// TIA Portal V20 export
FUNCTION_BLOCK "Sequence_3_SideTapeFixStage"   // FB32853, LAD
TITLE = Sequence
// Sequence template programmend in ladder logic
// stored: IsIECCheckEnabled true, MemoryReserve 100, Namespace Unit1.Em4, SetENOAutomatically true
   VAR_INPUT
      unitStatus { ExternalAccessible := 'False'; ExternalVisible := 'False'; ExternalWritable := 'False'} : "LAF_typeUnitStatus";   // Current unit status o be used in this EM
   END_VAR
   VAR
      instSequenceLADControl { ExternalWritable := 'False'} : "LAF_ControlLadSequence";
      instSequenceLADStatus { ExternalWritable := 'False'} : "LAF_StatusLadSequence";
      NoDataCheck { S7_SetPoint := 'True'} : "LER_typePartData";
      statTonTime { ExternalWritable := 'False'} : Array[0..9999] of TON_TIME;
   END_VAR
   VAR_TEMP
      tempCustomerAction : Bool;   // Placeholder for possible actions
      tempDo_nothing_and_wait_for_init : Bool;   // Placeholder for doing nothing
      tempSafeStateCondition : Bool;   // Temp Condition for the equipment module to be in a safe state
   END_VAR
   VAR CONSTANT
      stepDelayTime : Time := T#100ms;
      actionDelayTime : Time := T#1s;
      lowDelayTime : Time := T#300ms;
      STEP_IDLE : DInt := 1;
      JOB_1_STEP_01 : DInt := 101;
      JOB_1_STEP_10 : DInt := 110;
      JOB_1_STEP_11 : DInt := 111;
      JOB_1_STEP_20 : DInt := 120;
      JOB_1_STEP_30 : DInt := 130;
      JOB_1_STEP_31 : DInt := 131;
      JOB_1_STEP_32 : DInt := 132;
      JOB_1_STEP_33 : DInt := 133;
      JOB_1_STEP_34 : DInt := 134;
      JOB_1_STEP_35 : DInt := 135;
      JOB_1_STEP_40 : DInt := 140;
      JOB_1_STEP_50 : DInt := 150;
      JOB_1_STEP_60 : DInt := 160;
      JOB_1_STEP_70 : DInt := 170;
      JOB_1_STEP_80 : DInt := 180;
      JOB_1_STEP_90 : DInt := 190;
      JOB_2_STEP_01 : DInt := 201;
      JOB_2_STEP_10 : DInt := 210;
      JOB_2_STEP_11 : DInt := 211;
      JOB_2_STEP_12 : DInt := 212;
      JOB_2_STEP_13 : DInt := 213;
      JOB_2_STEP_14 : DInt := 214;
      JOB_2_STEP_20 : DInt := 220;
      JOB_2_STEP_21 : DInt := 221;
      JOB_2_STEP_22 : DInt := 222;
      JOB_2_STEP_23 : DInt := 223;
      JOB_2_STEP_24 : DInt := 224;
      JOB_2_STEP_30 : DInt := 230;
      JOB_2_STEP_31 : DInt := 231;
      JOB_2_STEP_32 : DInt := 232;
      JOB_2_STEP_40 : DInt := 240;
      JOB_2_STEP_50 : DInt := 250;
      JOB_2_STEP_60 : DInt := 260;
      JOB_2_STEP_70 : DInt := 270;
      JOB_2_STEP_80 : DInt := 280;
      JOB_2_STEP_90 : DInt := 290;
      JOB_3_STEP_01 : DInt := 301;
      JOB_3_STEP_02 : DInt := 302;
      JOB_3_STEP_03 : DInt := 303;
      JOB_3_STEP_10 : DInt := 310;
      JOB_3_STEP_11 : DInt := 311;
      JOB_3_STEP_12 : DInt := 312;
      JOB_3_STEP_13 : DInt := 313;
      JOB_3_STEP_14 : DInt := 314;
      JOB_3_STEP_15 : DInt := 315;
      JOB_3_STEP_16 : DInt := 316;
      JOB_3_STEP_17 : DInt := 317;
      JOB_3_STEP_20 : DInt := 320;
      JOB_3_STEP_21 : DInt := 321;
      JOB_3_STEP_22 : DInt := 322;
      JOB_3_STEP_23 : DInt := 323;
      JOB_3_STEP_24 : DInt := 324;
      JOB_3_STEP_25 : DInt := 325;
      JOB_3_STEP_26 : DInt := 326;
      JOB_3_STEP_27 : DInt := 327;
      JOB_3_STEP_30 : DInt := 330;
      JOB_3_STEP_31 : DInt := 331;
      JOB_3_STEP_32 : DInt := 332;
      JOB_3_STEP_33 : DInt := 333;
      JOB_3_STEP_34 : DInt := 334;
      JOB_3_STEP_35 : DInt := 335;
      JOB_3_STEP_36 : DInt := 336;
      JOB_3_STEP_37 : DInt := 337;
      JOB_3_STEP_40 : DInt := 340;
      JOB_3_STEP_41 : DInt := 341;
      JOB_3_STEP_42 : DInt := 342;
      JOB_3_STEP_43 : DInt := 343;
      JOB_3_STEP_44 : DInt := 344;
      JOB_3_STEP_45 : DInt := 345;
      JOB_3_STEP_46 : DInt := 346;
      JOB_3_STEP_47 : DInt := 347;
      JOB_3_STEP_50 : DInt := 350;
      JOB_3_STEP_60 : DInt := 360;
      JOB_3_STEP_70 : DInt := 370;
      JOB_3_STEP_80 : DInt := 380;
      JOB_3_STEP_90 : DInt := 390;
      JOB_4_STEP_01 : DInt := 401;
      JOB_4_STEP_10 : DInt := 410;
      JOB_4_STEP_11 : DInt := 411;
      JOB_4_STEP_12 : DInt := 412;
      JOB_4_STEP_20 : DInt := 420;
      JOB_4_STEP_21 : DInt := 421;
      JOB_4_STEP_22 : DInt := 422;
      JOB_4_STEP_23 : DInt := 423;
      JOB_4_STEP_24 : DInt := 424;
      JOB_4_STEP_25 : DInt := 425;
      JOB_4_STEP_30 : DInt := 430;
      JOB_4_STEP_40 : DInt := 440;
      JOB_4_STEP_50 : DInt := 450;
      JOB_4_STEP_60 : DInt := 460;
      JOB_4_STEP_70 : DInt := 470;
      JOB_4_STEP_80 : DInt := 480;
      JOB_4_STEP_90 : DInt := 490;
      JOB_5_STEP_01 : DInt := 501;
      JOB_5_STEP_10 : DInt := 510;
      JOB_5_STEP_11 : DInt := 511;
      JOB_5_STEP_12 : DInt := 512;
      JOB_5_STEP_20 : DInt := 520;
      JOB_5_STEP_30 : DInt := 530;
      JOB_5_STEP_40 : DInt := 540;
      JOB_5_STEP_50 : DInt := 550;
      JOB_5_STEP_60 : DInt := 560;
      JOB_5_STEP_70 : DInt := 570;
      JOB_5_STEP_80 : DInt := 580;
      JOB_5_STEP_90 : DInt := 590;
      JOB_6_STEP_01 : DInt := 601;
      JOB_6_STEP_10 : DInt := 610;
      JOB_6_STEP_11 : DInt := 611;
      JOB_6_STEP_12 : DInt := 612;
      JOB_6_STEP_20 : DInt := 620;
      JOB_6_STEP_21 : DInt := 621;
      JOB_6_STEP_22 : DInt := 622;
      JOB_6_STEP_30 : DInt := 630;
      JOB_6_STEP_40 : DInt := 640;
      JOB_6_STEP_50 : DInt := 650;
      JOB_6_STEP_60 : DInt := 660;
      JOB_6_STEP_70 : DInt := 670;
      JOB_6_STEP_80 : DInt := 680;
      JOB_6_STEP_90 : DInt := 690;
      JOB_7_STEP_01 : DInt := 701;
      JOB_7_STEP_10 : DInt := 710;
      JOB_7_STEP_20 : DInt := 720;
      JOB_7_STEP_21 : DInt := 721;
      JOB_7_STEP_22 : DInt := 722;
      JOB_7_STEP_23 : DInt := 723;
      JOB_7_STEP_30 : DInt := 730;
      JOB_7_STEP_40 : DInt := 740;
      JOB_7_STEP_50 : DInt := 750;
      JOB_7_STEP_60 : DInt := 760;
      JOB_7_STEP_70 : DInt := 770;
      JOB_7_STEP_80 : DInt := 780;
      JOB_7_STEP_81 : DInt := 781;
      JOB_7_STEP_82 : DInt := 782;
      JOB_7_STEP_90 : DInt := 790;
      STEP_IMMEDIATE_STOP : DInt := 9001;   // Step executed when an immediate stop command is triggered for the sequence (i.e. when unit is in state aborting)
      TO_DO_INSERT_ACTIONS_HERE : Bool := TRUE;   // Template : Add actions
      TO_DO_INSERT_CONDITION_FOR_TRANSITION_HERE : Bool := TRUE;   // Template : Add conditions
   END_VAR
   VAR_TEMP   // added for the SCL form of the ladder/FBD networks
      _w1 : Bool;
      _w2 : Bool;
      _w3 : Bool;
   END_VAR
BEGIN

REGION Network 1: BLOCK INFO HEADER
   // (company) / (C) Copyright (year)
   // ---------------------------------------------------------------------------------
   // Title:                             (Title of this block)
   // Comment/Function: (that is implemented in the block)
   // Library/Family:           (that the source is dedicated to)
   // Author:                        (department / person in charge / contact)
   // Target System:          (test system with FW version)
   // Engineering:              TIA Portal (SW version)
   // Restrictions:               (OB types, etc.)
   // Requirements:           (hardware, technological package, etc.)
   // ---------------------------------------------------------------------------------
   // Change log table:
   // Version          | Date             | Signature      | Expert in charge  | Changes applied ------------------------|----------------------|-------------------------|--------------------------------|-----------------------
   // 001.000.000 | yyyy-mm-dd | 0x00000000 | (name of expert) | First released version
END_REGION

REGION Network 2: DESCRIPTION
   // This is a template block provided by the Automation Framework. It can be used to create an own project.
   // The Block Info Header is prepared to put in your own data.
   // Description of the block could be added here and the docu created by Code2Docu.
END_REGION

REGION Network 3: *************** CONTROL **********************
END_REGION

REGION Network 4: Sequence Control ("Enter your Sequins number here")
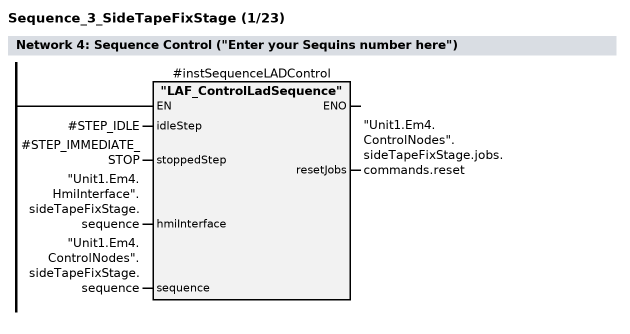
   RUNG wire#powerrail
      #instSequenceLADControl(idleStep := #STEP_IDLE, stoppedStep := #STEP_IMMEDIATE_STOP, hmiInterface := "Unit1.Em4.HmiInterface".sideTapeFixStage.sequence, sequence := "Unit1.Em4.ControlNodes".sideTapeFixStage.sequence, resetJobs => "Unit1.Em4.ControlNodes".sideTapeFixStage.jobs.commands.reset)
   END_RUNG
   // the same network as SCL:
   #instSequenceLADControl(idleStep := #STEP_IDLE,   // "LAF_ControlLadSequence"
                           stoppedStep := #STEP_IMMEDIATE_STOP,
                           hmiInterface := "Unit1.Em4.HmiInterface".sideTapeFixStage.sequence,
                           sequence := "Unit1.Em4.ControlNodes".sideTapeFixStage.sequence,
                           resetJobs => "Unit1.Em4.ControlNodes".sideTapeFixStage.jobs.commands.reset);
END_REGION

REGION Network 5: Step IDLE
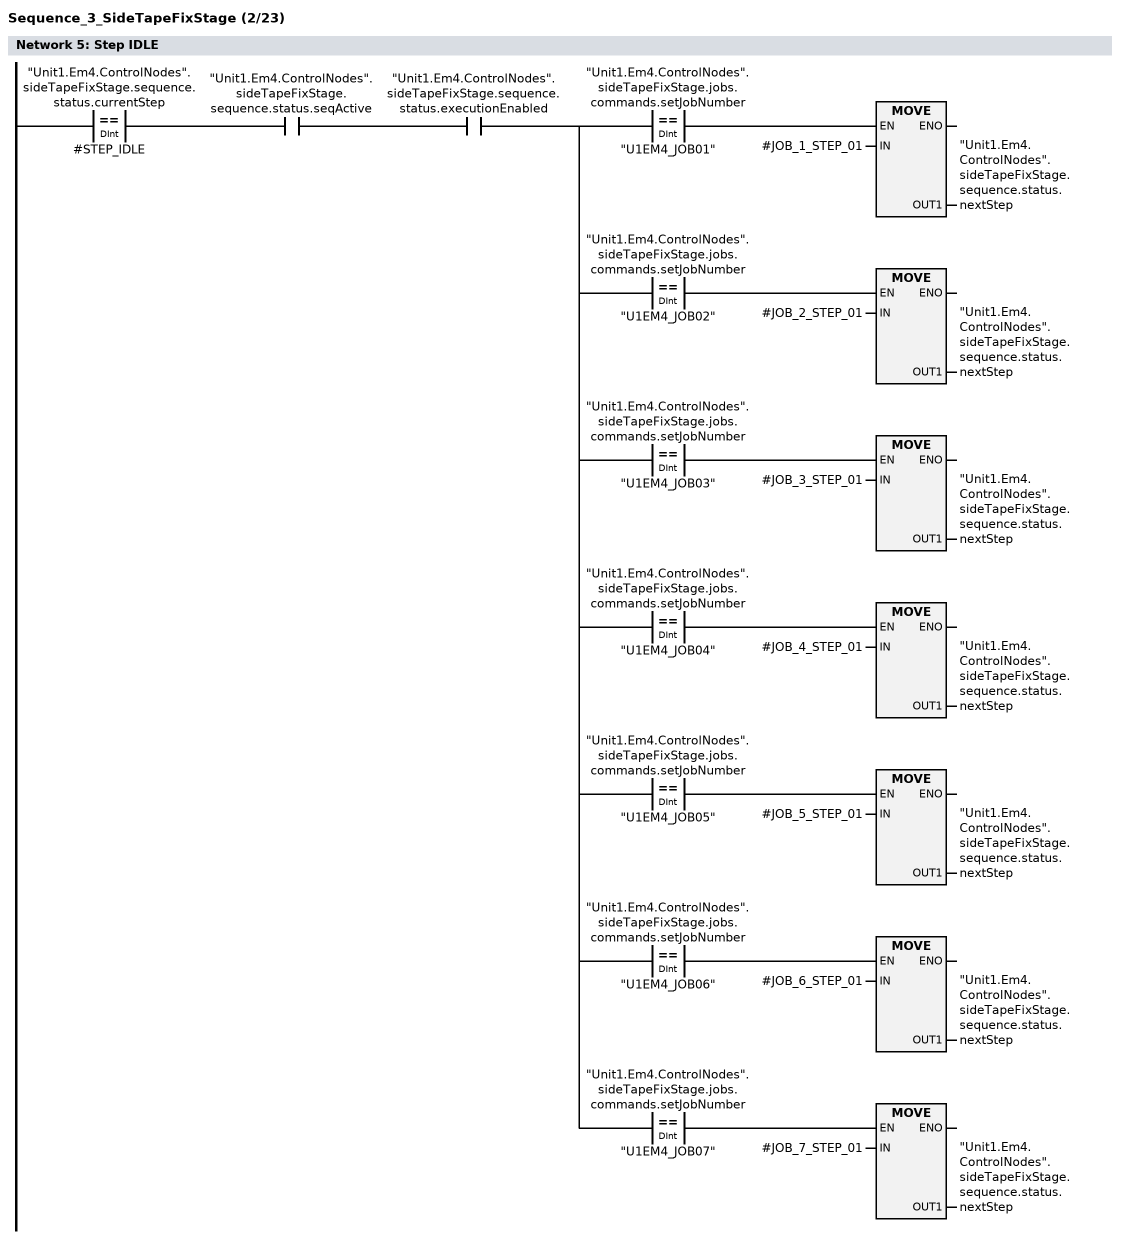
   RUNG wire#powerrail
      { S7_Templates := "SrcType := DInt" } EQ_Contact(in1 := "Unit1.Em4.ControlNodes".sideTapeFixStage.sequence.status.currentStep, in2 := #STEP_IDLE)
      Contact( "Unit1.Em4.ControlNodes".sideTapeFixStage.sequence.status.seqActive )
      Contact( "Unit1.Em4.ControlNodes".sideTapeFixStage.sequence.status.executionEnabled )
      wire#w1
      { S7_Templates := "SrcType := DInt" } EQ_Contact(in1 := "Unit1.Em4.ControlNodes".sideTapeFixStage.jobs.commands.setJobNumber, in2 := "U1EM4_JOB01")
      Move(in := #JOB_1_STEP_01, out1 => "Unit1.Em4.ControlNodes".sideTapeFixStage.sequence.status.nextStep)
   END_RUNG
   RUNG wire#w1
      { S7_Templates := "SrcType := DInt" } EQ_Contact(in1 := "Unit1.Em4.ControlNodes".sideTapeFixStage.jobs.commands.setJobNumber, in2 := "U1EM4_JOB02")
      Move(in := #JOB_2_STEP_01, out1 => "Unit1.Em4.ControlNodes".sideTapeFixStage.sequence.status.nextStep)
   END_RUNG
   RUNG wire#w1
      { S7_Templates := "SrcType := DInt" } EQ_Contact(in1 := "Unit1.Em4.ControlNodes".sideTapeFixStage.jobs.commands.setJobNumber, in2 := "U1EM4_JOB03")
      Move(in := #JOB_3_STEP_01, out1 => "Unit1.Em4.ControlNodes".sideTapeFixStage.sequence.status.nextStep)
   END_RUNG
   RUNG wire#w1
      { S7_Templates := "SrcType := DInt" } EQ_Contact(in1 := "Unit1.Em4.ControlNodes".sideTapeFixStage.jobs.commands.setJobNumber, in2 := "U1EM4_JOB04")
      Move(in := #JOB_4_STEP_01, out1 => "Unit1.Em4.ControlNodes".sideTapeFixStage.sequence.status.nextStep)
   END_RUNG
   RUNG wire#w1
      { S7_Templates := "SrcType := DInt" } EQ_Contact(in1 := "Unit1.Em4.ControlNodes".sideTapeFixStage.jobs.commands.setJobNumber, in2 := "U1EM4_JOB05")
      Move(in := #JOB_5_STEP_01, out1 => "Unit1.Em4.ControlNodes".sideTapeFixStage.sequence.status.nextStep)
   END_RUNG
   RUNG wire#w1
      { S7_Templates := "SrcType := DInt" } EQ_Contact(in1 := "Unit1.Em4.ControlNodes".sideTapeFixStage.jobs.commands.setJobNumber, in2 := "U1EM4_JOB06")
      Move(in := #JOB_6_STEP_01, out1 => "Unit1.Em4.ControlNodes".sideTapeFixStage.sequence.status.nextStep)
   END_RUNG
   RUNG wire#w1
      { S7_Templates := "SrcType := DInt" } EQ_Contact(in1 := "Unit1.Em4.ControlNodes".sideTapeFixStage.jobs.commands.setJobNumber, in2 := "U1EM4_JOB07")
      Move(in := #JOB_7_STEP_01, out1 => "Unit1.Em4.ControlNodes".sideTapeFixStage.sequence.status.nextStep)
   END_RUNG
   // the same network as SCL:
   #_w1 := ("Unit1.Em4.ControlNodes".sideTapeFixStage.sequence.status.currentStep = #STEP_IDLE) AND "Unit1.Em4.ControlNodes".sideTapeFixStage.sequence.status.seqActive AND "Unit1.Em4.ControlNodes".sideTapeFixStage.sequence.status.executionEnabled;
   IF #_w1 AND ("Unit1.Em4.ControlNodes".sideTapeFixStage.jobs.commands.setJobNumber = "U1EM4_JOB01") THEN
       "Unit1.Em4.ControlNodes".sideTapeFixStage.sequence.status.nextStep := #JOB_1_STEP_01;
   END_IF;
   IF #_w1 AND ("Unit1.Em4.ControlNodes".sideTapeFixStage.jobs.commands.setJobNumber = "U1EM4_JOB02") THEN
       "Unit1.Em4.ControlNodes".sideTapeFixStage.sequence.status.nextStep := #JOB_2_STEP_01;
   END_IF;
   IF #_w1 AND ("Unit1.Em4.ControlNodes".sideTapeFixStage.jobs.commands.setJobNumber = "U1EM4_JOB03") THEN
       "Unit1.Em4.ControlNodes".sideTapeFixStage.sequence.status.nextStep := #JOB_3_STEP_01;
   END_IF;
   IF #_w1 AND ("Unit1.Em4.ControlNodes".sideTapeFixStage.jobs.commands.setJobNumber = "U1EM4_JOB04") THEN
       "Unit1.Em4.ControlNodes".sideTapeFixStage.sequence.status.nextStep := #JOB_4_STEP_01;
   END_IF;
   IF #_w1 AND ("Unit1.Em4.ControlNodes".sideTapeFixStage.jobs.commands.setJobNumber = "U1EM4_JOB05") THEN
       "Unit1.Em4.ControlNodes".sideTapeFixStage.sequence.status.nextStep := #JOB_5_STEP_01;
   END_IF;
   IF #_w1 AND ("Unit1.Em4.ControlNodes".sideTapeFixStage.jobs.commands.setJobNumber = "U1EM4_JOB06") THEN
       "Unit1.Em4.ControlNodes".sideTapeFixStage.sequence.status.nextStep := #JOB_6_STEP_01;
   END_IF;
   IF #_w1 AND ("Unit1.Em4.ControlNodes".sideTapeFixStage.jobs.commands.setJobNumber = "U1EM4_JOB07") THEN
       "Unit1.Em4.ControlNodes".sideTapeFixStage.sequence.status.nextStep := #JOB_7_STEP_01;
   END_IF;
END_REGION

REGION Network 7: *************** JOB[1] HOMING *************************
END_REGION

REGION Network 8: Step[101] : JOB[1] Condition
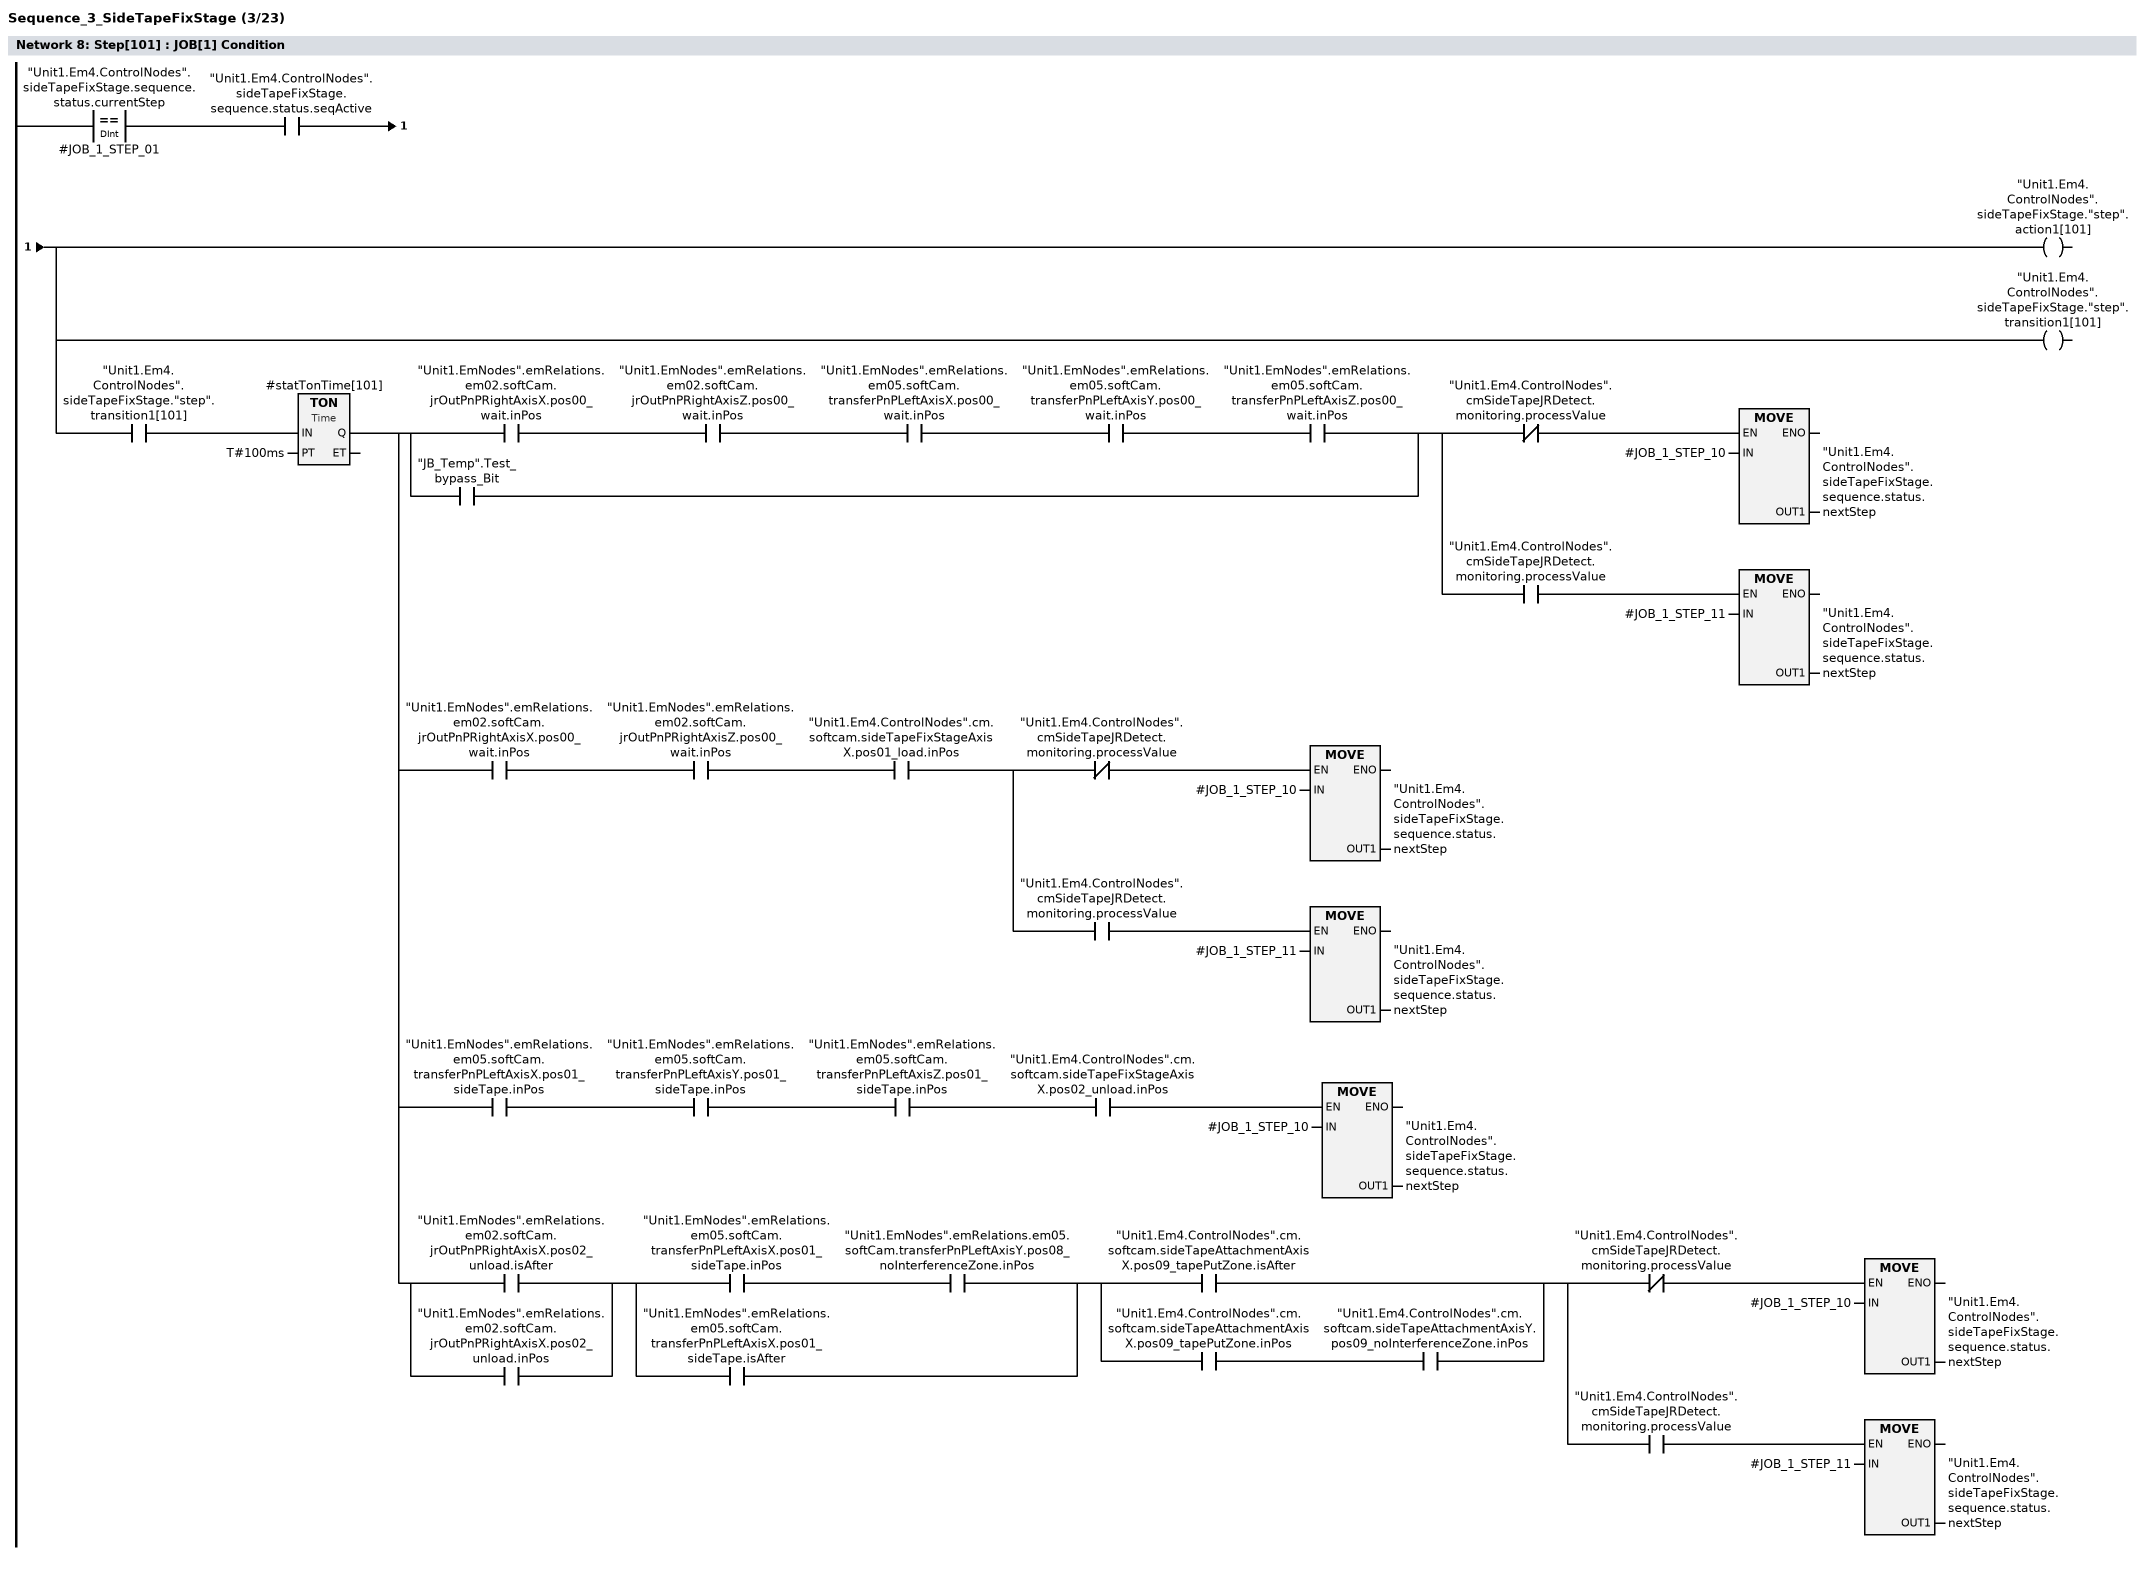
   RUNG wire#powerrail
      { S7_Templates := "SrcType := DInt" } EQ_Contact(in1 := "Unit1.Em4.ControlNodes".sideTapeFixStage.sequence.status.currentStep, in2 := #JOB_1_STEP_01)
      Contact( "Unit1.Em4.ControlNodes".sideTapeFixStage.sequence.status.seqActive )
      wire#w1
      Coil( "Unit1.Em4.ControlNodes".sideTapeFixStage."step".action1[101] )
   END_RUNG
   RUNG wire#w1
      Coil( "Unit1.Em4.ControlNodes".sideTapeFixStage."step".transition1[101] )
   END_RUNG
   RUNG wire#w1
      Contact( "Unit1.Em4.ControlNodes".sideTapeFixStage."step".transition1[101] )
      { S7_Templates := "time_type := Time" } #statTonTime[101].TON(pt := T#100ms, et =>)
      wire#w2
      Contact( "Unit1.EmNodes".emRelations.em02.softCam.jrOutPnPRightAxisX.pos00_wait.inPos )
      Contact( "Unit1.EmNodes".emRelations.em02.softCam.jrOutPnPRightAxisZ.pos00_wait.inPos )
      Contact( "Unit1.EmNodes".emRelations.em05.softCam.transferPnPLeftAxisX.pos00_wait.inPos )
      Contact( "Unit1.EmNodes".emRelations.em05.softCam.transferPnPLeftAxisY.pos00_wait.inPos )
      Contact( "Unit1.EmNodes".emRelations.em05.softCam.transferPnPLeftAxisZ.pos00_wait.inPos )
      wire#w3
      I_Contact( "Unit1.Em4.ControlNodes".cmSideTapeJRDetect.monitoring.processValue )
      Move(in := #JOB_1_STEP_10, out1 => "Unit1.Em4.ControlNodes".sideTapeFixStage.sequence.status.nextStep)
   END_RUNG
   RUNG wire#w2
      Contact( "JB_Temp".Test_bypass_Bit )
   END_RUNG wire#w3
   RUNG wire#w3
      Contact( "Unit1.Em4.ControlNodes".cmSideTapeJRDetect.monitoring.processValue )
      Move(in := #JOB_1_STEP_11, out1 => "Unit1.Em4.ControlNodes".sideTapeFixStage.sequence.status.nextStep)
   END_RUNG
   RUNG wire#w2
      Contact( "Unit1.EmNodes".emRelations.em02.softCam.jrOutPnPRightAxisX.pos00_wait.inPos )
      Contact( "Unit1.EmNodes".emRelations.em02.softCam.jrOutPnPRightAxisZ.pos00_wait.inPos )
      Contact( "Unit1.Em4.ControlNodes".cm.softcam.sideTapeFixStageAxisX.pos01_load.inPos )
      wire#w4
      I_Contact( "Unit1.Em4.ControlNodes".cmSideTapeJRDetect.monitoring.processValue )
      Move(in := #JOB_1_STEP_10, out1 => "Unit1.Em4.ControlNodes".sideTapeFixStage.sequence.status.nextStep)
   END_RUNG
   RUNG wire#w4
      Contact( "Unit1.Em4.ControlNodes".cmSideTapeJRDetect.monitoring.processValue )
      Move(in := #JOB_1_STEP_11, out1 => "Unit1.Em4.ControlNodes".sideTapeFixStage.sequence.status.nextStep)
   END_RUNG
   RUNG wire#w2
      Contact( "Unit1.EmNodes".emRelations.em05.softCam.transferPnPLeftAxisX.pos01_sideTape.inPos )
      Contact( "Unit1.EmNodes".emRelations.em05.softCam.transferPnPLeftAxisY.pos01_sideTape.inPos )
      Contact( "Unit1.EmNodes".emRelations.em05.softCam.transferPnPLeftAxisZ.pos01_sideTape.inPos )
      Contact( "Unit1.Em4.ControlNodes".cm.softcam.sideTapeFixStageAxisX.pos02_unload.inPos )
      Move(in := #JOB_1_STEP_10, out1 => "Unit1.Em4.ControlNodes".sideTapeFixStage.sequence.status.nextStep)
   END_RUNG
   RUNG wire#w2
      Contact( "Unit1.EmNodes".emRelations.em02.softCam.jrOutPnPRightAxisX.pos02_unload.isAfter )
      wire#w5
      Contact( "Unit1.EmNodes".emRelations.em05.softCam.transferPnPLeftAxisX.pos01_sideTape.inPos )
      Contact( "Unit1.EmNodes".emRelations.em05.softCam.transferPnPLeftAxisY.pos08_noInterferenceZone.inPos )
      wire#w6
      Contact( "Unit1.Em4.ControlNodes".cm.softcam.sideTapeAttachmentAxisX.pos09_tapePutZone.isAfter )
      wire#w7
      I_Contact( "Unit1.Em4.ControlNodes".cmSideTapeJRDetect.monitoring.processValue )
      Move(in := #JOB_1_STEP_10, out1 => "Unit1.Em4.ControlNodes".sideTapeFixStage.sequence.status.nextStep)
   END_RUNG
   RUNG wire#w2
      Contact( "Unit1.EmNodes".emRelations.em02.softCam.jrOutPnPRightAxisX.pos02_unload.inPos )
   END_RUNG wire#w5
   RUNG wire#w5
      Contact( "Unit1.EmNodes".emRelations.em05.softCam.transferPnPLeftAxisX.pos01_sideTape.isAfter )
   END_RUNG wire#w6
   RUNG wire#w6
      Contact( "Unit1.Em4.ControlNodes".cm.softcam.sideTapeAttachmentAxisX.pos09_tapePutZone.inPos )
      Contact( "Unit1.Em4.ControlNodes".cm.softcam.sideTapeAttachmentAxisY.pos09_noInterferenceZone.inPos )
   END_RUNG wire#w7
   RUNG wire#w7
      Contact( "Unit1.Em4.ControlNodes".cmSideTapeJRDetect.monitoring.processValue )
      Move(in := #JOB_1_STEP_11, out1 => "Unit1.Em4.ControlNodes".sideTapeFixStage.sequence.status.nextStep)
   END_RUNG
   // the same network as SCL:
   "Unit1.Em4.ControlNodes".sideTapeFixStage."step".action1[101] := ("Unit1.Em4.ControlNodes".sideTapeFixStage.sequence.status.currentStep = #JOB_1_STEP_01) AND "Unit1.Em4.ControlNodes".sideTapeFixStage.sequence.status.seqActive;
   "Unit1.Em4.ControlNodes".sideTapeFixStage."step".transition1[101] := ("Unit1.Em4.ControlNodes".sideTapeFixStage.sequence.status.currentStep = #JOB_1_STEP_01) AND "Unit1.Em4.ControlNodes".sideTapeFixStage.sequence.status.seqActive;
   #statTonTime[101].TON(IN := ("Unit1.Em4.ControlNodes".sideTapeFixStage.sequence.status.currentStep = #JOB_1_STEP_01) AND "Unit1.Em4.ControlNodes".sideTapeFixStage.sequence.status.seqActive AND "Unit1.Em4.ControlNodes".sideTapeFixStage."step".transition1[101],
                         PT := T#100ms);
   #_w1 := #statTonTime[101].Q AND (("Unit1.EmNodes".emRelations.em02.softCam.jrOutPnPRightAxisX.pos00_wait.inPos AND "Unit1.EmNodes".emRelations.em02.softCam.jrOutPnPRightAxisZ.pos00_wait.inPos AND "Unit1.EmNodes".emRelations.em05.softCam.transferPnPLeftAxisX.pos00_wait.inPos AND "Unit1.EmNodes".emRelations.em05.softCam.transferPnPLeftAxisY.pos00_wait.inPos AND "Unit1.EmNodes".emRelations.em05.softCam.transferPnPLeftAxisZ.pos00_wait.inPos) OR "JB_Temp".Test_bypass_Bit);
   IF #_w1 AND NOT "Unit1.Em4.ControlNodes".cmSideTapeJRDetect.monitoring.processValue THEN
       "Unit1.Em4.ControlNodes".sideTapeFixStage.sequence.status.nextStep := #JOB_1_STEP_10;
   END_IF;
   IF #_w1 AND "Unit1.Em4.ControlNodes".cmSideTapeJRDetect.monitoring.processValue THEN
       "Unit1.Em4.ControlNodes".sideTapeFixStage.sequence.status.nextStep := #JOB_1_STEP_11;
   END_IF;
   #_w2 := #statTonTime[101].Q AND "Unit1.EmNodes".emRelations.em02.softCam.jrOutPnPRightAxisX.pos00_wait.inPos AND "Unit1.EmNodes".emRelations.em02.softCam.jrOutPnPRightAxisZ.pos00_wait.inPos AND "Unit1.Em4.ControlNodes".cm.softcam.sideTapeFixStageAxisX.pos01_load.inPos;
   IF #_w2 AND NOT "Unit1.Em4.ControlNodes".cmSideTapeJRDetect.monitoring.processValue THEN
       "Unit1.Em4.ControlNodes".sideTapeFixStage.sequence.status.nextStep := #JOB_1_STEP_10;
   END_IF;
   IF #_w2 AND "Unit1.Em4.ControlNodes".cmSideTapeJRDetect.monitoring.processValue THEN
       "Unit1.Em4.ControlNodes".sideTapeFixStage.sequence.status.nextStep := #JOB_1_STEP_11;
   END_IF;
   IF #statTonTime[101].Q AND "Unit1.EmNodes".emRelations.em05.softCam.transferPnPLeftAxisX.pos01_sideTape.inPos AND "Unit1.EmNodes".emRelations.em05.softCam.transferPnPLeftAxisY.pos01_sideTape.inPos AND "Unit1.EmNodes".emRelations.em05.softCam.transferPnPLeftAxisZ.pos01_sideTape.inPos AND "Unit1.Em4.ControlNodes".cm.softcam.sideTapeFixStageAxisX.pos02_unload.inPos THEN
       "Unit1.Em4.ControlNodes".sideTapeFixStage.sequence.status.nextStep := #JOB_1_STEP_10;
   END_IF;
   #_w3 := #statTonTime[101].Q AND ("Unit1.EmNodes".emRelations.em02.softCam.jrOutPnPRightAxisX.pos02_unload.isAfter OR "Unit1.EmNodes".emRelations.em02.softCam.jrOutPnPRightAxisX.pos02_unload.inPos) AND (("Unit1.EmNodes".emRelations.em05.softCam.transferPnPLeftAxisX.pos01_sideTape.inPos AND "Unit1.EmNodes".emRelations.em05.softCam.transferPnPLeftAxisY.pos08_noInterferenceZone.inPos) OR "Unit1.EmNodes".emRelations.em05.softCam.transferPnPLeftAxisX.pos01_sideTape.isAfter) AND ("Unit1.Em4.ControlNodes".cm.softcam.sideTapeAttachmentAxisX.pos09_tapePutZone.isAfter OR ("Unit1.Em4.ControlNodes".cm.softcam.sideTapeAttachmentAxisX.pos09_tapePutZone.inPos AND "Unit1.Em4.ControlNodes".cm.softcam.sideTapeAttachmentAxisY.pos09_noInterferenceZone.inPos));
   IF #_w3 AND NOT "Unit1.Em4.ControlNodes".cmSideTapeJRDetect.monitoring.processValue THEN
       "Unit1.Em4.ControlNodes".sideTapeFixStage.sequence.status.nextStep := #JOB_1_STEP_10;
   END_IF;
   IF #_w3 AND "Unit1.Em4.ControlNodes".cmSideTapeJRDetect.monitoring.processValue THEN
       "Unit1.Em4.ControlNodes".sideTapeFixStage.sequence.status.nextStep := #JOB_1_STEP_11;
   END_IF;
END_REGION

REGION Network 9: Step[110] : Side Tape Fix Stage Clamp Open
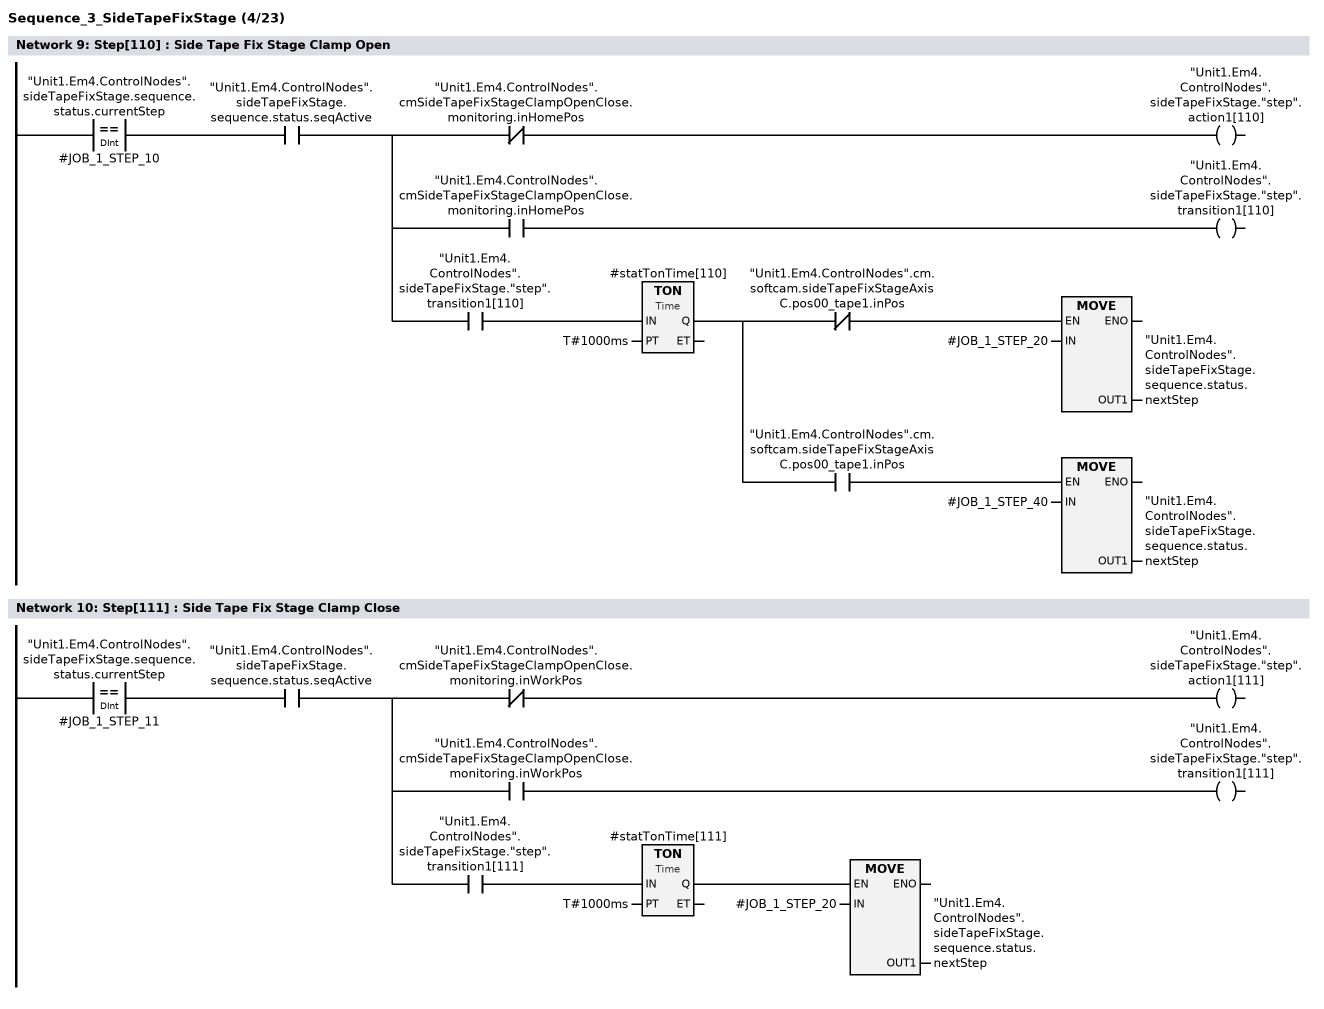
   RUNG wire#powerrail
      { S7_Templates := "SrcType := DInt" } EQ_Contact(in1 := "Unit1.Em4.ControlNodes".sideTapeFixStage.sequence.status.currentStep, in2 := #JOB_1_STEP_10)
      Contact( "Unit1.Em4.ControlNodes".sideTapeFixStage.sequence.status.seqActive )
      wire#w1
      I_Contact( "Unit1.Em4.ControlNodes".cmSideTapeFixStageClampOpenClose.monitoring.inHomePos )
      Coil( "Unit1.Em4.ControlNodes".sideTapeFixStage."step".action1[110] )
   END_RUNG
   RUNG wire#w1
      Contact( "Unit1.Em4.ControlNodes".cmSideTapeFixStageClampOpenClose.monitoring.inHomePos )
      Coil( "Unit1.Em4.ControlNodes".sideTapeFixStage."step".transition1[110] )
   END_RUNG
   RUNG wire#w1
      Contact( "Unit1.Em4.ControlNodes".sideTapeFixStage."step".transition1[110] )
      { S7_Templates := "time_type := Time" } #statTonTime[110].TON(pt := T#1000ms, et =>)
      wire#w2
      I_Contact( "Unit1.Em4.ControlNodes".cm.softcam.sideTapeFixStageAxisC.pos00_tape1.inPos )
      Move(in := #JOB_1_STEP_20, out1 => "Unit1.Em4.ControlNodes".sideTapeFixStage.sequence.status.nextStep)
   END_RUNG
   RUNG wire#w2
      Contact( "Unit1.Em4.ControlNodes".cm.softcam.sideTapeFixStageAxisC.pos00_tape1.inPos )
      Move(in := #JOB_1_STEP_40, out1 => "Unit1.Em4.ControlNodes".sideTapeFixStage.sequence.status.nextStep)
   END_RUNG
   // the same network as SCL:
   #_w1 := ("Unit1.Em4.ControlNodes".sideTapeFixStage.sequence.status.currentStep = #JOB_1_STEP_10) AND "Unit1.Em4.ControlNodes".sideTapeFixStage.sequence.status.seqActive;
   "Unit1.Em4.ControlNodes".sideTapeFixStage."step".action1[110] := #_w1 AND NOT "Unit1.Em4.ControlNodes".cmSideTapeFixStageClampOpenClose.monitoring.inHomePos;
   "Unit1.Em4.ControlNodes".sideTapeFixStage."step".transition1[110] := #_w1 AND "Unit1.Em4.ControlNodes".cmSideTapeFixStageClampOpenClose.monitoring.inHomePos;
   #statTonTime[110].TON(IN := #_w1 AND "Unit1.Em4.ControlNodes".sideTapeFixStage."step".transition1[110],
                         PT := T#1000ms);
   IF #statTonTime[110].Q AND NOT "Unit1.Em4.ControlNodes".cm.softcam.sideTapeFixStageAxisC.pos00_tape1.inPos THEN
       "Unit1.Em4.ControlNodes".sideTapeFixStage.sequence.status.nextStep := #JOB_1_STEP_20;
   END_IF;
   IF #statTonTime[110].Q AND "Unit1.Em4.ControlNodes".cm.softcam.sideTapeFixStageAxisC.pos00_tape1.inPos THEN
       "Unit1.Em4.ControlNodes".sideTapeFixStage.sequence.status.nextStep := #JOB_1_STEP_40;
   END_IF;
END_REGION

REGION Network 10: Step[111] : Side Tape Fix Stage Clamp Close
   RUNG wire#powerrail
      { S7_Templates := "SrcType := DInt" } EQ_Contact(in1 := "Unit1.Em4.ControlNodes".sideTapeFixStage.sequence.status.currentStep, in2 := #JOB_1_STEP_11)
      Contact( "Unit1.Em4.ControlNodes".sideTapeFixStage.sequence.status.seqActive )
      wire#w1
      I_Contact( "Unit1.Em4.ControlNodes".cmSideTapeFixStageClampOpenClose.monitoring.inWorkPos )
      Coil( "Unit1.Em4.ControlNodes".sideTapeFixStage."step".action1[111] )
   END_RUNG
   RUNG wire#w1
      Contact( "Unit1.Em4.ControlNodes".cmSideTapeFixStageClampOpenClose.monitoring.inWorkPos )
      Coil( "Unit1.Em4.ControlNodes".sideTapeFixStage."step".transition1[111] )
   END_RUNG
   RUNG wire#w1
      Contact( "Unit1.Em4.ControlNodes".sideTapeFixStage."step".transition1[111] )
      { S7_Templates := "time_type := Time" } #statTonTime[111].TON(pt := T#1000ms, et =>)
      Move(in := #JOB_1_STEP_20, out1 => "Unit1.Em4.ControlNodes".sideTapeFixStage.sequence.status.nextStep)
   END_RUNG
   // the same network as SCL:
   #_w1 := ("Unit1.Em4.ControlNodes".sideTapeFixStage.sequence.status.currentStep = #JOB_1_STEP_11) AND "Unit1.Em4.ControlNodes".sideTapeFixStage.sequence.status.seqActive;
   "Unit1.Em4.ControlNodes".sideTapeFixStage."step".action1[111] := #_w1 AND NOT "Unit1.Em4.ControlNodes".cmSideTapeFixStageClampOpenClose.monitoring.inWorkPos;
   "Unit1.Em4.ControlNodes".sideTapeFixStage."step".transition1[111] := #_w1 AND "Unit1.Em4.ControlNodes".cmSideTapeFixStageClampOpenClose.monitoring.inWorkPos;
   #statTonTime[111].TON(IN := #_w1 AND "Unit1.Em4.ControlNodes".sideTapeFixStage."step".transition1[111],
                         PT := T#1000ms);
   IF #statTonTime[111].Q THEN
       "Unit1.Em4.ControlNodes".sideTapeFixStage.sequence.status.nextStep := #JOB_1_STEP_20;
   END_IF;
END_REGION

REGION Network 11: Step[120] : Side Tape Fix Stage X-Axis Load Pos
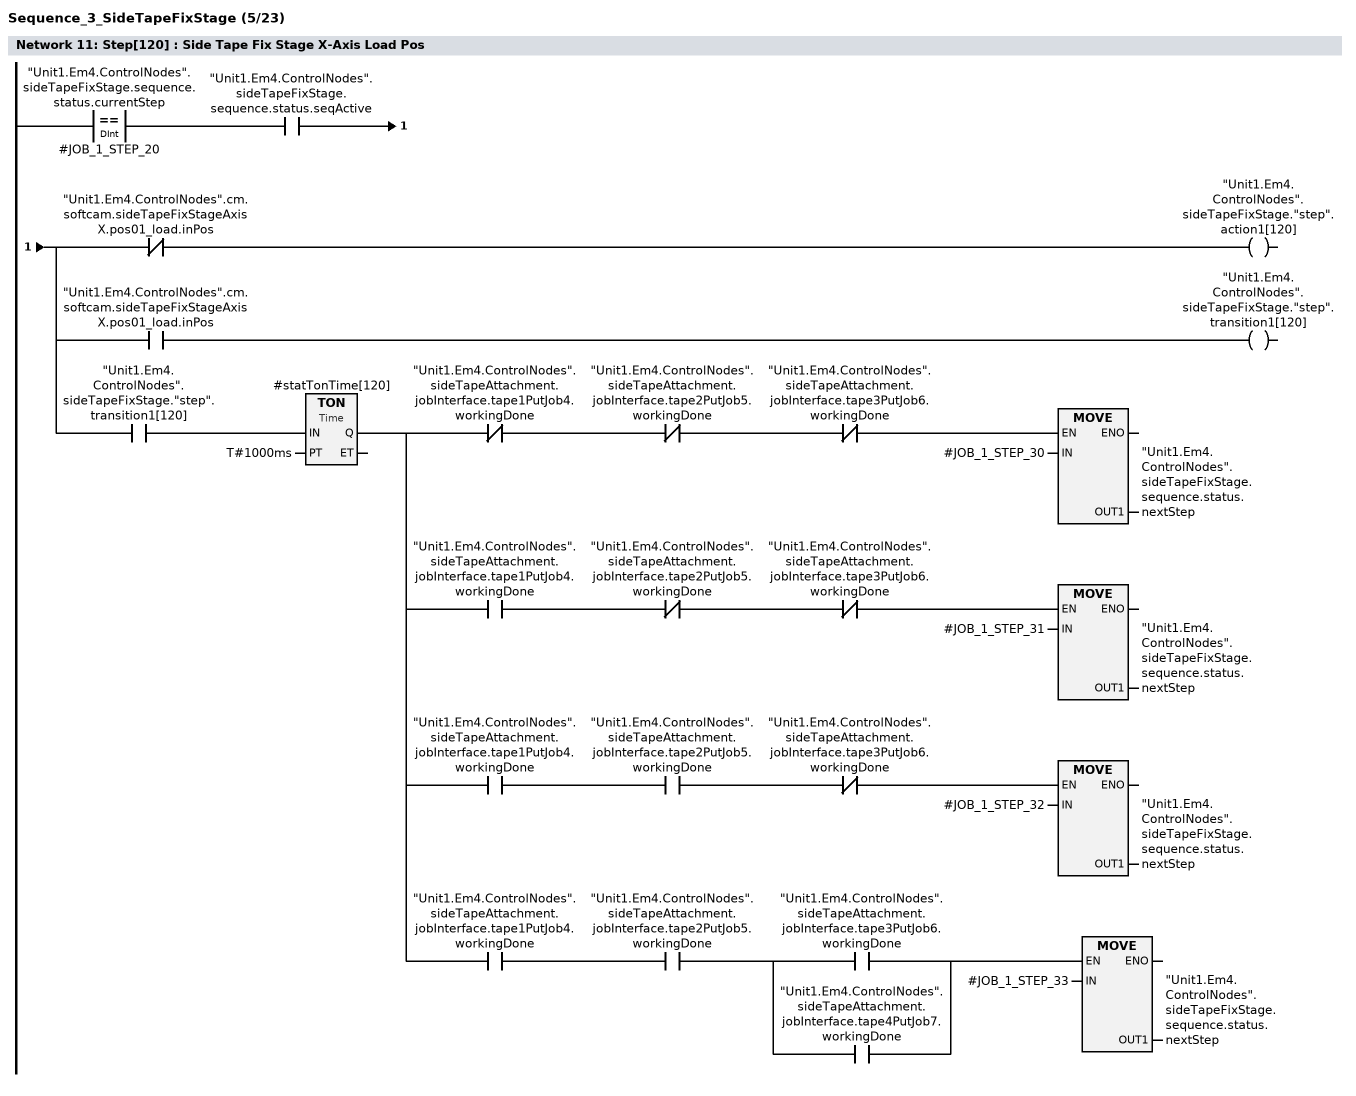
   RUNG wire#powerrail
      { S7_Templates := "SrcType := DInt" } EQ_Contact(in1 := "Unit1.Em4.ControlNodes".sideTapeFixStage.sequence.status.currentStep, in2 := #JOB_1_STEP_20)
      Contact( "Unit1.Em4.ControlNodes".sideTapeFixStage.sequence.status.seqActive )
      wire#w1
      I_Contact( "Unit1.Em4.ControlNodes".cm.softcam.sideTapeFixStageAxisX.pos01_load.inPos )
      Coil( "Unit1.Em4.ControlNodes".sideTapeFixStage."step".action1[120] )
   END_RUNG
   RUNG wire#w1
      Contact( "Unit1.Em4.ControlNodes".cm.softcam.sideTapeFixStageAxisX.pos01_load.inPos )
      Coil( "Unit1.Em4.ControlNodes".sideTapeFixStage."step".transition1[120] )
   END_RUNG
   RUNG wire#w1
      Contact( "Unit1.Em4.ControlNodes".sideTapeFixStage."step".transition1[120] )
      { S7_Templates := "time_type := Time" } #statTonTime[120].TON(pt := T#1000ms, et =>)
      wire#w2
      I_Contact( "Unit1.Em4.ControlNodes".sideTapeAttachment.jobInterface.tape1PutJob4.workingDone )
      I_Contact( "Unit1.Em4.ControlNodes".sideTapeAttachment.jobInterface.tape2PutJob5.workingDone )
      I_Contact( "Unit1.Em4.ControlNodes".sideTapeAttachment.jobInterface.tape3PutJob6.workingDone )
      Move(in := #JOB_1_STEP_30, out1 => "Unit1.Em4.ControlNodes".sideTapeFixStage.sequence.status.nextStep)
   END_RUNG
   RUNG wire#w2
      Contact( "Unit1.Em4.ControlNodes".sideTapeAttachment.jobInterface.tape1PutJob4.workingDone )
      I_Contact( "Unit1.Em4.ControlNodes".sideTapeAttachment.jobInterface.tape2PutJob5.workingDone )
      I_Contact( "Unit1.Em4.ControlNodes".sideTapeAttachment.jobInterface.tape3PutJob6.workingDone )
      Move(in := #JOB_1_STEP_31, out1 => "Unit1.Em4.ControlNodes".sideTapeFixStage.sequence.status.nextStep)
   END_RUNG
   RUNG wire#w2
      Contact( "Unit1.Em4.ControlNodes".sideTapeAttachment.jobInterface.tape1PutJob4.workingDone )
      Contact( "Unit1.Em4.ControlNodes".sideTapeAttachment.jobInterface.tape2PutJob5.workingDone )
      I_Contact( "Unit1.Em4.ControlNodes".sideTapeAttachment.jobInterface.tape3PutJob6.workingDone )
      Move(in := #JOB_1_STEP_32, out1 => "Unit1.Em4.ControlNodes".sideTapeFixStage.sequence.status.nextStep)
   END_RUNG
   RUNG wire#w2
      Contact( "Unit1.Em4.ControlNodes".sideTapeAttachment.jobInterface.tape1PutJob4.workingDone )
      Contact( "Unit1.Em4.ControlNodes".sideTapeAttachment.jobInterface.tape2PutJob5.workingDone )
      wire#w3
      Contact( "Unit1.Em4.ControlNodes".sideTapeAttachment.jobInterface.tape3PutJob6.workingDone )
      wire#w4
      Move(in := #JOB_1_STEP_33, out1 => "Unit1.Em4.ControlNodes".sideTapeFixStage.sequence.status.nextStep)
   END_RUNG
   RUNG wire#w3
      Contact( "Unit1.Em4.ControlNodes".sideTapeAttachment.jobInterface.tape4PutJob7.workingDone )
   END_RUNG wire#w4
   // the same network as SCL:
   #_w1 := ("Unit1.Em4.ControlNodes".sideTapeFixStage.sequence.status.currentStep = #JOB_1_STEP_20) AND "Unit1.Em4.ControlNodes".sideTapeFixStage.sequence.status.seqActive;
   "Unit1.Em4.ControlNodes".sideTapeFixStage."step".action1[120] := #_w1 AND NOT "Unit1.Em4.ControlNodes".cm.softcam.sideTapeFixStageAxisX.pos01_load.inPos;
   "Unit1.Em4.ControlNodes".sideTapeFixStage."step".transition1[120] := #_w1 AND "Unit1.Em4.ControlNodes".cm.softcam.sideTapeFixStageAxisX.pos01_load.inPos;
   #statTonTime[120].TON(IN := #_w1 AND "Unit1.Em4.ControlNodes".sideTapeFixStage."step".transition1[120],
                         PT := T#1000ms);
   IF #statTonTime[120].Q AND NOT "Unit1.Em4.ControlNodes".sideTapeAttachment.jobInterface.tape1PutJob4.workingDone AND NOT "Unit1.Em4.ControlNodes".sideTapeAttachment.jobInterface.tape2PutJob5.workingDone AND NOT "Unit1.Em4.ControlNodes".sideTapeAttachment.jobInterface.tape3PutJob6.workingDone THEN
       "Unit1.Em4.ControlNodes".sideTapeFixStage.sequence.status.nextStep := #JOB_1_STEP_30;
   END_IF;
   IF #statTonTime[120].Q AND "Unit1.Em4.ControlNodes".sideTapeAttachment.jobInterface.tape1PutJob4.workingDone AND NOT "Unit1.Em4.ControlNodes".sideTapeAttachment.jobInterface.tape2PutJob5.workingDone AND NOT "Unit1.Em4.ControlNodes".sideTapeAttachment.jobInterface.tape3PutJob6.workingDone THEN
       "Unit1.Em4.ControlNodes".sideTapeFixStage.sequence.status.nextStep := #JOB_1_STEP_31;
   END_IF;
   IF #statTonTime[120].Q AND "Unit1.Em4.ControlNodes".sideTapeAttachment.jobInterface.tape1PutJob4.workingDone AND "Unit1.Em4.ControlNodes".sideTapeAttachment.jobInterface.tape2PutJob5.workingDone AND NOT "Unit1.Em4.ControlNodes".sideTapeAttachment.jobInterface.tape3PutJob6.workingDone THEN
       "Unit1.Em4.ControlNodes".sideTapeFixStage.sequence.status.nextStep := #JOB_1_STEP_32;
   END_IF;
   IF #statTonTime[120].Q AND "Unit1.Em4.ControlNodes".sideTapeAttachment.jobInterface.tape1PutJob4.workingDone AND "Unit1.Em4.ControlNodes".sideTapeAttachment.jobInterface.tape2PutJob5.workingDone AND ("Unit1.Em4.ControlNodes".sideTapeAttachment.jobInterface.tape3PutJob6.workingDone OR "Unit1.Em4.ControlNodes".sideTapeAttachment.jobInterface.tape4PutJob7.workingDone) THEN
       "Unit1.Em4.ControlNodes".sideTapeFixStage.sequence.status.nextStep := #JOB_1_STEP_33;
   END_IF;
END_REGION

REGION Network 12: Step[130] : Side Tape Fix Stage C-Axis Wait Pos [Tape-1]
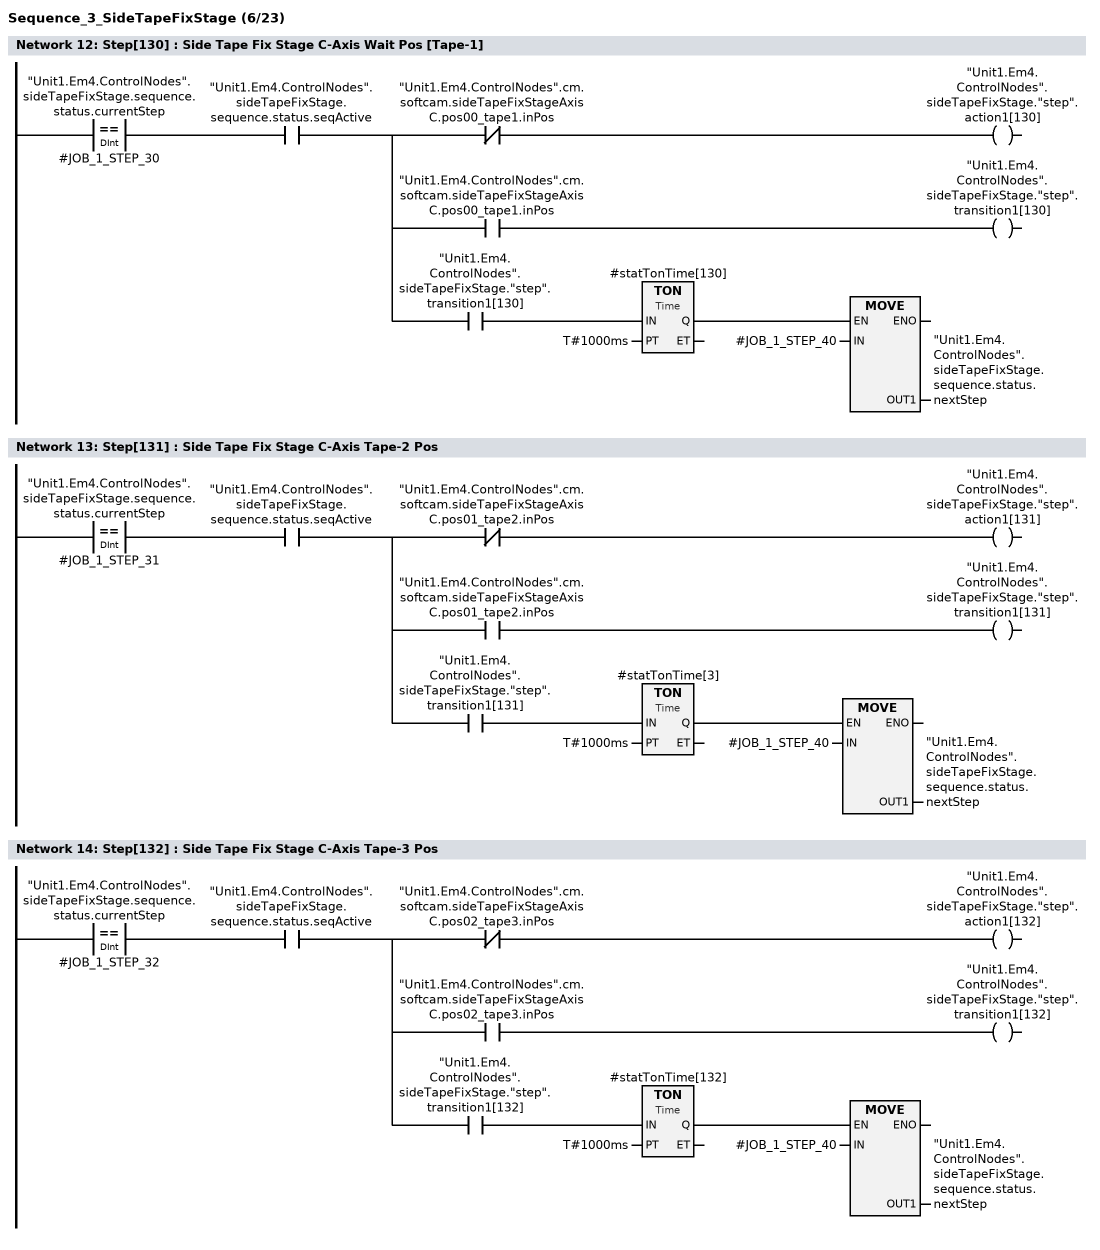
   RUNG wire#powerrail
      { S7_Templates := "SrcType := DInt" } EQ_Contact(in1 := "Unit1.Em4.ControlNodes".sideTapeFixStage.sequence.status.currentStep, in2 := #JOB_1_STEP_30)
      Contact( "Unit1.Em4.ControlNodes".sideTapeFixStage.sequence.status.seqActive )
      wire#w1
      I_Contact( "Unit1.Em4.ControlNodes".cm.softcam.sideTapeFixStageAxisC.pos00_tape1.inPos )
      Coil( "Unit1.Em4.ControlNodes".sideTapeFixStage."step".action1[130] )
   END_RUNG
   RUNG wire#w1
      Contact( "Unit1.Em4.ControlNodes".cm.softcam.sideTapeFixStageAxisC.pos00_tape1.inPos )
      Coil( "Unit1.Em4.ControlNodes".sideTapeFixStage."step".transition1[130] )
   END_RUNG
   RUNG wire#w1
      Contact( "Unit1.Em4.ControlNodes".sideTapeFixStage."step".transition1[130] )
      { S7_Templates := "time_type := Time" } #statTonTime[130].TON(pt := T#1000ms, et =>)
      Move(in := #JOB_1_STEP_40, out1 => "Unit1.Em4.ControlNodes".sideTapeFixStage.sequence.status.nextStep)
   END_RUNG
   // the same network as SCL:
   #_w1 := ("Unit1.Em4.ControlNodes".sideTapeFixStage.sequence.status.currentStep = #JOB_1_STEP_30) AND "Unit1.Em4.ControlNodes".sideTapeFixStage.sequence.status.seqActive;
   "Unit1.Em4.ControlNodes".sideTapeFixStage."step".action1[130] := #_w1 AND NOT "Unit1.Em4.ControlNodes".cm.softcam.sideTapeFixStageAxisC.pos00_tape1.inPos;
   "Unit1.Em4.ControlNodes".sideTapeFixStage."step".transition1[130] := #_w1 AND "Unit1.Em4.ControlNodes".cm.softcam.sideTapeFixStageAxisC.pos00_tape1.inPos;
   #statTonTime[130].TON(IN := #_w1 AND "Unit1.Em4.ControlNodes".sideTapeFixStage."step".transition1[130],
                         PT := T#1000ms);
   IF #statTonTime[130].Q THEN
       "Unit1.Em4.ControlNodes".sideTapeFixStage.sequence.status.nextStep := #JOB_1_STEP_40;
   END_IF;
END_REGION

REGION Network 13: Step[131] : Side Tape Fix Stage C-Axis Tape-2 Pos
   RUNG wire#powerrail
      { S7_Templates := "SrcType := DInt" } EQ_Contact(in1 := "Unit1.Em4.ControlNodes".sideTapeFixStage.sequence.status.currentStep, in2 := #JOB_1_STEP_31)
      Contact( "Unit1.Em4.ControlNodes".sideTapeFixStage.sequence.status.seqActive )
      wire#w1
      I_Contact( "Unit1.Em4.ControlNodes".cm.softcam.sideTapeFixStageAxisC.pos01_tape2.inPos )
      Coil( "Unit1.Em4.ControlNodes".sideTapeFixStage."step".action1[131] )
   END_RUNG
   RUNG wire#w1
      Contact( "Unit1.Em4.ControlNodes".cm.softcam.sideTapeFixStageAxisC.pos01_tape2.inPos )
      Coil( "Unit1.Em4.ControlNodes".sideTapeFixStage."step".transition1[131] )
   END_RUNG
   RUNG wire#w1
      Contact( "Unit1.Em4.ControlNodes".sideTapeFixStage."step".transition1[131] )
      { S7_Templates := "time_type := Time" } #statTonTime[3].TON(pt := T#1000ms, et =>)
      Move(in := #JOB_1_STEP_40, out1 => "Unit1.Em4.ControlNodes".sideTapeFixStage.sequence.status.nextStep)
   END_RUNG
   // the same network as SCL:
   #_w1 := ("Unit1.Em4.ControlNodes".sideTapeFixStage.sequence.status.currentStep = #JOB_1_STEP_31) AND "Unit1.Em4.ControlNodes".sideTapeFixStage.sequence.status.seqActive;
   "Unit1.Em4.ControlNodes".sideTapeFixStage."step".action1[131] := #_w1 AND NOT "Unit1.Em4.ControlNodes".cm.softcam.sideTapeFixStageAxisC.pos01_tape2.inPos;
   "Unit1.Em4.ControlNodes".sideTapeFixStage."step".transition1[131] := #_w1 AND "Unit1.Em4.ControlNodes".cm.softcam.sideTapeFixStageAxisC.pos01_tape2.inPos;
   #statTonTime[3].TON(IN := #_w1 AND "Unit1.Em4.ControlNodes".sideTapeFixStage."step".transition1[131],
                       PT := T#1000ms);
   IF #statTonTime[3].Q THEN
       "Unit1.Em4.ControlNodes".sideTapeFixStage.sequence.status.nextStep := #JOB_1_STEP_40;
   END_IF;
END_REGION

REGION Network 14: Step[132] : Side Tape Fix Stage C-Axis Tape-3 Pos
   RUNG wire#powerrail
      { S7_Templates := "SrcType := DInt" } EQ_Contact(in1 := "Unit1.Em4.ControlNodes".sideTapeFixStage.sequence.status.currentStep, in2 := #JOB_1_STEP_32)
      Contact( "Unit1.Em4.ControlNodes".sideTapeFixStage.sequence.status.seqActive )
      wire#w1
      I_Contact( "Unit1.Em4.ControlNodes".cm.softcam.sideTapeFixStageAxisC.pos02_tape3.inPos )
      Coil( "Unit1.Em4.ControlNodes".sideTapeFixStage."step".action1[132] )
   END_RUNG
   RUNG wire#w1
      Contact( "Unit1.Em4.ControlNodes".cm.softcam.sideTapeFixStageAxisC.pos02_tape3.inPos )
      Coil( "Unit1.Em4.ControlNodes".sideTapeFixStage."step".transition1[132] )
   END_RUNG
   RUNG wire#w1
      Contact( "Unit1.Em4.ControlNodes".sideTapeFixStage."step".transition1[132] )
      { S7_Templates := "time_type := Time" } #statTonTime[132].TON(pt := T#1000ms, et =>)
      Move(in := #JOB_1_STEP_40, out1 => "Unit1.Em4.ControlNodes".sideTapeFixStage.sequence.status.nextStep)
   END_RUNG
   // the same network as SCL:
   #_w1 := ("Unit1.Em4.ControlNodes".sideTapeFixStage.sequence.status.currentStep = #JOB_1_STEP_32) AND "Unit1.Em4.ControlNodes".sideTapeFixStage.sequence.status.seqActive;
   "Unit1.Em4.ControlNodes".sideTapeFixStage."step".action1[132] := #_w1 AND NOT "Unit1.Em4.ControlNodes".cm.softcam.sideTapeFixStageAxisC.pos02_tape3.inPos;
   "Unit1.Em4.ControlNodes".sideTapeFixStage."step".transition1[132] := #_w1 AND "Unit1.Em4.ControlNodes".cm.softcam.sideTapeFixStageAxisC.pos02_tape3.inPos;
   #statTonTime[132].TON(IN := #_w1 AND "Unit1.Em4.ControlNodes".sideTapeFixStage."step".transition1[132],
                         PT := T#1000ms);
   IF #statTonTime[132].Q THEN
       "Unit1.Em4.ControlNodes".sideTapeFixStage.sequence.status.nextStep := #JOB_1_STEP_40;
   END_IF;
END_REGION

REGION Network 15: Step[133] : Side Tape Fix Stage C-Axis Tape-4 Pos
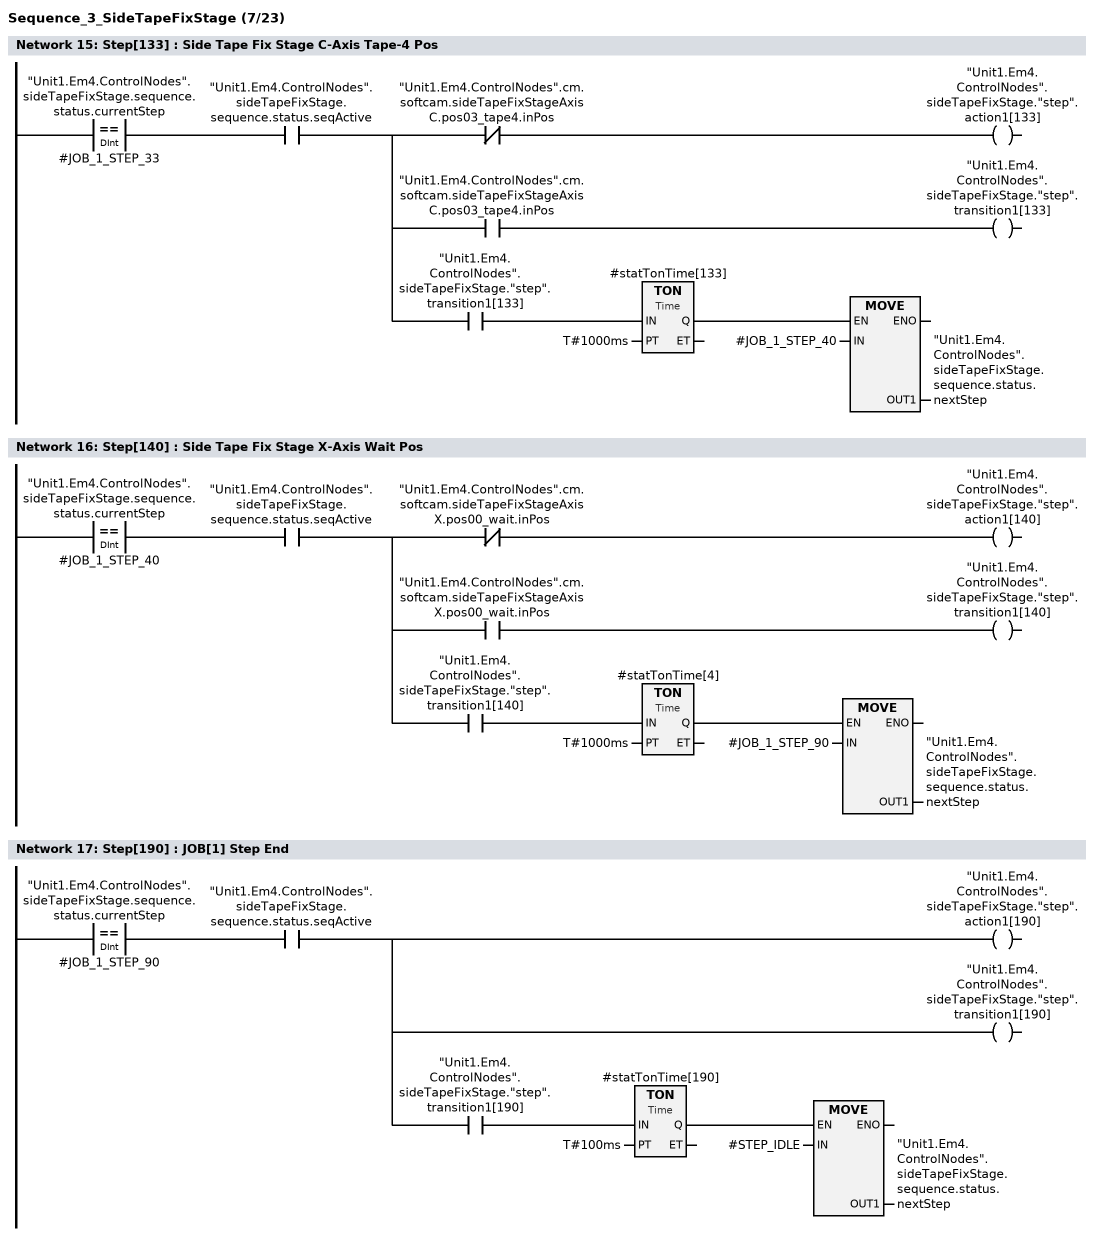
   RUNG wire#powerrail
      { S7_Templates := "SrcType := DInt" } EQ_Contact(in1 := "Unit1.Em4.ControlNodes".sideTapeFixStage.sequence.status.currentStep, in2 := #JOB_1_STEP_33)
      Contact( "Unit1.Em4.ControlNodes".sideTapeFixStage.sequence.status.seqActive )
      wire#w1
      I_Contact( "Unit1.Em4.ControlNodes".cm.softcam.sideTapeFixStageAxisC.pos03_tape4.inPos )
      Coil( "Unit1.Em4.ControlNodes".sideTapeFixStage."step".action1[133] )
   END_RUNG
   RUNG wire#w1
      Contact( "Unit1.Em4.ControlNodes".cm.softcam.sideTapeFixStageAxisC.pos03_tape4.inPos )
      Coil( "Unit1.Em4.ControlNodes".sideTapeFixStage."step".transition1[133] )
   END_RUNG
   RUNG wire#w1
      Contact( "Unit1.Em4.ControlNodes".sideTapeFixStage."step".transition1[133] )
      { S7_Templates := "time_type := Time" } #statTonTime[133].TON(pt := T#1000ms, et =>)
      Move(in := #JOB_1_STEP_40, out1 => "Unit1.Em4.ControlNodes".sideTapeFixStage.sequence.status.nextStep)
   END_RUNG
   // the same network as SCL:
   #_w1 := ("Unit1.Em4.ControlNodes".sideTapeFixStage.sequence.status.currentStep = #JOB_1_STEP_33) AND "Unit1.Em4.ControlNodes".sideTapeFixStage.sequence.status.seqActive;
   "Unit1.Em4.ControlNodes".sideTapeFixStage."step".action1[133] := #_w1 AND NOT "Unit1.Em4.ControlNodes".cm.softcam.sideTapeFixStageAxisC.pos03_tape4.inPos;
   "Unit1.Em4.ControlNodes".sideTapeFixStage."step".transition1[133] := #_w1 AND "Unit1.Em4.ControlNodes".cm.softcam.sideTapeFixStageAxisC.pos03_tape4.inPos;
   #statTonTime[133].TON(IN := #_w1 AND "Unit1.Em4.ControlNodes".sideTapeFixStage."step".transition1[133],
                         PT := T#1000ms);
   IF #statTonTime[133].Q THEN
       "Unit1.Em4.ControlNodes".sideTapeFixStage.sequence.status.nextStep := #JOB_1_STEP_40;
   END_IF;
END_REGION

REGION Network 16: Step[140] : Side Tape Fix Stage X-Axis Wait Pos
   RUNG wire#powerrail
      { S7_Templates := "SrcType := DInt" } EQ_Contact(in1 := "Unit1.Em4.ControlNodes".sideTapeFixStage.sequence.status.currentStep, in2 := #JOB_1_STEP_40)
      Contact( "Unit1.Em4.ControlNodes".sideTapeFixStage.sequence.status.seqActive )
      wire#w1
      I_Contact( "Unit1.Em4.ControlNodes".cm.softcam.sideTapeFixStageAxisX.pos00_wait.inPos )
      Coil( "Unit1.Em4.ControlNodes".sideTapeFixStage."step".action1[140] )
   END_RUNG
   RUNG wire#w1
      Contact( "Unit1.Em4.ControlNodes".cm.softcam.sideTapeFixStageAxisX.pos00_wait.inPos )
      Coil( "Unit1.Em4.ControlNodes".sideTapeFixStage."step".transition1[140] )
   END_RUNG
   RUNG wire#w1
      Contact( "Unit1.Em4.ControlNodes".sideTapeFixStage."step".transition1[140] )
      { S7_Templates := "time_type := Time" } #statTonTime[4].TON(pt := T#1000ms, et =>)
      Move(in := #JOB_1_STEP_90, out1 => "Unit1.Em4.ControlNodes".sideTapeFixStage.sequence.status.nextStep)
   END_RUNG
   // the same network as SCL:
   #_w1 := ("Unit1.Em4.ControlNodes".sideTapeFixStage.sequence.status.currentStep = #JOB_1_STEP_40) AND "Unit1.Em4.ControlNodes".sideTapeFixStage.sequence.status.seqActive;
   "Unit1.Em4.ControlNodes".sideTapeFixStage."step".action1[140] := #_w1 AND NOT "Unit1.Em4.ControlNodes".cm.softcam.sideTapeFixStageAxisX.pos00_wait.inPos;
   "Unit1.Em4.ControlNodes".sideTapeFixStage."step".transition1[140] := #_w1 AND "Unit1.Em4.ControlNodes".cm.softcam.sideTapeFixStageAxisX.pos00_wait.inPos;
   #statTonTime[4].TON(IN := #_w1 AND "Unit1.Em4.ControlNodes".sideTapeFixStage."step".transition1[140],
                       PT := T#1000ms);
   IF #statTonTime[4].Q THEN
       "Unit1.Em4.ControlNodes".sideTapeFixStage.sequence.status.nextStep := #JOB_1_STEP_90;
   END_IF;
END_REGION

REGION Network 17: Step[190] : JOB[1] Step End
   RUNG wire#powerrail
      { S7_Templates := "SrcType := DInt" } EQ_Contact(in1 := "Unit1.Em4.ControlNodes".sideTapeFixStage.sequence.status.currentStep, in2 := #JOB_1_STEP_90)
      Contact( "Unit1.Em4.ControlNodes".sideTapeFixStage.sequence.status.seqActive )
      wire#w1
      Coil( "Unit1.Em4.ControlNodes".sideTapeFixStage."step".action1[190] )
   END_RUNG
   RUNG wire#w1
      Coil( "Unit1.Em4.ControlNodes".sideTapeFixStage."step".transition1[190] )
   END_RUNG
   RUNG wire#w1
      Contact( "Unit1.Em4.ControlNodes".sideTapeFixStage."step".transition1[190] )
      { S7_Templates := "time_type := Time" } #statTonTime[190].TON(pt := T#100ms, et =>)
      Move(in := #STEP_IDLE, out1 => "Unit1.Em4.ControlNodes".sideTapeFixStage.sequence.status.nextStep)
   END_RUNG
   // the same network as SCL:
   "Unit1.Em4.ControlNodes".sideTapeFixStage."step".action1[190] := ("Unit1.Em4.ControlNodes".sideTapeFixStage.sequence.status.currentStep = #JOB_1_STEP_90) AND "Unit1.Em4.ControlNodes".sideTapeFixStage.sequence.status.seqActive;
   "Unit1.Em4.ControlNodes".sideTapeFixStage."step".transition1[190] := ("Unit1.Em4.ControlNodes".sideTapeFixStage.sequence.status.currentStep = #JOB_1_STEP_90) AND "Unit1.Em4.ControlNodes".sideTapeFixStage.sequence.status.seqActive;
   #statTonTime[190].TON(IN := ("Unit1.Em4.ControlNodes".sideTapeFixStage.sequence.status.currentStep = #JOB_1_STEP_90) AND "Unit1.Em4.ControlNodes".sideTapeFixStage.sequence.status.seqActive AND "Unit1.Em4.ControlNodes".sideTapeFixStage."step".transition1[190],
                         PT := T#100ms);
   IF #statTonTime[190].Q THEN
       "Unit1.Em4.ControlNodes".sideTapeFixStage.sequence.status.nextStep := #STEP_IDLE;
   END_IF;
END_REGION

REGION Network 18: *************** JOB[2] JR GET=AUTO *************************
END_REGION

REGION Network 19: Step[201] : JOB[2] Condition
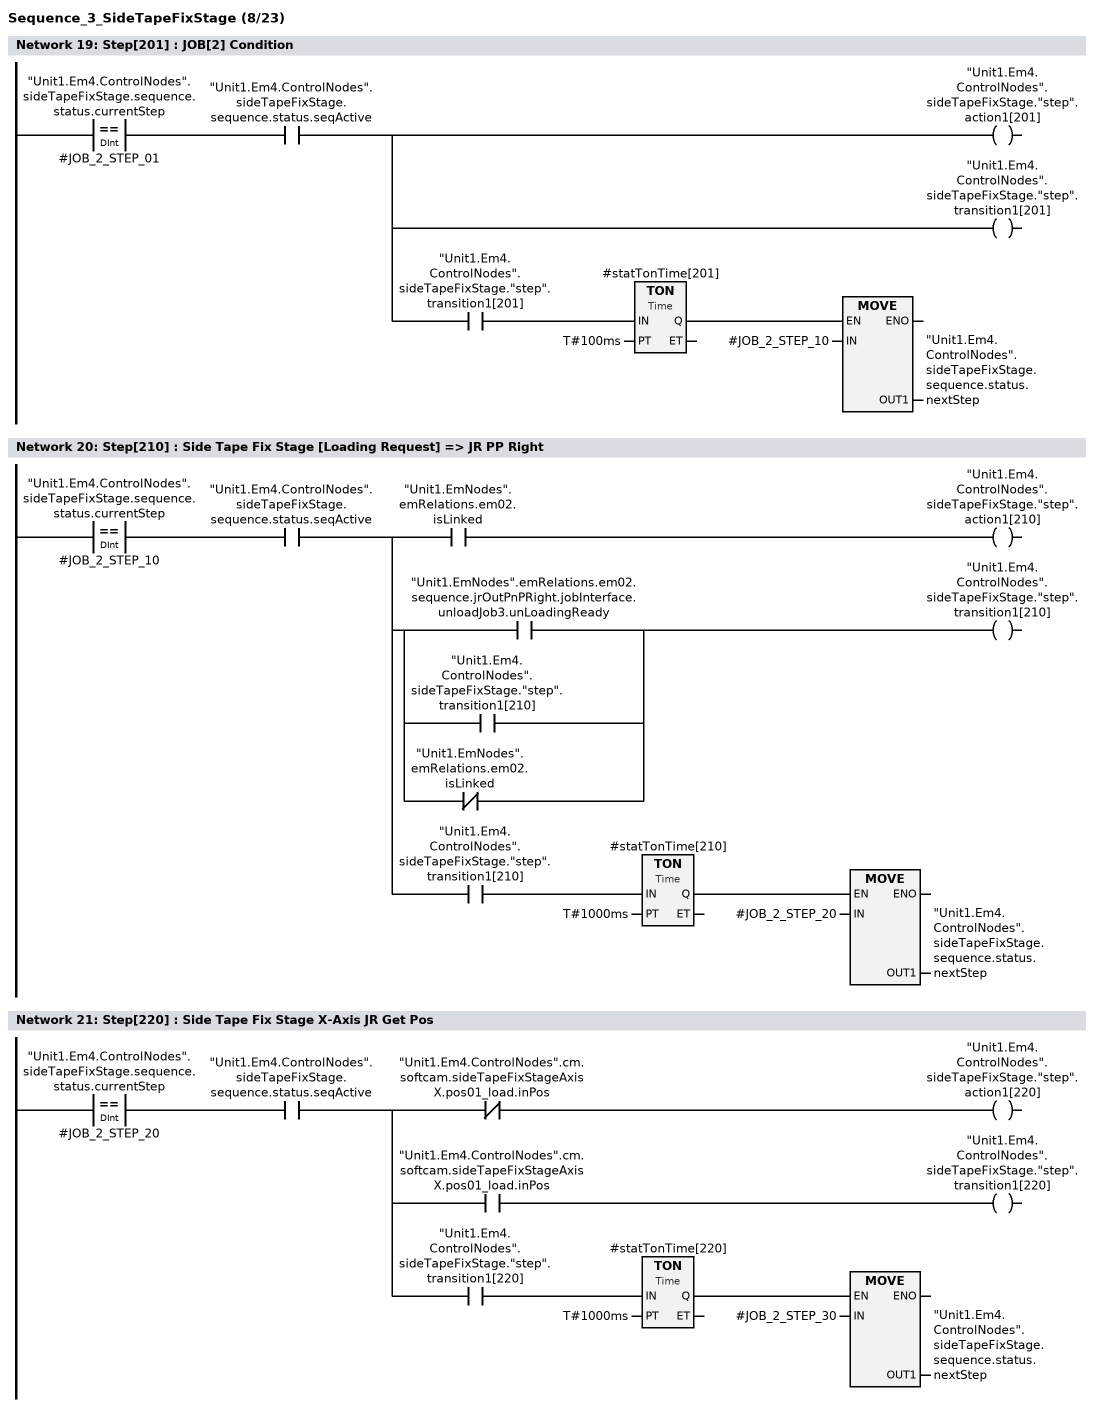
   RUNG wire#powerrail
      { S7_Templates := "SrcType := DInt" } EQ_Contact(in1 := "Unit1.Em4.ControlNodes".sideTapeFixStage.sequence.status.currentStep, in2 := #JOB_2_STEP_01)
      Contact( "Unit1.Em4.ControlNodes".sideTapeFixStage.sequence.status.seqActive )
      wire#w1
      Coil( "Unit1.Em4.ControlNodes".sideTapeFixStage."step".action1[201] )
   END_RUNG
   RUNG wire#w1
      Coil( "Unit1.Em4.ControlNodes".sideTapeFixStage."step".transition1[201] )
   END_RUNG
   RUNG wire#w1
      Contact( "Unit1.Em4.ControlNodes".sideTapeFixStage."step".transition1[201] )
      { S7_Templates := "time_type := Time" } #statTonTime[201].TON(pt := T#100ms, et =>)
      Move(in := #JOB_2_STEP_10, out1 => "Unit1.Em4.ControlNodes".sideTapeFixStage.sequence.status.nextStep)
   END_RUNG
   // the same network as SCL:
   "Unit1.Em4.ControlNodes".sideTapeFixStage."step".action1[201] := ("Unit1.Em4.ControlNodes".sideTapeFixStage.sequence.status.currentStep = #JOB_2_STEP_01) AND "Unit1.Em4.ControlNodes".sideTapeFixStage.sequence.status.seqActive;
   "Unit1.Em4.ControlNodes".sideTapeFixStage."step".transition1[201] := ("Unit1.Em4.ControlNodes".sideTapeFixStage.sequence.status.currentStep = #JOB_2_STEP_01) AND "Unit1.Em4.ControlNodes".sideTapeFixStage.sequence.status.seqActive;
   #statTonTime[201].TON(IN := ("Unit1.Em4.ControlNodes".sideTapeFixStage.sequence.status.currentStep = #JOB_2_STEP_01) AND "Unit1.Em4.ControlNodes".sideTapeFixStage.sequence.status.seqActive AND "Unit1.Em4.ControlNodes".sideTapeFixStage."step".transition1[201],
                         PT := T#100ms);
   IF #statTonTime[201].Q THEN
       "Unit1.Em4.ControlNodes".sideTapeFixStage.sequence.status.nextStep := #JOB_2_STEP_10;
   END_IF;
END_REGION

REGION Network 20: Step[210] : Side Tape Fix Stage [Loading Request] => JR PP Right
   RUNG wire#powerrail
      { S7_Templates := "SrcType := DInt" } EQ_Contact(in1 := "Unit1.Em4.ControlNodes".sideTapeFixStage.sequence.status.currentStep, in2 := #JOB_2_STEP_10)
      Contact( "Unit1.Em4.ControlNodes".sideTapeFixStage.sequence.status.seqActive )
      wire#w1
      Contact( "Unit1.EmNodes".emRelations.em02.isLinked )
      Coil( "Unit1.Em4.ControlNodes".sideTapeFixStage."step".action1[210] )
   END_RUNG
   RUNG wire#w1
      Contact( "Unit1.EmNodes".emRelations.em02.sequence.jrOutPnPRight.jobInterface.unloadJob3.unLoadingReady )
      wire#w2
      Coil( "Unit1.Em4.ControlNodes".sideTapeFixStage."step".transition1[210] )
   END_RUNG
   RUNG wire#w1
      Contact( "Unit1.Em4.ControlNodes".sideTapeFixStage."step".transition1[210] )
   END_RUNG wire#w2
   RUNG wire#w1
      I_Contact( "Unit1.EmNodes".emRelations.em02.isLinked )
   END_RUNG wire#w2
   RUNG wire#w1
      Contact( "Unit1.Em4.ControlNodes".sideTapeFixStage."step".transition1[210] )
      { S7_Templates := "time_type := Time" } #statTonTime[210].TON(pt := T#1000ms, et =>)
      Move(in := #JOB_2_STEP_20, out1 => "Unit1.Em4.ControlNodes".sideTapeFixStage.sequence.status.nextStep)
   END_RUNG
   // the same network as SCL:
   #_w1 := ("Unit1.Em4.ControlNodes".sideTapeFixStage.sequence.status.currentStep = #JOB_2_STEP_10) AND "Unit1.Em4.ControlNodes".sideTapeFixStage.sequence.status.seqActive;
   "Unit1.Em4.ControlNodes".sideTapeFixStage."step".action1[210] := #_w1 AND "Unit1.EmNodes".emRelations.em02.isLinked;
   "Unit1.Em4.ControlNodes".sideTapeFixStage."step".transition1[210] := #_w1 AND ("Unit1.EmNodes".emRelations.em02.sequence.jrOutPnPRight.jobInterface.unloadJob3.unLoadingReady OR "Unit1.Em4.ControlNodes".sideTapeFixStage."step".transition1[210] OR NOT "Unit1.EmNodes".emRelations.em02.isLinked);
   #statTonTime[210].TON(IN := #_w1 AND "Unit1.Em4.ControlNodes".sideTapeFixStage."step".transition1[210],
                         PT := T#1000ms);
   IF #statTonTime[210].Q THEN
       "Unit1.Em4.ControlNodes".sideTapeFixStage.sequence.status.nextStep := #JOB_2_STEP_20;
   END_IF;
END_REGION

REGION Network 21: Step[220] : Side Tape Fix Stage X-Axis JR Get Pos
   RUNG wire#powerrail
      { S7_Templates := "SrcType := DInt" } EQ_Contact(in1 := "Unit1.Em4.ControlNodes".sideTapeFixStage.sequence.status.currentStep, in2 := #JOB_2_STEP_20)
      Contact( "Unit1.Em4.ControlNodes".sideTapeFixStage.sequence.status.seqActive )
      wire#w1
      I_Contact( "Unit1.Em4.ControlNodes".cm.softcam.sideTapeFixStageAxisX.pos01_load.inPos )
      Coil( "Unit1.Em4.ControlNodes".sideTapeFixStage."step".action1[220] )
   END_RUNG
   RUNG wire#w1
      Contact( "Unit1.Em4.ControlNodes".cm.softcam.sideTapeFixStageAxisX.pos01_load.inPos )
      Coil( "Unit1.Em4.ControlNodes".sideTapeFixStage."step".transition1[220] )
   END_RUNG
   RUNG wire#w1
      Contact( "Unit1.Em4.ControlNodes".sideTapeFixStage."step".transition1[220] )
      { S7_Templates := "time_type := Time" } #statTonTime[220].TON(pt := T#1000ms, et =>)
      Move(in := #JOB_2_STEP_30, out1 => "Unit1.Em4.ControlNodes".sideTapeFixStage.sequence.status.nextStep)
   END_RUNG
   // the same network as SCL:
   #_w1 := ("Unit1.Em4.ControlNodes".sideTapeFixStage.sequence.status.currentStep = #JOB_2_STEP_20) AND "Unit1.Em4.ControlNodes".sideTapeFixStage.sequence.status.seqActive;
   "Unit1.Em4.ControlNodes".sideTapeFixStage."step".action1[220] := #_w1 AND NOT "Unit1.Em4.ControlNodes".cm.softcam.sideTapeFixStageAxisX.pos01_load.inPos;
   "Unit1.Em4.ControlNodes".sideTapeFixStage."step".transition1[220] := #_w1 AND "Unit1.Em4.ControlNodes".cm.softcam.sideTapeFixStageAxisX.pos01_load.inPos;
   #statTonTime[220].TON(IN := #_w1 AND "Unit1.Em4.ControlNodes".sideTapeFixStage."step".transition1[220],
                         PT := T#1000ms);
   IF #statTonTime[220].Q THEN
       "Unit1.Em4.ControlNodes".sideTapeFixStage.sequence.status.nextStep := #JOB_2_STEP_30;
   END_IF;
END_REGION

REGION Network 22: Step[230] : Side Tape Fix Stage Clamp Close
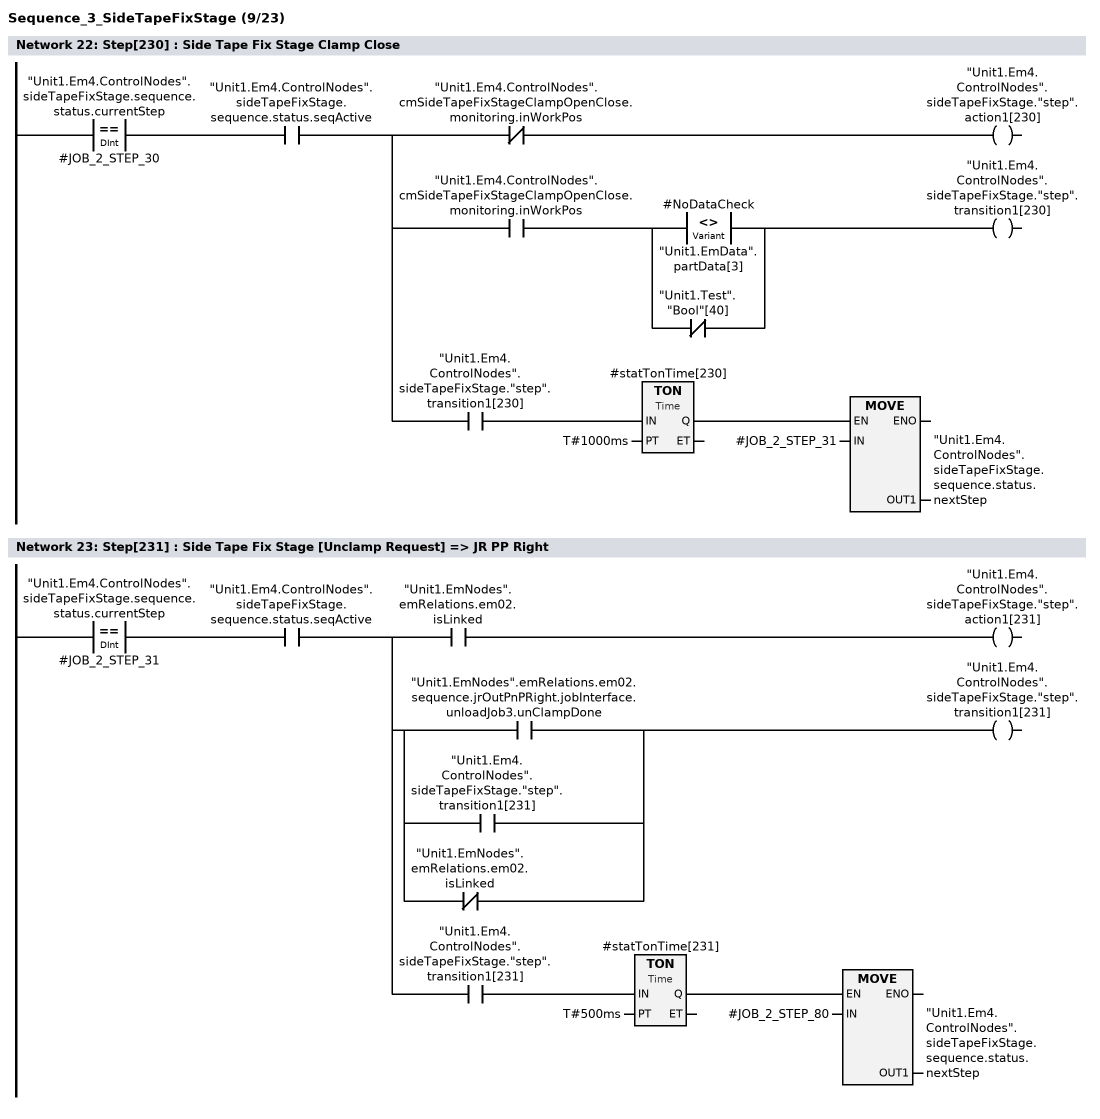
   RUNG wire#powerrail
      { S7_Templates := "SrcType := DInt" } EQ_Contact(in1 := "Unit1.Em4.ControlNodes".sideTapeFixStage.sequence.status.currentStep, in2 := #JOB_2_STEP_30)
      Contact( "Unit1.Em4.ControlNodes".sideTapeFixStage.sequence.status.seqActive )
      wire#w1
      I_Contact( "Unit1.Em4.ControlNodes".cmSideTapeFixStageClampOpenClose.monitoring.inWorkPos )
      Coil( "Unit1.Em4.ControlNodes".sideTapeFixStage."step".action1[230] )
   END_RUNG
   RUNG wire#w1
      Contact( "Unit1.Em4.ControlNodes".cmSideTapeFixStageClampOpenClose.monitoring.inWorkPos )
      wire#w2
      { S7_Templates := "SrcType := Variant" } NE_Contact(in1 := #NoDataCheck, in2 := "Unit1.EmData".partData[3])
      wire#w3
      Coil( "Unit1.Em4.ControlNodes".sideTapeFixStage."step".transition1[230] )
   END_RUNG
   RUNG wire#w2
      I_Contact( "Unit1.Test"."Bool"[40] )
   END_RUNG wire#w3
   RUNG wire#w1
      Contact( "Unit1.Em4.ControlNodes".sideTapeFixStage."step".transition1[230] )
      { S7_Templates := "time_type := Time" } #statTonTime[230].TON(pt := T#1000ms, et =>)
      Move(in := #JOB_2_STEP_31, out1 => "Unit1.Em4.ControlNodes".sideTapeFixStage.sequence.status.nextStep)
   END_RUNG
   // the same network as SCL:
   #_w1 := ("Unit1.Em4.ControlNodes".sideTapeFixStage.sequence.status.currentStep = #JOB_2_STEP_30) AND "Unit1.Em4.ControlNodes".sideTapeFixStage.sequence.status.seqActive;
   "Unit1.Em4.ControlNodes".sideTapeFixStage."step".action1[230] := #_w1 AND NOT "Unit1.Em4.ControlNodes".cmSideTapeFixStageClampOpenClose.monitoring.inWorkPos;
   "Unit1.Em4.ControlNodes".sideTapeFixStage."step".transition1[230] := #_w1 AND "Unit1.Em4.ControlNodes".cmSideTapeFixStageClampOpenClose.monitoring.inWorkPos AND ((#NoDataCheck <> "Unit1.EmData".partData[3]) OR NOT "Unit1.Test"."Bool"[40]);
   #statTonTime[230].TON(IN := #_w1 AND "Unit1.Em4.ControlNodes".sideTapeFixStage."step".transition1[230],
                         PT := T#1000ms);
   IF #statTonTime[230].Q THEN
       "Unit1.Em4.ControlNodes".sideTapeFixStage.sequence.status.nextStep := #JOB_2_STEP_31;
   END_IF;
END_REGION

REGION Network 23: Step[231] : Side Tape Fix Stage [Unclamp Request] => JR PP Right
   RUNG wire#powerrail
      { S7_Templates := "SrcType := DInt" } EQ_Contact(in1 := "Unit1.Em4.ControlNodes".sideTapeFixStage.sequence.status.currentStep, in2 := #JOB_2_STEP_31)
      Contact( "Unit1.Em4.ControlNodes".sideTapeFixStage.sequence.status.seqActive )
      wire#w1
      Contact( "Unit1.EmNodes".emRelations.em02.isLinked )
      Coil( "Unit1.Em4.ControlNodes".sideTapeFixStage."step".action1[231] )
   END_RUNG
   RUNG wire#w1
      Contact( "Unit1.EmNodes".emRelations.em02.sequence.jrOutPnPRight.jobInterface.unloadJob3.unClampDone )
      wire#w2
      Coil( "Unit1.Em4.ControlNodes".sideTapeFixStage."step".transition1[231] )
   END_RUNG
   RUNG wire#w1
      Contact( "Unit1.Em4.ControlNodes".sideTapeFixStage."step".transition1[231] )
   END_RUNG wire#w2
   RUNG wire#w1
      I_Contact( "Unit1.EmNodes".emRelations.em02.isLinked )
   END_RUNG wire#w2
   RUNG wire#w1
      Contact( "Unit1.Em4.ControlNodes".sideTapeFixStage."step".transition1[231] )
      { S7_Templates := "time_type := Time" } #statTonTime[231].TON(pt := T#500ms, et =>)
      Move(in := #JOB_2_STEP_80, out1 => "Unit1.Em4.ControlNodes".sideTapeFixStage.sequence.status.nextStep)
   END_RUNG
   // the same network as SCL:
   #_w1 := ("Unit1.Em4.ControlNodes".sideTapeFixStage.sequence.status.currentStep = #JOB_2_STEP_31) AND "Unit1.Em4.ControlNodes".sideTapeFixStage.sequence.status.seqActive;
   "Unit1.Em4.ControlNodes".sideTapeFixStage."step".action1[231] := #_w1 AND "Unit1.EmNodes".emRelations.em02.isLinked;
   "Unit1.Em4.ControlNodes".sideTapeFixStage."step".transition1[231] := #_w1 AND ("Unit1.EmNodes".emRelations.em02.sequence.jrOutPnPRight.jobInterface.unloadJob3.unClampDone OR "Unit1.Em4.ControlNodes".sideTapeFixStage."step".transition1[231] OR NOT "Unit1.EmNodes".emRelations.em02.isLinked);
   #statTonTime[231].TON(IN := #_w1 AND "Unit1.Em4.ControlNodes".sideTapeFixStage."step".transition1[231],
                         PT := T#500ms);
   IF #statTonTime[231].Q THEN
       "Unit1.Em4.ControlNodes".sideTapeFixStage.sequence.status.nextStep := #JOB_2_STEP_80;
   END_IF;
END_REGION

REGION Network 24: Step[280] : Side Tape Fix Stage X-Axis Wait Pos
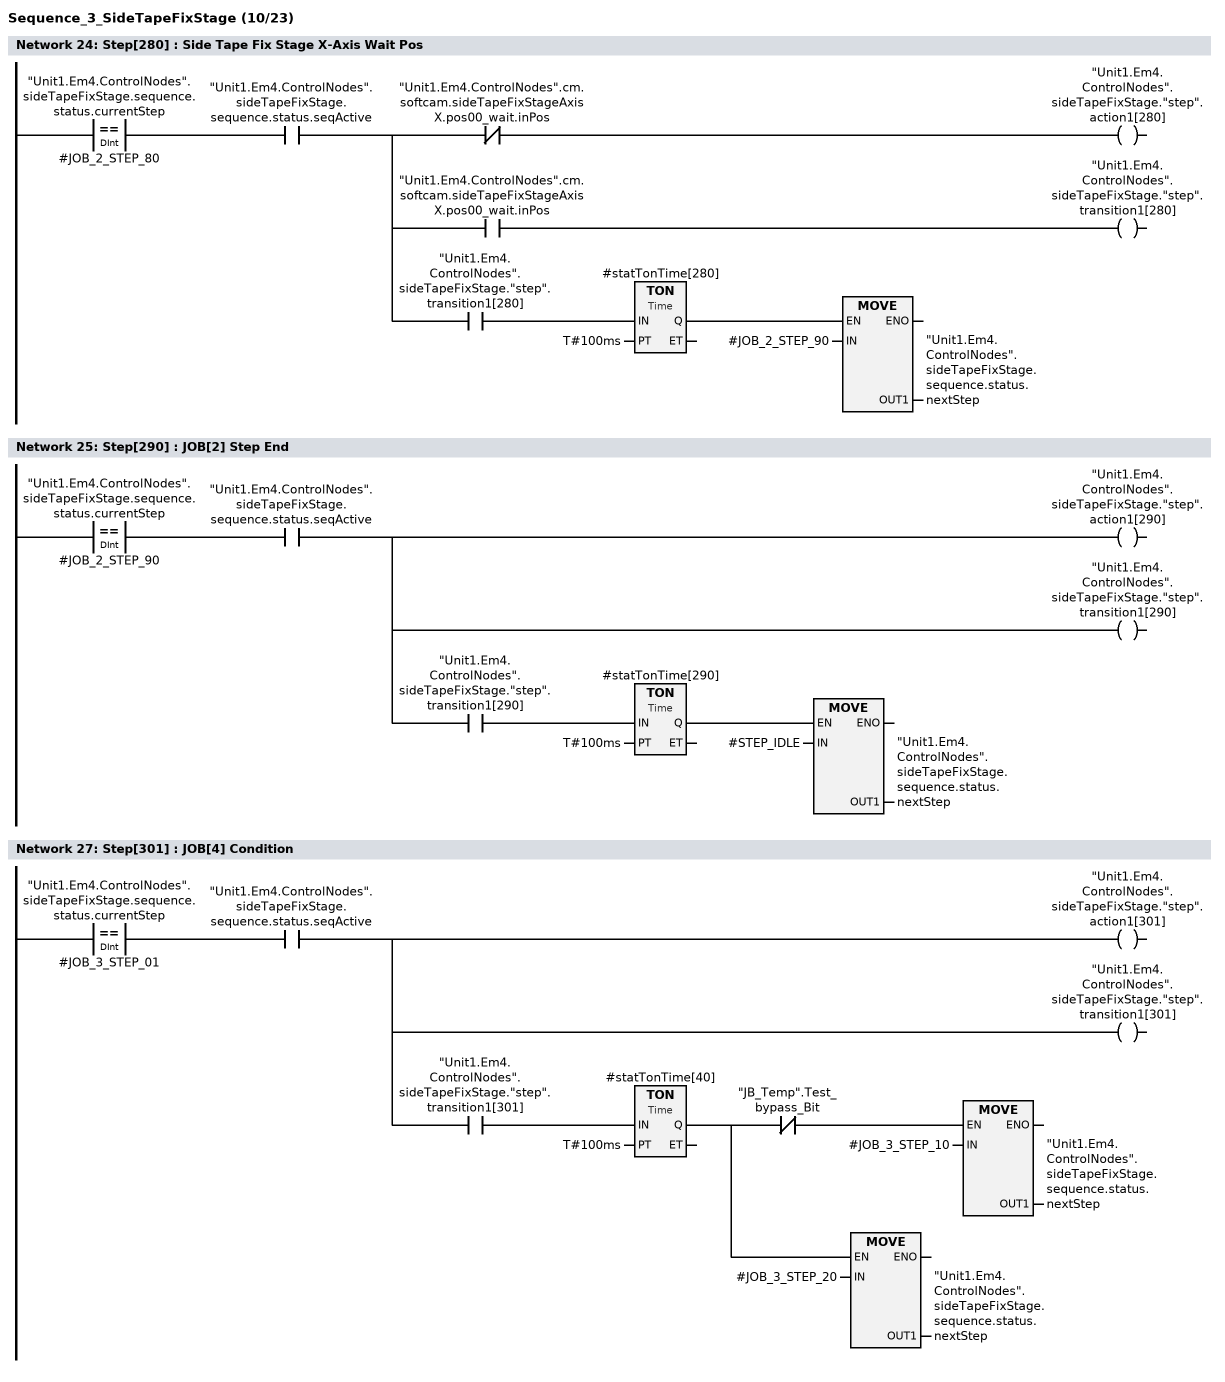
   RUNG wire#powerrail
      { S7_Templates := "SrcType := DInt" } EQ_Contact(in1 := "Unit1.Em4.ControlNodes".sideTapeFixStage.sequence.status.currentStep, in2 := #JOB_2_STEP_80)
      Contact( "Unit1.Em4.ControlNodes".sideTapeFixStage.sequence.status.seqActive )
      wire#w1
      I_Contact( "Unit1.Em4.ControlNodes".cm.softcam.sideTapeFixStageAxisX.pos00_wait.inPos )
      Coil( "Unit1.Em4.ControlNodes".sideTapeFixStage."step".action1[280] )
   END_RUNG
   RUNG wire#w1
      Contact( "Unit1.Em4.ControlNodes".cm.softcam.sideTapeFixStageAxisX.pos00_wait.inPos )
      Coil( "Unit1.Em4.ControlNodes".sideTapeFixStage."step".transition1[280] )
   END_RUNG
   RUNG wire#w1
      Contact( "Unit1.Em4.ControlNodes".sideTapeFixStage."step".transition1[280] )
      { S7_Templates := "time_type := Time" } #statTonTime[280].TON(pt := T#100ms, et =>)
      Move(in := #JOB_2_STEP_90, out1 => "Unit1.Em4.ControlNodes".sideTapeFixStage.sequence.status.nextStep)
   END_RUNG
   // the same network as SCL:
   #_w1 := ("Unit1.Em4.ControlNodes".sideTapeFixStage.sequence.status.currentStep = #JOB_2_STEP_80) AND "Unit1.Em4.ControlNodes".sideTapeFixStage.sequence.status.seqActive;
   "Unit1.Em4.ControlNodes".sideTapeFixStage."step".action1[280] := #_w1 AND NOT "Unit1.Em4.ControlNodes".cm.softcam.sideTapeFixStageAxisX.pos00_wait.inPos;
   "Unit1.Em4.ControlNodes".sideTapeFixStage."step".transition1[280] := #_w1 AND "Unit1.Em4.ControlNodes".cm.softcam.sideTapeFixStageAxisX.pos00_wait.inPos;
   #statTonTime[280].TON(IN := #_w1 AND "Unit1.Em4.ControlNodes".sideTapeFixStage."step".transition1[280],
                         PT := T#100ms);
   IF #statTonTime[280].Q THEN
       "Unit1.Em4.ControlNodes".sideTapeFixStage.sequence.status.nextStep := #JOB_2_STEP_90;
   END_IF;
END_REGION

REGION Network 25: Step[290] : JOB[2] Step End
   RUNG wire#powerrail
      { S7_Templates := "SrcType := DInt" } EQ_Contact(in1 := "Unit1.Em4.ControlNodes".sideTapeFixStage.sequence.status.currentStep, in2 := #JOB_2_STEP_90)
      Contact( "Unit1.Em4.ControlNodes".sideTapeFixStage.sequence.status.seqActive )
      wire#w1
      Coil( "Unit1.Em4.ControlNodes".sideTapeFixStage."step".action1[290] )
   END_RUNG
   RUNG wire#w1
      Coil( "Unit1.Em4.ControlNodes".sideTapeFixStage."step".transition1[290] )
   END_RUNG
   RUNG wire#w1
      Contact( "Unit1.Em4.ControlNodes".sideTapeFixStage."step".transition1[290] )
      { S7_Templates := "time_type := Time" } #statTonTime[290].TON(pt := T#100ms, et =>)
      Move(in := #STEP_IDLE, out1 => "Unit1.Em4.ControlNodes".sideTapeFixStage.sequence.status.nextStep)
   END_RUNG
   // the same network as SCL:
   "Unit1.Em4.ControlNodes".sideTapeFixStage."step".action1[290] := ("Unit1.Em4.ControlNodes".sideTapeFixStage.sequence.status.currentStep = #JOB_2_STEP_90) AND "Unit1.Em4.ControlNodes".sideTapeFixStage.sequence.status.seqActive;
   "Unit1.Em4.ControlNodes".sideTapeFixStage."step".transition1[290] := ("Unit1.Em4.ControlNodes".sideTapeFixStage.sequence.status.currentStep = #JOB_2_STEP_90) AND "Unit1.Em4.ControlNodes".sideTapeFixStage.sequence.status.seqActive;
   #statTonTime[290].TON(IN := ("Unit1.Em4.ControlNodes".sideTapeFixStage.sequence.status.currentStep = #JOB_2_STEP_90) AND "Unit1.Em4.ControlNodes".sideTapeFixStage.sequence.status.seqActive AND "Unit1.Em4.ControlNodes".sideTapeFixStage."step".transition1[290],
                         PT := T#100ms);
   IF #statTonTime[290].Q THEN
       "Unit1.Em4.ControlNodes".sideTapeFixStage.sequence.status.nextStep := #STEP_IDLE;
   END_IF;
END_REGION

REGION Network 26: *************** JOB[3] SIDE TAPING-1=AUTO *************************
END_REGION

REGION Network 27: Step[301] : JOB[4] Condition
   RUNG wire#powerrail
      { S7_Templates := "SrcType := DInt" } EQ_Contact(in1 := "Unit1.Em4.ControlNodes".sideTapeFixStage.sequence.status.currentStep, in2 := #JOB_3_STEP_01)
      Contact( "Unit1.Em4.ControlNodes".sideTapeFixStage.sequence.status.seqActive )
      wire#w1
      Coil( "Unit1.Em4.ControlNodes".sideTapeFixStage."step".action1[301] )
   END_RUNG
   RUNG wire#w1
      Coil( "Unit1.Em4.ControlNodes".sideTapeFixStage."step".transition1[301] )
   END_RUNG
   RUNG wire#w1
      Contact( "Unit1.Em4.ControlNodes".sideTapeFixStage."step".transition1[301] )
      { S7_Templates := "time_type := Time" } #statTonTime[40].TON(pt := T#100ms, et =>)
      wire#w2
      I_Contact( "JB_Temp".Test_bypass_Bit )
      Move(in := #JOB_3_STEP_10, out1 => "Unit1.Em4.ControlNodes".sideTapeFixStage.sequence.status.nextStep)
   END_RUNG
   RUNG wire#w2
      Move(in := #JOB_3_STEP_20, out1 => "Unit1.Em4.ControlNodes".sideTapeFixStage.sequence.status.nextStep)
   END_RUNG
   // the same network as SCL:
   "Unit1.Em4.ControlNodes".sideTapeFixStage."step".action1[301] := ("Unit1.Em4.ControlNodes".sideTapeFixStage.sequence.status.currentStep = #JOB_3_STEP_01) AND "Unit1.Em4.ControlNodes".sideTapeFixStage.sequence.status.seqActive;
   "Unit1.Em4.ControlNodes".sideTapeFixStage."step".transition1[301] := ("Unit1.Em4.ControlNodes".sideTapeFixStage.sequence.status.currentStep = #JOB_3_STEP_01) AND "Unit1.Em4.ControlNodes".sideTapeFixStage.sequence.status.seqActive;
   #statTonTime[40].TON(IN := ("Unit1.Em4.ControlNodes".sideTapeFixStage.sequence.status.currentStep = #JOB_3_STEP_01) AND "Unit1.Em4.ControlNodes".sideTapeFixStage.sequence.status.seqActive AND "Unit1.Em4.ControlNodes".sideTapeFixStage."step".transition1[301],
                        PT := T#100ms);
   IF #statTonTime[40].Q AND NOT "JB_Temp".Test_bypass_Bit THEN
       "Unit1.Em4.ControlNodes".sideTapeFixStage.sequence.status.nextStep := #JOB_3_STEP_10;
   END_IF;
   IF #statTonTime[40].Q THEN
       "Unit1.Em4.ControlNodes".sideTapeFixStage.sequence.status.nextStep := #JOB_3_STEP_20;
   END_IF;
END_REGION

REGION Network 28: Step[310] : Spare
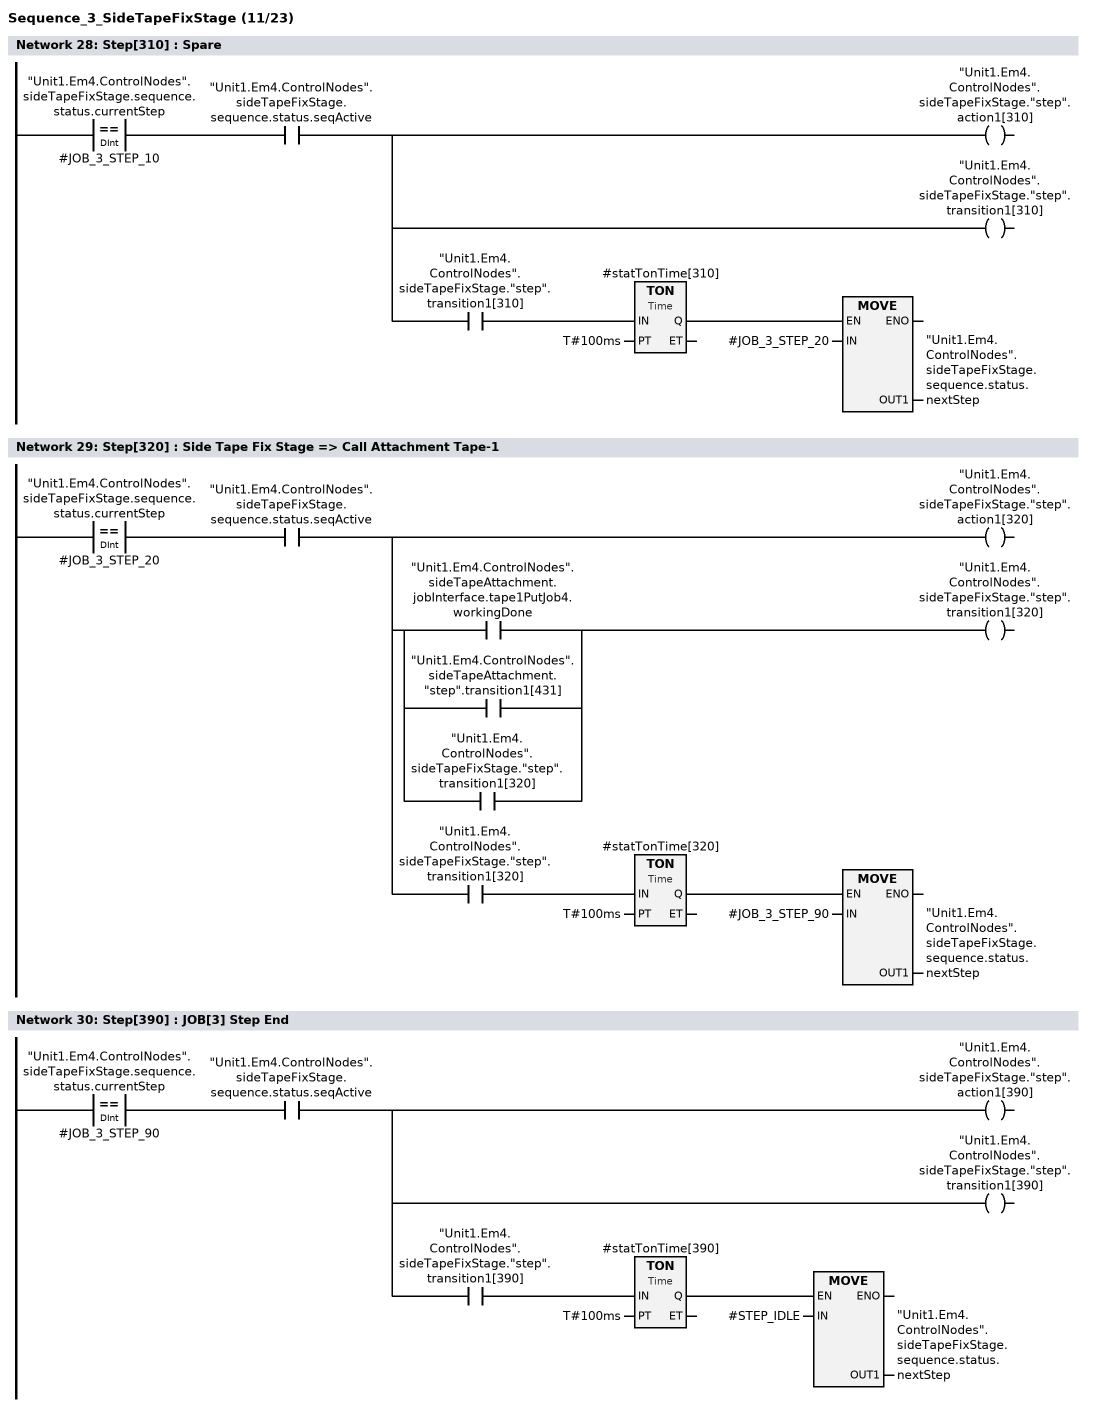
   RUNG wire#powerrail
      { S7_Templates := "SrcType := DInt" } EQ_Contact(in1 := "Unit1.Em4.ControlNodes".sideTapeFixStage.sequence.status.currentStep, in2 := #JOB_3_STEP_10)
      Contact( "Unit1.Em4.ControlNodes".sideTapeFixStage.sequence.status.seqActive )
      wire#w1
      Coil( "Unit1.Em4.ControlNodes".sideTapeFixStage."step".action1[310] )
   END_RUNG
   RUNG wire#w1
      Coil( "Unit1.Em4.ControlNodes".sideTapeFixStage."step".transition1[310] )
   END_RUNG
   RUNG wire#w1
      Contact( "Unit1.Em4.ControlNodes".sideTapeFixStage."step".transition1[310] )
      { S7_Templates := "time_type := Time" } #statTonTime[310].TON(pt := T#100ms, et =>)
      Move(in := #JOB_3_STEP_20, out1 => "Unit1.Em4.ControlNodes".sideTapeFixStage.sequence.status.nextStep)
   END_RUNG
   // the same network as SCL:
   "Unit1.Em4.ControlNodes".sideTapeFixStage."step".action1[310] := ("Unit1.Em4.ControlNodes".sideTapeFixStage.sequence.status.currentStep = #JOB_3_STEP_10) AND "Unit1.Em4.ControlNodes".sideTapeFixStage.sequence.status.seqActive;
   "Unit1.Em4.ControlNodes".sideTapeFixStage."step".transition1[310] := ("Unit1.Em4.ControlNodes".sideTapeFixStage.sequence.status.currentStep = #JOB_3_STEP_10) AND "Unit1.Em4.ControlNodes".sideTapeFixStage.sequence.status.seqActive;
   #statTonTime[310].TON(IN := ("Unit1.Em4.ControlNodes".sideTapeFixStage.sequence.status.currentStep = #JOB_3_STEP_10) AND "Unit1.Em4.ControlNodes".sideTapeFixStage.sequence.status.seqActive AND "Unit1.Em4.ControlNodes".sideTapeFixStage."step".transition1[310],
                         PT := T#100ms);
   IF #statTonTime[310].Q THEN
       "Unit1.Em4.ControlNodes".sideTapeFixStage.sequence.status.nextStep := #JOB_3_STEP_20;
   END_IF;
END_REGION

REGION Network 29: Step[320] : Side Tape Fix Stage => Call Attachment Tape-1
   RUNG wire#powerrail
      { S7_Templates := "SrcType := DInt" } EQ_Contact(in1 := "Unit1.Em4.ControlNodes".sideTapeFixStage.sequence.status.currentStep, in2 := #JOB_3_STEP_20)
      Contact( "Unit1.Em4.ControlNodes".sideTapeFixStage.sequence.status.seqActive )
      wire#w1
      Coil( "Unit1.Em4.ControlNodes".sideTapeFixStage."step".action1[320] )
   END_RUNG
   RUNG wire#w1
      Contact( "Unit1.Em4.ControlNodes".sideTapeAttachment.jobInterface.tape1PutJob4.workingDone )
      wire#w2
      Coil( "Unit1.Em4.ControlNodes".sideTapeFixStage."step".transition1[320] )
   END_RUNG
   RUNG wire#w1
      Contact( "Unit1.Em4.ControlNodes".sideTapeAttachment."step".transition1[431] )
   END_RUNG wire#w2
   RUNG wire#w1
      Contact( "Unit1.Em4.ControlNodes".sideTapeFixStage."step".transition1[320] )
   END_RUNG wire#w2
   RUNG wire#w1
      Contact( "Unit1.Em4.ControlNodes".sideTapeFixStage."step".transition1[320] )
      { S7_Templates := "time_type := Time" } #statTonTime[320].TON(pt := T#100ms, et =>)
      Move(in := #JOB_3_STEP_90, out1 => "Unit1.Em4.ControlNodes".sideTapeFixStage.sequence.status.nextStep)
   END_RUNG
   // the same network as SCL:
   "Unit1.Em4.ControlNodes".sideTapeFixStage."step".action1[320] := ("Unit1.Em4.ControlNodes".sideTapeFixStage.sequence.status.currentStep = #JOB_3_STEP_20) AND "Unit1.Em4.ControlNodes".sideTapeFixStage.sequence.status.seqActive;
   "Unit1.Em4.ControlNodes".sideTapeFixStage."step".transition1[320] := ("Unit1.Em4.ControlNodes".sideTapeFixStage.sequence.status.currentStep = #JOB_3_STEP_20) AND "Unit1.Em4.ControlNodes".sideTapeFixStage.sequence.status.seqActive AND ("Unit1.Em4.ControlNodes".sideTapeAttachment.jobInterface.tape1PutJob4.workingDone OR "Unit1.Em4.ControlNodes".sideTapeAttachment."step".transition1[431] OR "Unit1.Em4.ControlNodes".sideTapeFixStage."step".transition1[320]);
   #statTonTime[320].TON(IN := ("Unit1.Em4.ControlNodes".sideTapeFixStage.sequence.status.currentStep = #JOB_3_STEP_20) AND "Unit1.Em4.ControlNodes".sideTapeFixStage.sequence.status.seqActive AND "Unit1.Em4.ControlNodes".sideTapeFixStage."step".transition1[320],
                         PT := T#100ms);
   IF #statTonTime[320].Q THEN
       "Unit1.Em4.ControlNodes".sideTapeFixStage.sequence.status.nextStep := #JOB_3_STEP_90;
   END_IF;
END_REGION

REGION Network 30: Step[390] : JOB[3] Step End
   RUNG wire#powerrail
      { S7_Templates := "SrcType := DInt" } EQ_Contact(in1 := "Unit1.Em4.ControlNodes".sideTapeFixStage.sequence.status.currentStep, in2 := #JOB_3_STEP_90)
      Contact( "Unit1.Em4.ControlNodes".sideTapeFixStage.sequence.status.seqActive )
      wire#w1
      Coil( "Unit1.Em4.ControlNodes".sideTapeFixStage."step".action1[390] )
   END_RUNG
   RUNG wire#w1
      Coil( "Unit1.Em4.ControlNodes".sideTapeFixStage."step".transition1[390] )
   END_RUNG
   RUNG wire#w1
      Contact( "Unit1.Em4.ControlNodes".sideTapeFixStage."step".transition1[390] )
      { S7_Templates := "time_type := Time" } #statTonTime[390].TON(pt := T#100ms, et =>)
      Move(in := #STEP_IDLE, out1 => "Unit1.Em4.ControlNodes".sideTapeFixStage.sequence.status.nextStep)
   END_RUNG
   // the same network as SCL:
   "Unit1.Em4.ControlNodes".sideTapeFixStage."step".action1[390] := ("Unit1.Em4.ControlNodes".sideTapeFixStage.sequence.status.currentStep = #JOB_3_STEP_90) AND "Unit1.Em4.ControlNodes".sideTapeFixStage.sequence.status.seqActive;
   "Unit1.Em4.ControlNodes".sideTapeFixStage."step".transition1[390] := ("Unit1.Em4.ControlNodes".sideTapeFixStage.sequence.status.currentStep = #JOB_3_STEP_90) AND "Unit1.Em4.ControlNodes".sideTapeFixStage.sequence.status.seqActive;
   #statTonTime[390].TON(IN := ("Unit1.Em4.ControlNodes".sideTapeFixStage.sequence.status.currentStep = #JOB_3_STEP_90) AND "Unit1.Em4.ControlNodes".sideTapeFixStage.sequence.status.seqActive AND "Unit1.Em4.ControlNodes".sideTapeFixStage."step".transition1[390],
                         PT := T#100ms);
   IF #statTonTime[390].Q THEN
       "Unit1.Em4.ControlNodes".sideTapeFixStage.sequence.status.nextStep := #STEP_IDLE;
   END_IF;
END_REGION

REGION Network 31: *************** JOB[4] SIDE TAPING-2=AUTO *************************
END_REGION

REGION Network 32: Step[401] : JOB[4] Condition
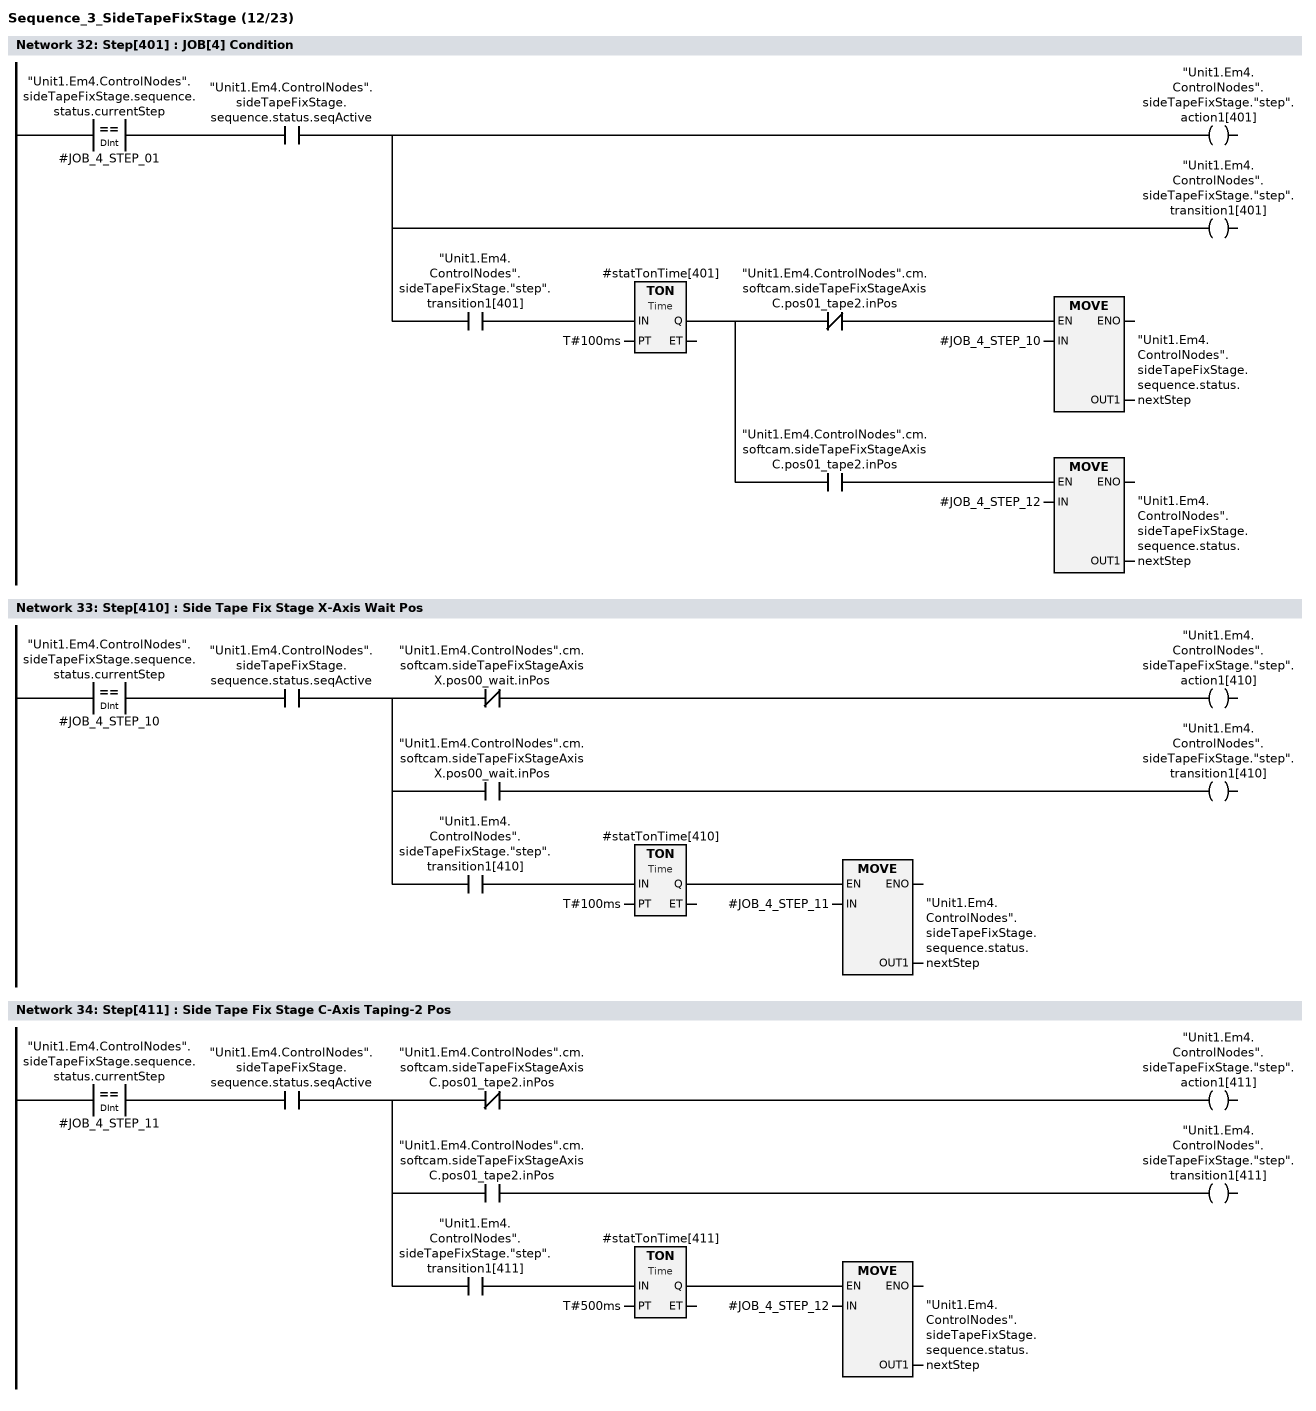
   RUNG wire#powerrail
      { S7_Templates := "SrcType := DInt" } EQ_Contact(in1 := "Unit1.Em4.ControlNodes".sideTapeFixStage.sequence.status.currentStep, in2 := #JOB_4_STEP_01)
      Contact( "Unit1.Em4.ControlNodes".sideTapeFixStage.sequence.status.seqActive )
      wire#w1
      Coil( "Unit1.Em4.ControlNodes".sideTapeFixStage."step".action1[401] )
   END_RUNG
   RUNG wire#w1
      Coil( "Unit1.Em4.ControlNodes".sideTapeFixStage."step".transition1[401] )
   END_RUNG
   RUNG wire#w1
      Contact( "Unit1.Em4.ControlNodes".sideTapeFixStage."step".transition1[401] )
      { S7_Templates := "time_type := Time" } #statTonTime[401].TON(pt := T#100ms, et =>)
      wire#w2
      I_Contact( "Unit1.Em4.ControlNodes".cm.softcam.sideTapeFixStageAxisC.pos01_tape2.inPos )
      Move(in := #JOB_4_STEP_10, out1 => "Unit1.Em4.ControlNodes".sideTapeFixStage.sequence.status.nextStep)
   END_RUNG
   RUNG wire#w2
      Contact( "Unit1.Em4.ControlNodes".cm.softcam.sideTapeFixStageAxisC.pos01_tape2.inPos )
      Move(in := #JOB_4_STEP_12, out1 => "Unit1.Em4.ControlNodes".sideTapeFixStage.sequence.status.nextStep)
   END_RUNG
   // the same network as SCL:
   "Unit1.Em4.ControlNodes".sideTapeFixStage."step".action1[401] := ("Unit1.Em4.ControlNodes".sideTapeFixStage.sequence.status.currentStep = #JOB_4_STEP_01) AND "Unit1.Em4.ControlNodes".sideTapeFixStage.sequence.status.seqActive;
   "Unit1.Em4.ControlNodes".sideTapeFixStage."step".transition1[401] := ("Unit1.Em4.ControlNodes".sideTapeFixStage.sequence.status.currentStep = #JOB_4_STEP_01) AND "Unit1.Em4.ControlNodes".sideTapeFixStage.sequence.status.seqActive;
   #statTonTime[401].TON(IN := ("Unit1.Em4.ControlNodes".sideTapeFixStage.sequence.status.currentStep = #JOB_4_STEP_01) AND "Unit1.Em4.ControlNodes".sideTapeFixStage.sequence.status.seqActive AND "Unit1.Em4.ControlNodes".sideTapeFixStage."step".transition1[401],
                         PT := T#100ms);
   IF #statTonTime[401].Q AND NOT "Unit1.Em4.ControlNodes".cm.softcam.sideTapeFixStageAxisC.pos01_tape2.inPos THEN
       "Unit1.Em4.ControlNodes".sideTapeFixStage.sequence.status.nextStep := #JOB_4_STEP_10;
   END_IF;
   IF #statTonTime[401].Q AND "Unit1.Em4.ControlNodes".cm.softcam.sideTapeFixStageAxisC.pos01_tape2.inPos THEN
       "Unit1.Em4.ControlNodes".sideTapeFixStage.sequence.status.nextStep := #JOB_4_STEP_12;
   END_IF;
END_REGION

REGION Network 33: Step[410] : Side Tape Fix Stage X-Axis Wait Pos
   RUNG wire#powerrail
      { S7_Templates := "SrcType := DInt" } EQ_Contact(in1 := "Unit1.Em4.ControlNodes".sideTapeFixStage.sequence.status.currentStep, in2 := #JOB_4_STEP_10)
      Contact( "Unit1.Em4.ControlNodes".sideTapeFixStage.sequence.status.seqActive )
      wire#w1
      I_Contact( "Unit1.Em4.ControlNodes".cm.softcam.sideTapeFixStageAxisX.pos00_wait.inPos )
      Coil( "Unit1.Em4.ControlNodes".sideTapeFixStage."step".action1[410] )
   END_RUNG
   RUNG wire#w1
      Contact( "Unit1.Em4.ControlNodes".cm.softcam.sideTapeFixStageAxisX.pos00_wait.inPos )
      Coil( "Unit1.Em4.ControlNodes".sideTapeFixStage."step".transition1[410] )
   END_RUNG
   RUNG wire#w1
      Contact( "Unit1.Em4.ControlNodes".sideTapeFixStage."step".transition1[410] )
      { S7_Templates := "time_type := Time" } #statTonTime[410].TON(pt := T#100ms, et =>)
      Move(in := #JOB_4_STEP_11, out1 => "Unit1.Em4.ControlNodes".sideTapeFixStage.sequence.status.nextStep)
   END_RUNG
   // the same network as SCL:
   #_w1 := ("Unit1.Em4.ControlNodes".sideTapeFixStage.sequence.status.currentStep = #JOB_4_STEP_10) AND "Unit1.Em4.ControlNodes".sideTapeFixStage.sequence.status.seqActive;
   "Unit1.Em4.ControlNodes".sideTapeFixStage."step".action1[410] := #_w1 AND NOT "Unit1.Em4.ControlNodes".cm.softcam.sideTapeFixStageAxisX.pos00_wait.inPos;
   "Unit1.Em4.ControlNodes".sideTapeFixStage."step".transition1[410] := #_w1 AND "Unit1.Em4.ControlNodes".cm.softcam.sideTapeFixStageAxisX.pos00_wait.inPos;
   #statTonTime[410].TON(IN := #_w1 AND "Unit1.Em4.ControlNodes".sideTapeFixStage."step".transition1[410],
                         PT := T#100ms);
   IF #statTonTime[410].Q THEN
       "Unit1.Em4.ControlNodes".sideTapeFixStage.sequence.status.nextStep := #JOB_4_STEP_11;
   END_IF;
END_REGION

REGION Network 34: Step[411] : Side Tape Fix Stage C-Axis Taping-2 Pos
   RUNG wire#powerrail
      { S7_Templates := "SrcType := DInt" } EQ_Contact(in1 := "Unit1.Em4.ControlNodes".sideTapeFixStage.sequence.status.currentStep, in2 := #JOB_4_STEP_11)
      Contact( "Unit1.Em4.ControlNodes".sideTapeFixStage.sequence.status.seqActive )
      wire#w1
      I_Contact( "Unit1.Em4.ControlNodes".cm.softcam.sideTapeFixStageAxisC.pos01_tape2.inPos )
      Coil( "Unit1.Em4.ControlNodes".sideTapeFixStage."step".action1[411] )
   END_RUNG
   RUNG wire#w1
      Contact( "Unit1.Em4.ControlNodes".cm.softcam.sideTapeFixStageAxisC.pos01_tape2.inPos )
      Coil( "Unit1.Em4.ControlNodes".sideTapeFixStage."step".transition1[411] )
   END_RUNG
   RUNG wire#w1
      Contact( "Unit1.Em4.ControlNodes".sideTapeFixStage."step".transition1[411] )
      { S7_Templates := "time_type := Time" } #statTonTime[411].TON(pt := T#500ms, et =>)
      Move(in := #JOB_4_STEP_12, out1 => "Unit1.Em4.ControlNodes".sideTapeFixStage.sequence.status.nextStep)
   END_RUNG
   // the same network as SCL:
   #_w1 := ("Unit1.Em4.ControlNodes".sideTapeFixStage.sequence.status.currentStep = #JOB_4_STEP_11) AND "Unit1.Em4.ControlNodes".sideTapeFixStage.sequence.status.seqActive;
   "Unit1.Em4.ControlNodes".sideTapeFixStage."step".action1[411] := #_w1 AND NOT "Unit1.Em4.ControlNodes".cm.softcam.sideTapeFixStageAxisC.pos01_tape2.inPos;
   "Unit1.Em4.ControlNodes".sideTapeFixStage."step".transition1[411] := #_w1 AND "Unit1.Em4.ControlNodes".cm.softcam.sideTapeFixStageAxisC.pos01_tape2.inPos;
   #statTonTime[411].TON(IN := #_w1 AND "Unit1.Em4.ControlNodes".sideTapeFixStage."step".transition1[411],
                         PT := T#500ms);
   IF #statTonTime[411].Q THEN
       "Unit1.Em4.ControlNodes".sideTapeFixStage.sequence.status.nextStep := #JOB_4_STEP_12;
   END_IF;
END_REGION

REGION Network 35: Step[412] : Side Tape Fix Stage X-Axis Wait Pos
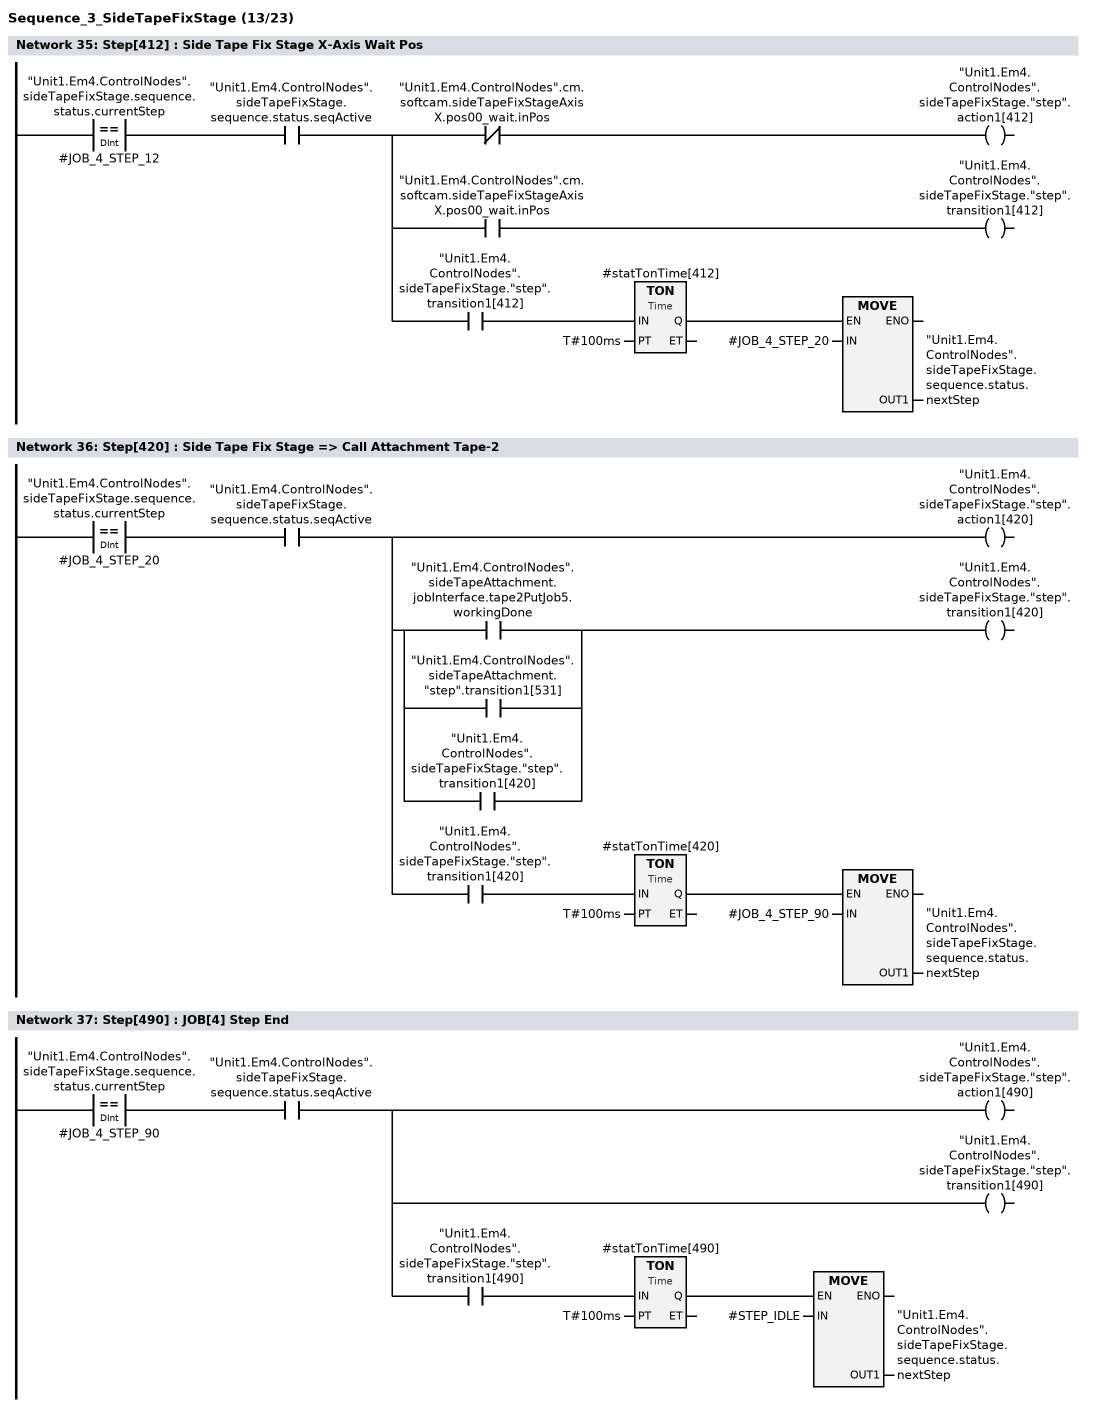
   RUNG wire#powerrail
      { S7_Templates := "SrcType := DInt" } EQ_Contact(in1 := "Unit1.Em4.ControlNodes".sideTapeFixStage.sequence.status.currentStep, in2 := #JOB_4_STEP_12)
      Contact( "Unit1.Em4.ControlNodes".sideTapeFixStage.sequence.status.seqActive )
      wire#w1
      I_Contact( "Unit1.Em4.ControlNodes".cm.softcam.sideTapeFixStageAxisX.pos00_wait.inPos )
      Coil( "Unit1.Em4.ControlNodes".sideTapeFixStage."step".action1[412] )
   END_RUNG
   RUNG wire#w1
      Contact( "Unit1.Em4.ControlNodes".cm.softcam.sideTapeFixStageAxisX.pos00_wait.inPos )
      Coil( "Unit1.Em4.ControlNodes".sideTapeFixStage."step".transition1[412] )
   END_RUNG
   RUNG wire#w1
      Contact( "Unit1.Em4.ControlNodes".sideTapeFixStage."step".transition1[412] )
      { S7_Templates := "time_type := Time" } #statTonTime[412].TON(pt := T#100ms, et =>)
      Move(in := #JOB_4_STEP_20, out1 => "Unit1.Em4.ControlNodes".sideTapeFixStage.sequence.status.nextStep)
   END_RUNG
   // the same network as SCL:
   #_w1 := ("Unit1.Em4.ControlNodes".sideTapeFixStage.sequence.status.currentStep = #JOB_4_STEP_12) AND "Unit1.Em4.ControlNodes".sideTapeFixStage.sequence.status.seqActive;
   "Unit1.Em4.ControlNodes".sideTapeFixStage."step".action1[412] := #_w1 AND NOT "Unit1.Em4.ControlNodes".cm.softcam.sideTapeFixStageAxisX.pos00_wait.inPos;
   "Unit1.Em4.ControlNodes".sideTapeFixStage."step".transition1[412] := #_w1 AND "Unit1.Em4.ControlNodes".cm.softcam.sideTapeFixStageAxisX.pos00_wait.inPos;
   #statTonTime[412].TON(IN := #_w1 AND "Unit1.Em4.ControlNodes".sideTapeFixStage."step".transition1[412],
                         PT := T#100ms);
   IF #statTonTime[412].Q THEN
       "Unit1.Em4.ControlNodes".sideTapeFixStage.sequence.status.nextStep := #JOB_4_STEP_20;
   END_IF;
END_REGION

REGION Network 36: Step[420] : Side Tape Fix Stage => Call Attachment Tape-2
   RUNG wire#powerrail
      { S7_Templates := "SrcType := DInt" } EQ_Contact(in1 := "Unit1.Em4.ControlNodes".sideTapeFixStage.sequence.status.currentStep, in2 := #JOB_4_STEP_20)
      Contact( "Unit1.Em4.ControlNodes".sideTapeFixStage.sequence.status.seqActive )
      wire#w1
      Coil( "Unit1.Em4.ControlNodes".sideTapeFixStage."step".action1[420] )
   END_RUNG
   RUNG wire#w1
      Contact( "Unit1.Em4.ControlNodes".sideTapeAttachment.jobInterface.tape2PutJob5.workingDone )
      wire#w2
      Coil( "Unit1.Em4.ControlNodes".sideTapeFixStage."step".transition1[420] )
   END_RUNG
   RUNG wire#w1
      Contact( "Unit1.Em4.ControlNodes".sideTapeAttachment."step".transition1[531] )
   END_RUNG wire#w2
   RUNG wire#w1
      Contact( "Unit1.Em4.ControlNodes".sideTapeFixStage."step".transition1[420] )
   END_RUNG wire#w2
   RUNG wire#w1
      Contact( "Unit1.Em4.ControlNodes".sideTapeFixStage."step".transition1[420] )
      { S7_Templates := "time_type := Time" } #statTonTime[420].TON(pt := T#100ms, et =>)
      Move(in := #JOB_4_STEP_90, out1 => "Unit1.Em4.ControlNodes".sideTapeFixStage.sequence.status.nextStep)
   END_RUNG
   // the same network as SCL:
   "Unit1.Em4.ControlNodes".sideTapeFixStage."step".action1[420] := ("Unit1.Em4.ControlNodes".sideTapeFixStage.sequence.status.currentStep = #JOB_4_STEP_20) AND "Unit1.Em4.ControlNodes".sideTapeFixStage.sequence.status.seqActive;
   "Unit1.Em4.ControlNodes".sideTapeFixStage."step".transition1[420] := ("Unit1.Em4.ControlNodes".sideTapeFixStage.sequence.status.currentStep = #JOB_4_STEP_20) AND "Unit1.Em4.ControlNodes".sideTapeFixStage.sequence.status.seqActive AND ("Unit1.Em4.ControlNodes".sideTapeAttachment.jobInterface.tape2PutJob5.workingDone OR "Unit1.Em4.ControlNodes".sideTapeAttachment."step".transition1[531] OR "Unit1.Em4.ControlNodes".sideTapeFixStage."step".transition1[420]);
   #statTonTime[420].TON(IN := ("Unit1.Em4.ControlNodes".sideTapeFixStage.sequence.status.currentStep = #JOB_4_STEP_20) AND "Unit1.Em4.ControlNodes".sideTapeFixStage.sequence.status.seqActive AND "Unit1.Em4.ControlNodes".sideTapeFixStage."step".transition1[420],
                         PT := T#100ms);
   IF #statTonTime[420].Q THEN
       "Unit1.Em4.ControlNodes".sideTapeFixStage.sequence.status.nextStep := #JOB_4_STEP_90;
   END_IF;
END_REGION

REGION Network 37: Step[490] : JOB[4] Step End
   RUNG wire#powerrail
      { S7_Templates := "SrcType := DInt" } EQ_Contact(in1 := "Unit1.Em4.ControlNodes".sideTapeFixStage.sequence.status.currentStep, in2 := #JOB_4_STEP_90)
      Contact( "Unit1.Em4.ControlNodes".sideTapeFixStage.sequence.status.seqActive )
      wire#w1
      Coil( "Unit1.Em4.ControlNodes".sideTapeFixStage."step".action1[490] )
   END_RUNG
   RUNG wire#w1
      Coil( "Unit1.Em4.ControlNodes".sideTapeFixStage."step".transition1[490] )
   END_RUNG
   RUNG wire#w1
      Contact( "Unit1.Em4.ControlNodes".sideTapeFixStage."step".transition1[490] )
      { S7_Templates := "time_type := Time" } #statTonTime[490].TON(pt := T#100ms, et =>)
      Move(in := #STEP_IDLE, out1 => "Unit1.Em4.ControlNodes".sideTapeFixStage.sequence.status.nextStep)
   END_RUNG
   // the same network as SCL:
   "Unit1.Em4.ControlNodes".sideTapeFixStage."step".action1[490] := ("Unit1.Em4.ControlNodes".sideTapeFixStage.sequence.status.currentStep = #JOB_4_STEP_90) AND "Unit1.Em4.ControlNodes".sideTapeFixStage.sequence.status.seqActive;
   "Unit1.Em4.ControlNodes".sideTapeFixStage."step".transition1[490] := ("Unit1.Em4.ControlNodes".sideTapeFixStage.sequence.status.currentStep = #JOB_4_STEP_90) AND "Unit1.Em4.ControlNodes".sideTapeFixStage.sequence.status.seqActive;
   #statTonTime[490].TON(IN := ("Unit1.Em4.ControlNodes".sideTapeFixStage.sequence.status.currentStep = #JOB_4_STEP_90) AND "Unit1.Em4.ControlNodes".sideTapeFixStage.sequence.status.seqActive AND "Unit1.Em4.ControlNodes".sideTapeFixStage."step".transition1[490],
                         PT := T#100ms);
   IF #statTonTime[490].Q THEN
       "Unit1.Em4.ControlNodes".sideTapeFixStage.sequence.status.nextStep := #STEP_IDLE;
   END_IF;
END_REGION

REGION Network 38: *************** JOB[5] SIDE TAPING-3=AUTO *************************
END_REGION

REGION Network 39: Step[501] : JOB[5] Condition
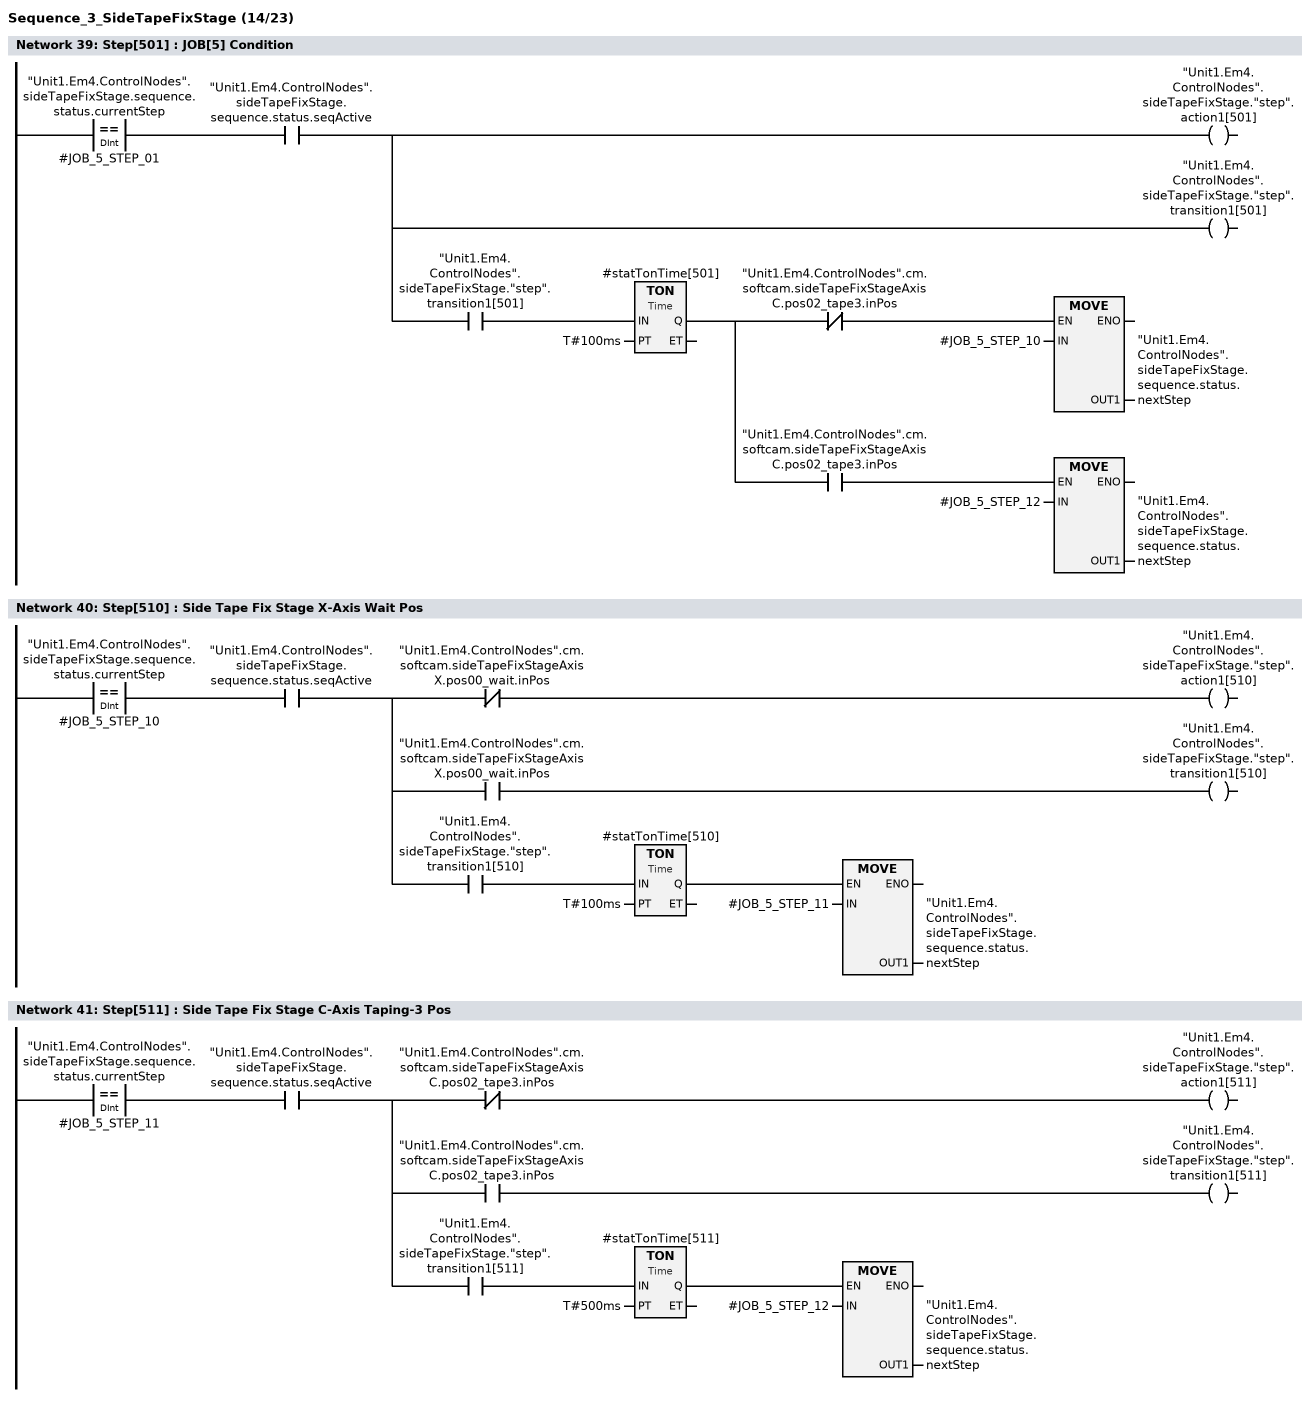
   RUNG wire#powerrail
      { S7_Templates := "SrcType := DInt" } EQ_Contact(in1 := "Unit1.Em4.ControlNodes".sideTapeFixStage.sequence.status.currentStep, in2 := #JOB_5_STEP_01)
      Contact( "Unit1.Em4.ControlNodes".sideTapeFixStage.sequence.status.seqActive )
      wire#w1
      Coil( "Unit1.Em4.ControlNodes".sideTapeFixStage."step".action1[501] )
   END_RUNG
   RUNG wire#w1
      Coil( "Unit1.Em4.ControlNodes".sideTapeFixStage."step".transition1[501] )
   END_RUNG
   RUNG wire#w1
      Contact( "Unit1.Em4.ControlNodes".sideTapeFixStage."step".transition1[501] )
      { S7_Templates := "time_type := Time" } #statTonTime[501].TON(pt := T#100ms, et =>)
      wire#w2
      I_Contact( "Unit1.Em4.ControlNodes".cm.softcam.sideTapeFixStageAxisC.pos02_tape3.inPos )
      Move(in := #JOB_5_STEP_10, out1 => "Unit1.Em4.ControlNodes".sideTapeFixStage.sequence.status.nextStep)
   END_RUNG
   RUNG wire#w2
      Contact( "Unit1.Em4.ControlNodes".cm.softcam.sideTapeFixStageAxisC.pos02_tape3.inPos )
      Move(in := #JOB_5_STEP_12, out1 => "Unit1.Em4.ControlNodes".sideTapeFixStage.sequence.status.nextStep)
   END_RUNG
   // the same network as SCL:
   "Unit1.Em4.ControlNodes".sideTapeFixStage."step".action1[501] := ("Unit1.Em4.ControlNodes".sideTapeFixStage.sequence.status.currentStep = #JOB_5_STEP_01) AND "Unit1.Em4.ControlNodes".sideTapeFixStage.sequence.status.seqActive;
   "Unit1.Em4.ControlNodes".sideTapeFixStage."step".transition1[501] := ("Unit1.Em4.ControlNodes".sideTapeFixStage.sequence.status.currentStep = #JOB_5_STEP_01) AND "Unit1.Em4.ControlNodes".sideTapeFixStage.sequence.status.seqActive;
   #statTonTime[501].TON(IN := ("Unit1.Em4.ControlNodes".sideTapeFixStage.sequence.status.currentStep = #JOB_5_STEP_01) AND "Unit1.Em4.ControlNodes".sideTapeFixStage.sequence.status.seqActive AND "Unit1.Em4.ControlNodes".sideTapeFixStage."step".transition1[501],
                         PT := T#100ms);
   IF #statTonTime[501].Q AND NOT "Unit1.Em4.ControlNodes".cm.softcam.sideTapeFixStageAxisC.pos02_tape3.inPos THEN
       "Unit1.Em4.ControlNodes".sideTapeFixStage.sequence.status.nextStep := #JOB_5_STEP_10;
   END_IF;
   IF #statTonTime[501].Q AND "Unit1.Em4.ControlNodes".cm.softcam.sideTapeFixStageAxisC.pos02_tape3.inPos THEN
       "Unit1.Em4.ControlNodes".sideTapeFixStage.sequence.status.nextStep := #JOB_5_STEP_12;
   END_IF;
END_REGION

REGION Network 40: Step[510] : Side Tape Fix Stage X-Axis Wait Pos
   RUNG wire#powerrail
      { S7_Templates := "SrcType := DInt" } EQ_Contact(in1 := "Unit1.Em4.ControlNodes".sideTapeFixStage.sequence.status.currentStep, in2 := #JOB_5_STEP_10)
      Contact( "Unit1.Em4.ControlNodes".sideTapeFixStage.sequence.status.seqActive )
      wire#w1
      I_Contact( "Unit1.Em4.ControlNodes".cm.softcam.sideTapeFixStageAxisX.pos00_wait.inPos )
      Coil( "Unit1.Em4.ControlNodes".sideTapeFixStage."step".action1[510] )
   END_RUNG
   RUNG wire#w1
      Contact( "Unit1.Em4.ControlNodes".cm.softcam.sideTapeFixStageAxisX.pos00_wait.inPos )
      Coil( "Unit1.Em4.ControlNodes".sideTapeFixStage."step".transition1[510] )
   END_RUNG
   RUNG wire#w1
      Contact( "Unit1.Em4.ControlNodes".sideTapeFixStage."step".transition1[510] )
      { S7_Templates := "time_type := Time" } #statTonTime[510].TON(pt := T#100ms, et =>)
      Move(in := #JOB_5_STEP_11, out1 => "Unit1.Em4.ControlNodes".sideTapeFixStage.sequence.status.nextStep)
   END_RUNG
   // the same network as SCL:
   #_w1 := ("Unit1.Em4.ControlNodes".sideTapeFixStage.sequence.status.currentStep = #JOB_5_STEP_10) AND "Unit1.Em4.ControlNodes".sideTapeFixStage.sequence.status.seqActive;
   "Unit1.Em4.ControlNodes".sideTapeFixStage."step".action1[510] := #_w1 AND NOT "Unit1.Em4.ControlNodes".cm.softcam.sideTapeFixStageAxisX.pos00_wait.inPos;
   "Unit1.Em4.ControlNodes".sideTapeFixStage."step".transition1[510] := #_w1 AND "Unit1.Em4.ControlNodes".cm.softcam.sideTapeFixStageAxisX.pos00_wait.inPos;
   #statTonTime[510].TON(IN := #_w1 AND "Unit1.Em4.ControlNodes".sideTapeFixStage."step".transition1[510],
                         PT := T#100ms);
   IF #statTonTime[510].Q THEN
       "Unit1.Em4.ControlNodes".sideTapeFixStage.sequence.status.nextStep := #JOB_5_STEP_11;
   END_IF;
END_REGION

REGION Network 41: Step[511] : Side Tape Fix Stage C-Axis Taping-3 Pos
   RUNG wire#powerrail
      { S7_Templates := "SrcType := DInt" } EQ_Contact(in1 := "Unit1.Em4.ControlNodes".sideTapeFixStage.sequence.status.currentStep, in2 := #JOB_5_STEP_11)
      Contact( "Unit1.Em4.ControlNodes".sideTapeFixStage.sequence.status.seqActive )
      wire#w1
      I_Contact( "Unit1.Em4.ControlNodes".cm.softcam.sideTapeFixStageAxisC.pos02_tape3.inPos )
      Coil( "Unit1.Em4.ControlNodes".sideTapeFixStage."step".action1[511] )
   END_RUNG
   RUNG wire#w1
      Contact( "Unit1.Em4.ControlNodes".cm.softcam.sideTapeFixStageAxisC.pos02_tape3.inPos )
      Coil( "Unit1.Em4.ControlNodes".sideTapeFixStage."step".transition1[511] )
   END_RUNG
   RUNG wire#w1
      Contact( "Unit1.Em4.ControlNodes".sideTapeFixStage."step".transition1[511] )
      { S7_Templates := "time_type := Time" } #statTonTime[511].TON(pt := T#500ms, et =>)
      Move(in := #JOB_5_STEP_12, out1 => "Unit1.Em4.ControlNodes".sideTapeFixStage.sequence.status.nextStep)
   END_RUNG
   // the same network as SCL:
   #_w1 := ("Unit1.Em4.ControlNodes".sideTapeFixStage.sequence.status.currentStep = #JOB_5_STEP_11) AND "Unit1.Em4.ControlNodes".sideTapeFixStage.sequence.status.seqActive;
   "Unit1.Em4.ControlNodes".sideTapeFixStage."step".action1[511] := #_w1 AND NOT "Unit1.Em4.ControlNodes".cm.softcam.sideTapeFixStageAxisC.pos02_tape3.inPos;
   "Unit1.Em4.ControlNodes".sideTapeFixStage."step".transition1[511] := #_w1 AND "Unit1.Em4.ControlNodes".cm.softcam.sideTapeFixStageAxisC.pos02_tape3.inPos;
   #statTonTime[511].TON(IN := #_w1 AND "Unit1.Em4.ControlNodes".sideTapeFixStage."step".transition1[511],
                         PT := T#500ms);
   IF #statTonTime[511].Q THEN
       "Unit1.Em4.ControlNodes".sideTapeFixStage.sequence.status.nextStep := #JOB_5_STEP_12;
   END_IF;
END_REGION

REGION Network 42: Step[512] : Side Tape Fix Stage X-Axis Wait Pos
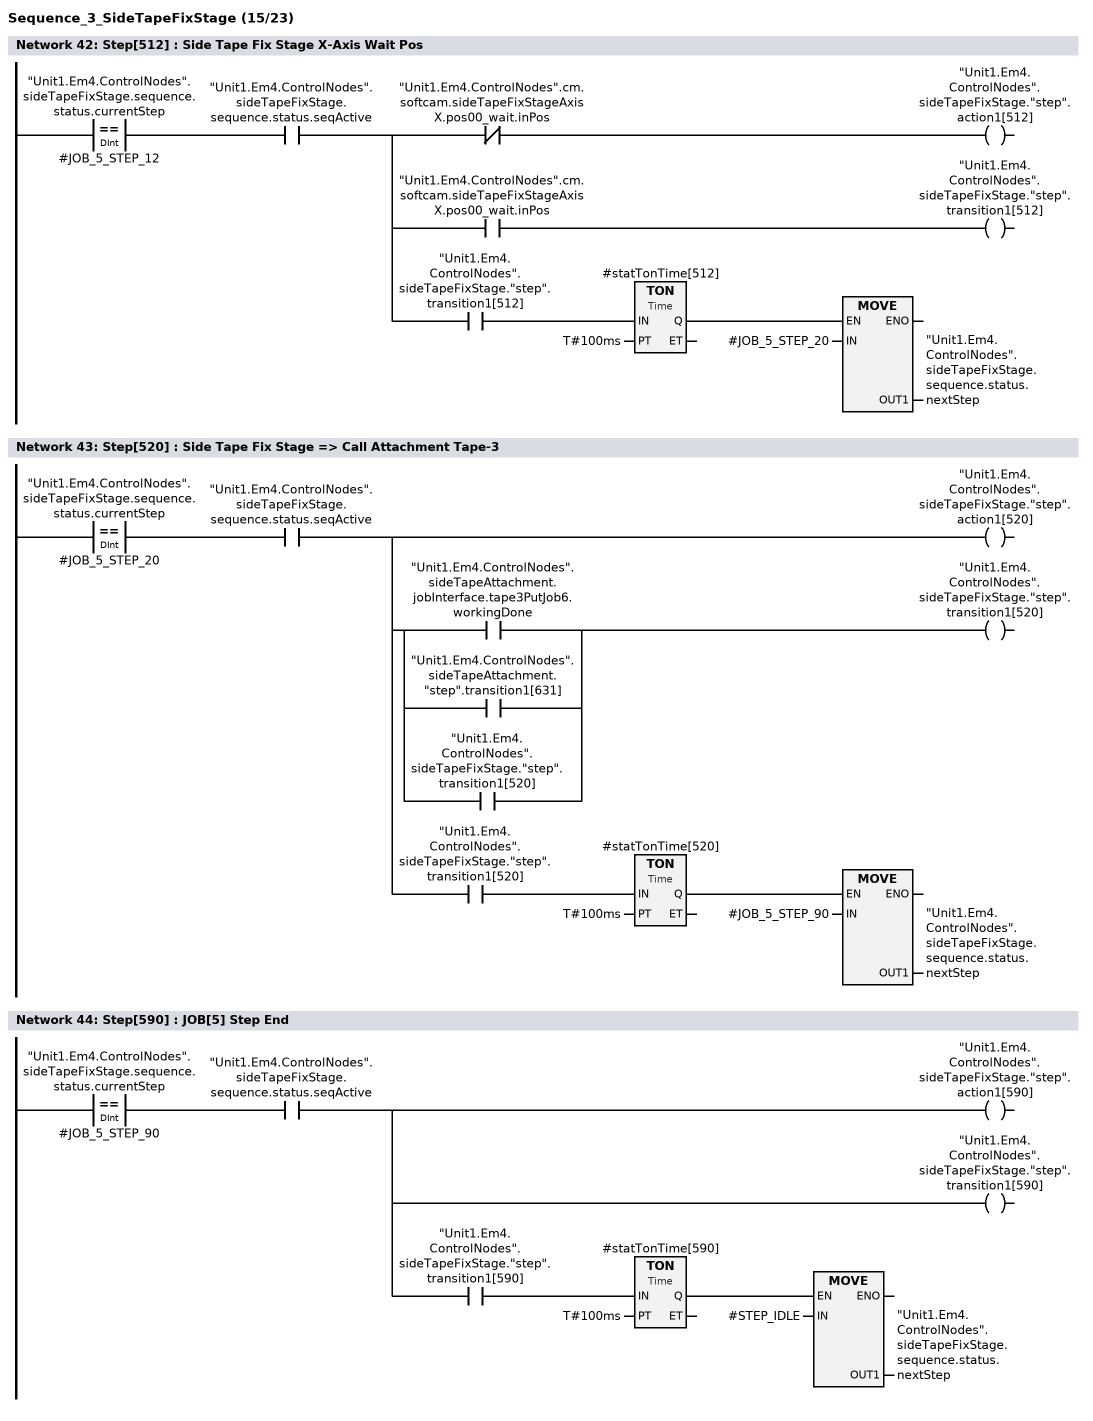
   RUNG wire#powerrail
      { S7_Templates := "SrcType := DInt" } EQ_Contact(in1 := "Unit1.Em4.ControlNodes".sideTapeFixStage.sequence.status.currentStep, in2 := #JOB_5_STEP_12)
      Contact( "Unit1.Em4.ControlNodes".sideTapeFixStage.sequence.status.seqActive )
      wire#w1
      I_Contact( "Unit1.Em4.ControlNodes".cm.softcam.sideTapeFixStageAxisX.pos00_wait.inPos )
      Coil( "Unit1.Em4.ControlNodes".sideTapeFixStage."step".action1[512] )
   END_RUNG
   RUNG wire#w1
      Contact( "Unit1.Em4.ControlNodes".cm.softcam.sideTapeFixStageAxisX.pos00_wait.inPos )
      Coil( "Unit1.Em4.ControlNodes".sideTapeFixStage."step".transition1[512] )
   END_RUNG
   RUNG wire#w1
      Contact( "Unit1.Em4.ControlNodes".sideTapeFixStage."step".transition1[512] )
      { S7_Templates := "time_type := Time" } #statTonTime[512].TON(pt := T#100ms, et =>)
      Move(in := #JOB_5_STEP_20, out1 => "Unit1.Em4.ControlNodes".sideTapeFixStage.sequence.status.nextStep)
   END_RUNG
   // the same network as SCL:
   #_w1 := ("Unit1.Em4.ControlNodes".sideTapeFixStage.sequence.status.currentStep = #JOB_5_STEP_12) AND "Unit1.Em4.ControlNodes".sideTapeFixStage.sequence.status.seqActive;
   "Unit1.Em4.ControlNodes".sideTapeFixStage."step".action1[512] := #_w1 AND NOT "Unit1.Em4.ControlNodes".cm.softcam.sideTapeFixStageAxisX.pos00_wait.inPos;
   "Unit1.Em4.ControlNodes".sideTapeFixStage."step".transition1[512] := #_w1 AND "Unit1.Em4.ControlNodes".cm.softcam.sideTapeFixStageAxisX.pos00_wait.inPos;
   #statTonTime[512].TON(IN := #_w1 AND "Unit1.Em4.ControlNodes".sideTapeFixStage."step".transition1[512],
                         PT := T#100ms);
   IF #statTonTime[512].Q THEN
       "Unit1.Em4.ControlNodes".sideTapeFixStage.sequence.status.nextStep := #JOB_5_STEP_20;
   END_IF;
END_REGION

REGION Network 43: Step[520] : Side Tape Fix Stage => Call Attachment Tape-3
   RUNG wire#powerrail
      { S7_Templates := "SrcType := DInt" } EQ_Contact(in1 := "Unit1.Em4.ControlNodes".sideTapeFixStage.sequence.status.currentStep, in2 := #JOB_5_STEP_20)
      Contact( "Unit1.Em4.ControlNodes".sideTapeFixStage.sequence.status.seqActive )
      wire#w1
      Coil( "Unit1.Em4.ControlNodes".sideTapeFixStage."step".action1[520] )
   END_RUNG
   RUNG wire#w1
      Contact( "Unit1.Em4.ControlNodes".sideTapeAttachment.jobInterface.tape3PutJob6.workingDone )
      wire#w2
      Coil( "Unit1.Em4.ControlNodes".sideTapeFixStage."step".transition1[520] )
   END_RUNG
   RUNG wire#w1
      Contact( "Unit1.Em4.ControlNodes".sideTapeAttachment."step".transition1[631] )
   END_RUNG wire#w2
   RUNG wire#w1
      Contact( "Unit1.Em4.ControlNodes".sideTapeFixStage."step".transition1[520] )
   END_RUNG wire#w2
   RUNG wire#w1
      Contact( "Unit1.Em4.ControlNodes".sideTapeFixStage."step".transition1[520] )
      { S7_Templates := "time_type := Time" } #statTonTime[520].TON(pt := T#100ms, et =>)
      Move(in := #JOB_5_STEP_90, out1 => "Unit1.Em4.ControlNodes".sideTapeFixStage.sequence.status.nextStep)
   END_RUNG
   // the same network as SCL:
   "Unit1.Em4.ControlNodes".sideTapeFixStage."step".action1[520] := ("Unit1.Em4.ControlNodes".sideTapeFixStage.sequence.status.currentStep = #JOB_5_STEP_20) AND "Unit1.Em4.ControlNodes".sideTapeFixStage.sequence.status.seqActive;
   "Unit1.Em4.ControlNodes".sideTapeFixStage."step".transition1[520] := ("Unit1.Em4.ControlNodes".sideTapeFixStage.sequence.status.currentStep = #JOB_5_STEP_20) AND "Unit1.Em4.ControlNodes".sideTapeFixStage.sequence.status.seqActive AND ("Unit1.Em4.ControlNodes".sideTapeAttachment.jobInterface.tape3PutJob6.workingDone OR "Unit1.Em4.ControlNodes".sideTapeAttachment."step".transition1[631] OR "Unit1.Em4.ControlNodes".sideTapeFixStage."step".transition1[520]);
   #statTonTime[520].TON(IN := ("Unit1.Em4.ControlNodes".sideTapeFixStage.sequence.status.currentStep = #JOB_5_STEP_20) AND "Unit1.Em4.ControlNodes".sideTapeFixStage.sequence.status.seqActive AND "Unit1.Em4.ControlNodes".sideTapeFixStage."step".transition1[520],
                         PT := T#100ms);
   IF #statTonTime[520].Q THEN
       "Unit1.Em4.ControlNodes".sideTapeFixStage.sequence.status.nextStep := #JOB_5_STEP_90;
   END_IF;
END_REGION

REGION Network 44: Step[590] : JOB[5] Step End
   RUNG wire#powerrail
      { S7_Templates := "SrcType := DInt" } EQ_Contact(in1 := "Unit1.Em4.ControlNodes".sideTapeFixStage.sequence.status.currentStep, in2 := #JOB_5_STEP_90)
      Contact( "Unit1.Em4.ControlNodes".sideTapeFixStage.sequence.status.seqActive )
      wire#w1
      Coil( "Unit1.Em4.ControlNodes".sideTapeFixStage."step".action1[590] )
   END_RUNG
   RUNG wire#w1
      Coil( "Unit1.Em4.ControlNodes".sideTapeFixStage."step".transition1[590] )
   END_RUNG
   RUNG wire#w1
      Contact( "Unit1.Em4.ControlNodes".sideTapeFixStage."step".transition1[590] )
      { S7_Templates := "time_type := Time" } #statTonTime[590].TON(pt := T#100ms, et =>)
      Move(in := #STEP_IDLE, out1 => "Unit1.Em4.ControlNodes".sideTapeFixStage.sequence.status.nextStep)
   END_RUNG
   // the same network as SCL:
   "Unit1.Em4.ControlNodes".sideTapeFixStage."step".action1[590] := ("Unit1.Em4.ControlNodes".sideTapeFixStage.sequence.status.currentStep = #JOB_5_STEP_90) AND "Unit1.Em4.ControlNodes".sideTapeFixStage.sequence.status.seqActive;
   "Unit1.Em4.ControlNodes".sideTapeFixStage."step".transition1[590] := ("Unit1.Em4.ControlNodes".sideTapeFixStage.sequence.status.currentStep = #JOB_5_STEP_90) AND "Unit1.Em4.ControlNodes".sideTapeFixStage.sequence.status.seqActive;
   #statTonTime[590].TON(IN := ("Unit1.Em4.ControlNodes".sideTapeFixStage.sequence.status.currentStep = #JOB_5_STEP_90) AND "Unit1.Em4.ControlNodes".sideTapeFixStage.sequence.status.seqActive AND "Unit1.Em4.ControlNodes".sideTapeFixStage."step".transition1[590],
                         PT := T#100ms);
   IF #statTonTime[590].Q THEN
       "Unit1.Em4.ControlNodes".sideTapeFixStage.sequence.status.nextStep := #STEP_IDLE;
   END_IF;
END_REGION

REGION Network 45: *************** JOB[6] SIDE TAPING-4=AUTO *************************
END_REGION

REGION Network 46: Step[601] : JOB[6] Condition
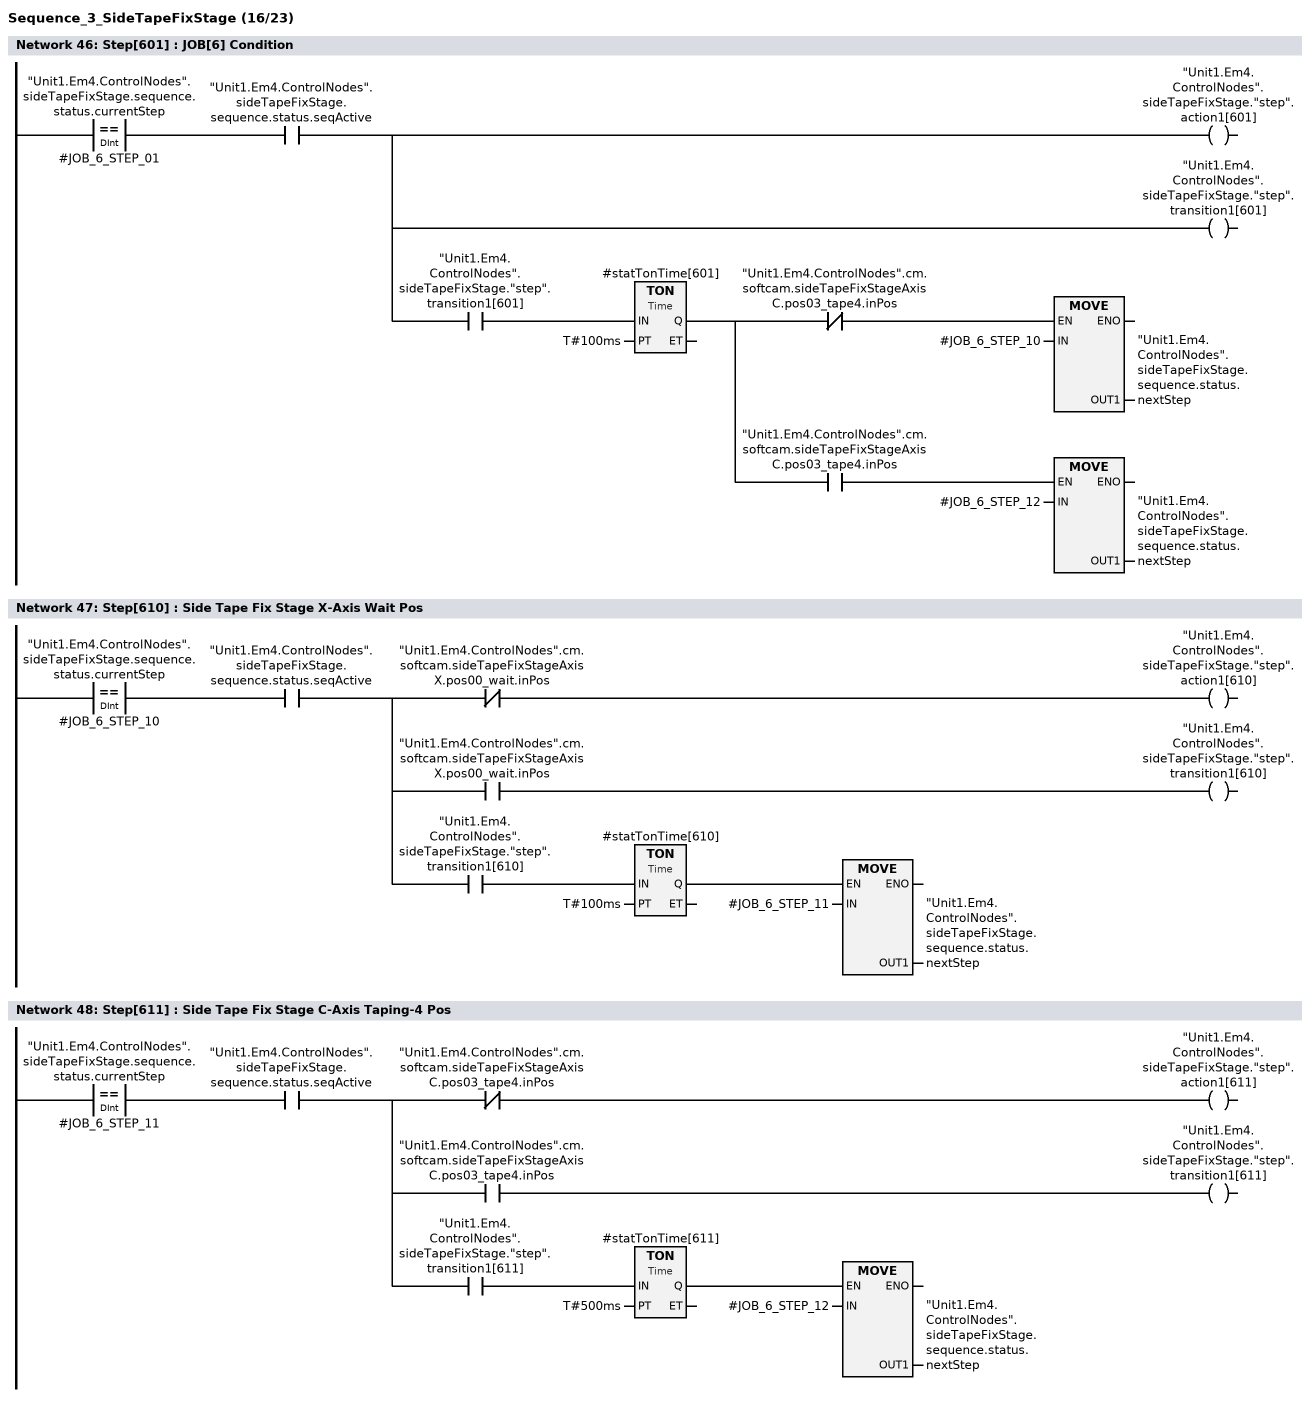
   RUNG wire#powerrail
      { S7_Templates := "SrcType := DInt" } EQ_Contact(in1 := "Unit1.Em4.ControlNodes".sideTapeFixStage.sequence.status.currentStep, in2 := #JOB_6_STEP_01)
      Contact( "Unit1.Em4.ControlNodes".sideTapeFixStage.sequence.status.seqActive )
      wire#w1
      Coil( "Unit1.Em4.ControlNodes".sideTapeFixStage."step".action1[601] )
   END_RUNG
   RUNG wire#w1
      Coil( "Unit1.Em4.ControlNodes".sideTapeFixStage."step".transition1[601] )
   END_RUNG
   RUNG wire#w1
      Contact( "Unit1.Em4.ControlNodes".sideTapeFixStage."step".transition1[601] )
      { S7_Templates := "time_type := Time" } #statTonTime[601].TON(pt := T#100ms, et =>)
      wire#w2
      I_Contact( "Unit1.Em4.ControlNodes".cm.softcam.sideTapeFixStageAxisC.pos03_tape4.inPos )
      Move(in := #JOB_6_STEP_10, out1 => "Unit1.Em4.ControlNodes".sideTapeFixStage.sequence.status.nextStep)
   END_RUNG
   RUNG wire#w2
      Contact( "Unit1.Em4.ControlNodes".cm.softcam.sideTapeFixStageAxisC.pos03_tape4.inPos )
      Move(in := #JOB_6_STEP_12, out1 => "Unit1.Em4.ControlNodes".sideTapeFixStage.sequence.status.nextStep)
   END_RUNG
   // the same network as SCL:
   "Unit1.Em4.ControlNodes".sideTapeFixStage."step".action1[601] := ("Unit1.Em4.ControlNodes".sideTapeFixStage.sequence.status.currentStep = #JOB_6_STEP_01) AND "Unit1.Em4.ControlNodes".sideTapeFixStage.sequence.status.seqActive;
   "Unit1.Em4.ControlNodes".sideTapeFixStage."step".transition1[601] := ("Unit1.Em4.ControlNodes".sideTapeFixStage.sequence.status.currentStep = #JOB_6_STEP_01) AND "Unit1.Em4.ControlNodes".sideTapeFixStage.sequence.status.seqActive;
   #statTonTime[601].TON(IN := ("Unit1.Em4.ControlNodes".sideTapeFixStage.sequence.status.currentStep = #JOB_6_STEP_01) AND "Unit1.Em4.ControlNodes".sideTapeFixStage.sequence.status.seqActive AND "Unit1.Em4.ControlNodes".sideTapeFixStage."step".transition1[601],
                         PT := T#100ms);
   IF #statTonTime[601].Q AND NOT "Unit1.Em4.ControlNodes".cm.softcam.sideTapeFixStageAxisC.pos03_tape4.inPos THEN
       "Unit1.Em4.ControlNodes".sideTapeFixStage.sequence.status.nextStep := #JOB_6_STEP_10;
   END_IF;
   IF #statTonTime[601].Q AND "Unit1.Em4.ControlNodes".cm.softcam.sideTapeFixStageAxisC.pos03_tape4.inPos THEN
       "Unit1.Em4.ControlNodes".sideTapeFixStage.sequence.status.nextStep := #JOB_6_STEP_12;
   END_IF;
END_REGION

REGION Network 47: Step[610] : Side Tape Fix Stage X-Axis Wait Pos
   RUNG wire#powerrail
      { S7_Templates := "SrcType := DInt" } EQ_Contact(in1 := "Unit1.Em4.ControlNodes".sideTapeFixStage.sequence.status.currentStep, in2 := #JOB_6_STEP_10)
      Contact( "Unit1.Em4.ControlNodes".sideTapeFixStage.sequence.status.seqActive )
      wire#w1
      I_Contact( "Unit1.Em4.ControlNodes".cm.softcam.sideTapeFixStageAxisX.pos00_wait.inPos )
      Coil( "Unit1.Em4.ControlNodes".sideTapeFixStage."step".action1[610] )
   END_RUNG
   RUNG wire#w1
      Contact( "Unit1.Em4.ControlNodes".cm.softcam.sideTapeFixStageAxisX.pos00_wait.inPos )
      Coil( "Unit1.Em4.ControlNodes".sideTapeFixStage."step".transition1[610] )
   END_RUNG
   RUNG wire#w1
      Contact( "Unit1.Em4.ControlNodes".sideTapeFixStage."step".transition1[610] )
      { S7_Templates := "time_type := Time" } #statTonTime[610].TON(pt := T#100ms, et =>)
      Move(in := #JOB_6_STEP_11, out1 => "Unit1.Em4.ControlNodes".sideTapeFixStage.sequence.status.nextStep)
   END_RUNG
   // the same network as SCL:
   #_w1 := ("Unit1.Em4.ControlNodes".sideTapeFixStage.sequence.status.currentStep = #JOB_6_STEP_10) AND "Unit1.Em4.ControlNodes".sideTapeFixStage.sequence.status.seqActive;
   "Unit1.Em4.ControlNodes".sideTapeFixStage."step".action1[610] := #_w1 AND NOT "Unit1.Em4.ControlNodes".cm.softcam.sideTapeFixStageAxisX.pos00_wait.inPos;
   "Unit1.Em4.ControlNodes".sideTapeFixStage."step".transition1[610] := #_w1 AND "Unit1.Em4.ControlNodes".cm.softcam.sideTapeFixStageAxisX.pos00_wait.inPos;
   #statTonTime[610].TON(IN := #_w1 AND "Unit1.Em4.ControlNodes".sideTapeFixStage."step".transition1[610],
                         PT := T#100ms);
   IF #statTonTime[610].Q THEN
       "Unit1.Em4.ControlNodes".sideTapeFixStage.sequence.status.nextStep := #JOB_6_STEP_11;
   END_IF;
END_REGION

REGION Network 48: Step[611] : Side Tape Fix Stage C-Axis Taping-4 Pos
   RUNG wire#powerrail
      { S7_Templates := "SrcType := DInt" } EQ_Contact(in1 := "Unit1.Em4.ControlNodes".sideTapeFixStage.sequence.status.currentStep, in2 := #JOB_6_STEP_11)
      Contact( "Unit1.Em4.ControlNodes".sideTapeFixStage.sequence.status.seqActive )
      wire#w1
      I_Contact( "Unit1.Em4.ControlNodes".cm.softcam.sideTapeFixStageAxisC.pos03_tape4.inPos )
      Coil( "Unit1.Em4.ControlNodes".sideTapeFixStage."step".action1[611] )
   END_RUNG
   RUNG wire#w1
      Contact( "Unit1.Em4.ControlNodes".cm.softcam.sideTapeFixStageAxisC.pos03_tape4.inPos )
      Coil( "Unit1.Em4.ControlNodes".sideTapeFixStage."step".transition1[611] )
   END_RUNG
   RUNG wire#w1
      Contact( "Unit1.Em4.ControlNodes".sideTapeFixStage."step".transition1[611] )
      { S7_Templates := "time_type := Time" } #statTonTime[611].TON(pt := T#500ms, et =>)
      Move(in := #JOB_6_STEP_12, out1 => "Unit1.Em4.ControlNodes".sideTapeFixStage.sequence.status.nextStep)
   END_RUNG
   // the same network as SCL:
   #_w1 := ("Unit1.Em4.ControlNodes".sideTapeFixStage.sequence.status.currentStep = #JOB_6_STEP_11) AND "Unit1.Em4.ControlNodes".sideTapeFixStage.sequence.status.seqActive;
   "Unit1.Em4.ControlNodes".sideTapeFixStage."step".action1[611] := #_w1 AND NOT "Unit1.Em4.ControlNodes".cm.softcam.sideTapeFixStageAxisC.pos03_tape4.inPos;
   "Unit1.Em4.ControlNodes".sideTapeFixStage."step".transition1[611] := #_w1 AND "Unit1.Em4.ControlNodes".cm.softcam.sideTapeFixStageAxisC.pos03_tape4.inPos;
   #statTonTime[611].TON(IN := #_w1 AND "Unit1.Em4.ControlNodes".sideTapeFixStage."step".transition1[611],
                         PT := T#500ms);
   IF #statTonTime[611].Q THEN
       "Unit1.Em4.ControlNodes".sideTapeFixStage.sequence.status.nextStep := #JOB_6_STEP_12;
   END_IF;
END_REGION

REGION Network 49: Step[612] : Side Tape Fix Stage X-Axis Wait Pos
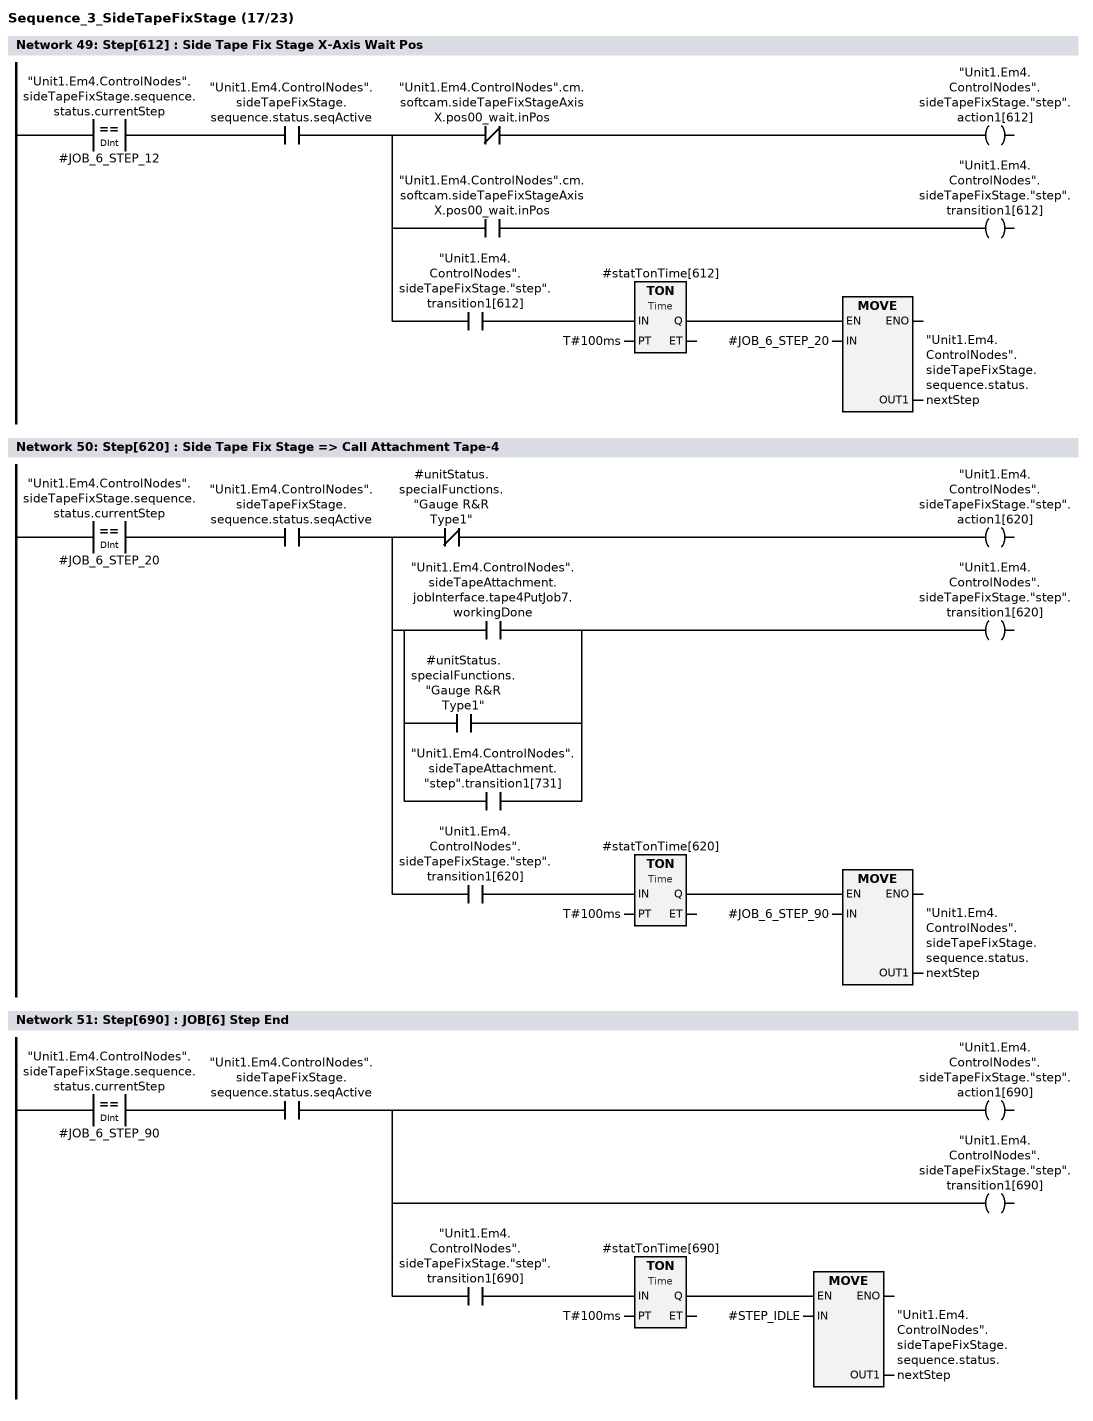
   RUNG wire#powerrail
      { S7_Templates := "SrcType := DInt" } EQ_Contact(in1 := "Unit1.Em4.ControlNodes".sideTapeFixStage.sequence.status.currentStep, in2 := #JOB_6_STEP_12)
      Contact( "Unit1.Em4.ControlNodes".sideTapeFixStage.sequence.status.seqActive )
      wire#w1
      I_Contact( "Unit1.Em4.ControlNodes".cm.softcam.sideTapeFixStageAxisX.pos00_wait.inPos )
      Coil( "Unit1.Em4.ControlNodes".sideTapeFixStage."step".action1[612] )
   END_RUNG
   RUNG wire#w1
      Contact( "Unit1.Em4.ControlNodes".cm.softcam.sideTapeFixStageAxisX.pos00_wait.inPos )
      Coil( "Unit1.Em4.ControlNodes".sideTapeFixStage."step".transition1[612] )
   END_RUNG
   RUNG wire#w1
      Contact( "Unit1.Em4.ControlNodes".sideTapeFixStage."step".transition1[612] )
      { S7_Templates := "time_type := Time" } #statTonTime[612].TON(pt := T#100ms, et =>)
      Move(in := #JOB_6_STEP_20, out1 => "Unit1.Em4.ControlNodes".sideTapeFixStage.sequence.status.nextStep)
   END_RUNG
   // the same network as SCL:
   #_w1 := ("Unit1.Em4.ControlNodes".sideTapeFixStage.sequence.status.currentStep = #JOB_6_STEP_12) AND "Unit1.Em4.ControlNodes".sideTapeFixStage.sequence.status.seqActive;
   "Unit1.Em4.ControlNodes".sideTapeFixStage."step".action1[612] := #_w1 AND NOT "Unit1.Em4.ControlNodes".cm.softcam.sideTapeFixStageAxisX.pos00_wait.inPos;
   "Unit1.Em4.ControlNodes".sideTapeFixStage."step".transition1[612] := #_w1 AND "Unit1.Em4.ControlNodes".cm.softcam.sideTapeFixStageAxisX.pos00_wait.inPos;
   #statTonTime[612].TON(IN := #_w1 AND "Unit1.Em4.ControlNodes".sideTapeFixStage."step".transition1[612],
                         PT := T#100ms);
   IF #statTonTime[612].Q THEN
       "Unit1.Em4.ControlNodes".sideTapeFixStage.sequence.status.nextStep := #JOB_6_STEP_20;
   END_IF;
END_REGION

REGION Network 50: Step[620] : Side Tape Fix Stage => Call Attachment Tape-4
   RUNG wire#powerrail
      { S7_Templates := "SrcType := DInt" } EQ_Contact(in1 := "Unit1.Em4.ControlNodes".sideTapeFixStage.sequence.status.currentStep, in2 := #JOB_6_STEP_20)
      Contact( "Unit1.Em4.ControlNodes".sideTapeFixStage.sequence.status.seqActive )
      wire#w1
      I_Contact( #unitStatus.specialFunctions."Gauge R&R Type1" )
      Coil( "Unit1.Em4.ControlNodes".sideTapeFixStage."step".action1[620] )
   END_RUNG
   RUNG wire#w1
      Contact( "Unit1.Em4.ControlNodes".sideTapeAttachment.jobInterface.tape4PutJob7.workingDone )
      wire#w2
      Coil( "Unit1.Em4.ControlNodes".sideTapeFixStage."step".transition1[620] )
   END_RUNG
   RUNG wire#w1
      Contact( #unitStatus.specialFunctions."Gauge R&R Type1" )
   END_RUNG wire#w2
   RUNG wire#w1
      Contact( "Unit1.Em4.ControlNodes".sideTapeAttachment."step".transition1[731] )
   END_RUNG wire#w2
   RUNG wire#w1
      Contact( "Unit1.Em4.ControlNodes".sideTapeFixStage."step".transition1[620] )
      { S7_Templates := "time_type := Time" } #statTonTime[620].TON(pt := T#100ms, et =>)
      Move(in := #JOB_6_STEP_90, out1 => "Unit1.Em4.ControlNodes".sideTapeFixStage.sequence.status.nextStep)
   END_RUNG
   // the same network as SCL:
   #_w1 := ("Unit1.Em4.ControlNodes".sideTapeFixStage.sequence.status.currentStep = #JOB_6_STEP_20) AND "Unit1.Em4.ControlNodes".sideTapeFixStage.sequence.status.seqActive;
   "Unit1.Em4.ControlNodes".sideTapeFixStage."step".action1[620] := #_w1 AND NOT #unitStatus.specialFunctions."Gauge R&R Type1";
   "Unit1.Em4.ControlNodes".sideTapeFixStage."step".transition1[620] := #_w1 AND ("Unit1.Em4.ControlNodes".sideTapeAttachment.jobInterface.tape4PutJob7.workingDone OR #unitStatus.specialFunctions."Gauge R&R Type1" OR "Unit1.Em4.ControlNodes".sideTapeAttachment."step".transition1[731]);
   #statTonTime[620].TON(IN := #_w1 AND "Unit1.Em4.ControlNodes".sideTapeFixStage."step".transition1[620],
                         PT := T#100ms);
   IF #statTonTime[620].Q THEN
       "Unit1.Em4.ControlNodes".sideTapeFixStage.sequence.status.nextStep := #JOB_6_STEP_90;
   END_IF;
END_REGION

